E1_2004 CHANNEL  ; 侧压B3左伺服JOG低速
E1_2005 CHANNEL  ; 侧压B3左伺服JOG低速
E1_2006 CHANNEL  ; 侧压B3左伺服加速时间
E1_2007 CHANNEL  ; 侧压B3左伺服加速时间
E1_2008 CHANNEL  ; 侧压B3左伺服减速时间
E1_2009 CHANNEL  ; 侧压B3左伺服减速时间
E1_201 CHANNEL  ; NC433_2_X轴当前位置
E1_2010 CHANNEL  ; 侧压B3左伺服原点偏移
E1_2011 CHANNEL  ; 侧压B3左伺服原点偏移
E1_2012 CHANNEL  ; 侧压B3左伺服正软极限
E1_2013 CHANNEL  ; 侧压B3左伺服正软极限
E1_2014 CHANNEL  ; 侧压B3左伺服负软极限
E1_2015 CHANNEL  ; 负软极限
E1_202 CHANNEL  ; NC433_2_X轴存储器操作正被执行序列号
E1_2020 CHANNEL  ; 侧压B3左伺服待机位
E1_2021 CHANNEL  ; 侧压B3左伺服待机位
E1_2022 CHANNEL  ; 侧压B3左伺服拨料退回位
E1_2023 CHANNEL  ; 侧压B3左伺服拨料退回位
E1_2024 CHANNEL  ; 侧压B3左伺服拨料位
E1_2025 CHANNEL  ; 侧压B3左伺服拨料位
E1_2026 CHANNEL  ; 侧压B3左伺服减速位
E1_2027 CHANNEL  ; 侧压B3左伺服减速位
E1_2028 CHANNEL  ; 侧压B3左伺服等距热压位
E1_2029 CHANNEL  ; 侧压B3左伺服等距热压位
E1_203 CHANNEL  ; NC433_2_X轴存储器操作正被执行序列号
E1_2030 CHANNEL  ; 侧压B3左伺服6#位
E1_2031 CHANNEL  ; 侧压B3左伺服6#位
E1_2032 CHANNEL  ; 侧压B3左伺服7#位
E1_2033 CHANNEL  ; 侧压B3左伺服7#位
E1_2034 CHANNEL  ; 侧压B3左伺服8#位
E1_2035 CHANNEL  ; 侧压B3左伺服8#位
E1_2036 CHANNEL  ; 侧压B3左伺服9#位
E1_2037 CHANNEL  ; 侧压B3左伺服9#位
E1_2038 CHANNEL  ; 侧压B3左伺服10#位
E1_2039 CHANNEL  ; 侧压B3左伺服10#位
E1_204 CHANNEL  ; NC433_2_Y轴当前位置
E1_2046 CHANNEL  ; B3两轴回原宽度
E1_205 CHANNEL  ; NC433_2_Y轴当前位置
E1_2050 CHANNEL  ; 侧压B3右伺服自动速度
E1_2051 CHANNEL  ; 侧压B3右伺服自动速度
E1_2052 CHANNEL  ; 侧压B3右伺服JOG高速
E1_2053 CHANNEL  ; 侧压B3右伺服JOG高速
E1_2054 CHANNEL  ; 侧压B3右伺服JOG低速
E1_2055 CHANNEL  ; 侧压B3右伺服JOG低速
E1_2056 CHANNEL  ; 侧压B3右伺服加速时间
E1_2057 CHANNEL  ; 侧压B3右伺服加速时间
E1_2058 CHANNEL  ; 侧压B3右伺服减速时间
E1_2059 CHANNEL  ; 侧压B3右伺服减速时间
E1_206 CHANNEL  ; NC433_2_Y轴存储器操作正被执行序列号
E1_2060 CHANNEL  ; 侧压B3右伺服原点偏移
E1_2061 CHANNEL  ; 侧压B3右伺服原点偏移
E1_2062 CHANNEL  ; 侧压B3右伺服正软极限
E1_2063 CHANNEL  ; 侧压B3右伺服正软极限
E1_2064 CHANNEL  ; 侧压B3右伺服负软极限
E1_2065 CHANNEL  ; 负软极限
E1_207 CHANNEL  ; NC433_2_Y轴存储器操作正被执行序列号
E1_2070 CHANNEL  ; 侧压B3右伺服待机位
E1_2071 CHANNEL  ; 侧压B3右伺服待机位
E1_2072 CHANNEL  ; 侧压B3右伺服拨料退回位
E1_2073 CHANNEL  ; 侧压B3右伺服拨料退回位
E1_2074 CHANNEL  ; 侧压B3右伺服拨料位
E1_2075 CHANNEL  ; 侧压B3右伺服拨料位
E1_2076 CHANNEL  ; 侧压B3右伺服减速位
E1_2077 CHANNEL  ; 侧压B3右伺服减速位
E1_2078 CHANNEL  ; 侧压B3右伺服等距热压位
E1_2079 CHANNEL  ; 侧压B3右伺服等距热压位
E1_208 CHANNEL  ; NC433_2_Z轴当前位置
E1_2080 CHANNEL  ; 侧压B3右伺服6#位
E1_2081 CHANNEL  ; 侧压B3右伺服6#位
E1_2082 CHANNEL  ; 侧压B3右伺服7#位
E1_2083 CHANNEL  ; 侧压B3右伺服7#位
E1_2084 CHANNEL  ; 侧压B3右伺服8#位
E1_2085 CHANNEL  ; 侧压B3右伺服8#位
E1_2086 CHANNEL  ; 侧压B3右伺服9#位
E1_2087 CHANNEL  ; 侧压B3右伺服9#位
E1_2088 CHANNEL  ; 侧压B3右伺服10#位
E1_2089 CHANNEL  ; 侧压B3右伺服10#位
E1_209 CHANNEL  ; NC433_2_Z轴当前位置
E1_21 CHANNEL  ; NC433_0_Y轴直接操作位置
E1_210 CHANNEL  ; NC433_2_Z轴存储器操作正被执行序列号
E1_2100 CHANNEL  ; 侧压B4左伺服自动速度
E1_2101 CHANNEL  ; 侧压B4左伺服自动速度
E1_2102 CHANNEL  ; 侧压B4左伺服JOG高速
E1_2103 CHANNEL  ; 侧压B4左伺服JOG高速
E1_2104 CHANNEL  ; 侧压B4左伺服JOG低速
E1_2105 CHANNEL  ; 侧压B4左伺服JOG低速
E1_2106 CHANNEL  ; 侧压B4左伺服加速时间
E1_2107 CHANNEL  ; 侧压B4左伺服加速时间
E1_2108 CHANNEL  ; 侧压B4左伺服减速时间
E1_2109 CHANNEL  ; 侧压B4左伺服减速时间
E1_211 CHANNEL  ; NC433_2_Z轴存储器操作正被执行序列号
E1_2110 CHANNEL  ; 侧压B4左伺服原点偏移
E1_2111 CHANNEL  ; 侧压B4左伺服原点偏移
E1_2112 CHANNEL  ; 侧压B4左伺服正软极限
E1_2113 CHANNEL  ; 侧压B4左伺服正软极限
E1_2114 CHANNEL  ; 侧压B4左伺服负软极限
E1_2115 CHANNEL  ; 负软极限
E1_212 CHANNEL  ; NC433_2_U轴当前位置
E1_2120 CHANNEL  ; 侧压B4左伺服待机位
E1_2121 CHANNEL  ; 侧压B4左伺服待机位
E1_2122 CHANNEL  ; 侧压B4左伺服拨料退回位
E1_2123 CHANNEL  ; 侧压B4左伺服拨料退回位
E1_2124 CHANNEL  ; 侧压B4左伺服拨料位
E1_2125 CHANNEL  ; 侧压B4左伺服拨料位
E1_2126 CHANNEL  ; 侧压B4左伺服减速位
E1_2127 CHANNEL  ; 侧压B4左伺服减速位
E1_2128 CHANNEL  ; 侧压B4左伺服等距热压位
E1_2129 CHANNEL  ; 侧压B4左伺服等距热压位
E1_213 CHANNEL  ; NC433_2_U轴当前位置
E1_2130 CHANNEL  ; 侧压B4左伺服6#位
E1_2131 CHANNEL  ; 侧压B4左伺服6#位
E1_2132 CHANNEL  ; 侧压B4左伺服7#位
E1_2133 CHANNEL  ; 侧压B4左伺服7#位
E1_2134 CHANNEL  ; 侧压B4左伺服8#位
E1_2135 CHANNEL  ; 侧压B4左伺服8#位
E1_2136 CHANNEL  ; 侧压B4左伺服9#位
E1_2137 CHANNEL  ; 侧压B4左伺服9#位
E1_2138 CHANNEL  ; 侧压B4左伺服10#位
E1_2139 CHANNEL  ; 侧压B4左伺服10#位
E1_214 CHANNEL  ; NC433_2_U轴存储器操作正被执行序列号
E1_2146 CHANNEL  ; B4两轴回原宽度
E1_215 CHANNEL  ; NC433_2_U轴存储器操作正被执行序列号
E1_2150 CHANNEL  ; 侧压B4右伺服自动速度
E1_2151 CHANNEL  ; 侧压B4右伺服自动速度
E1_2152 CHANNEL  ; 侧压B4右伺服JOG高速
E1_2153 CHANNEL  ; 侧压B4右伺服JOG高速
E1_2154 CHANNEL  ; 侧压B4右伺服JOG低速
E1_2155 CHANNEL  ; 侧压B4右伺服JOG低速
E1_2156 CHANNEL  ; 侧压B4右伺服加速时间
E1_2157 CHANNEL  ; 侧压B4右伺服加速时间
E1_2158 CHANNEL  ; 侧压B4右伺服减速时间
E1_2159 CHANNEL  ; 侧压B4右伺服减速时间
E1_216 CHANNEL  ; NC433_3 数据传送写字数
E1_2160 CHANNEL  ; 侧压B4右伺服原点偏移
E1_2161 CHANNEL  ; 侧压B4右伺服原点偏移
E1_2162 CHANNEL  ; 侧压B4右伺服正软极限
E1_2163 CHANNEL  ; 侧压B4右伺服正软极限
E1_2164 CHANNEL  ; 侧压B4右伺服负软极限
E1_2165 CHANNEL  ; 负软极限
E1_217 CHANNEL  ; NC433_3 数据传送写源区域
E1_2170 CHANNEL  ; 侧压B4右伺服待机位
E1_2171 CHANNEL  ; 侧压B4右伺服待机位
E1_2172 CHANNEL  ; 侧压B4右伺服拨料退回位
E1_2173 CHANNEL  ; 侧压B4右伺服拨料退回位
E1_2174 CHANNEL  ; 侧压B4右伺服拨料位
E1_2175 CHANNEL  ; 侧压B4右伺服拨料位
E1_2176 CHANNEL  ; 侧压B4右伺服减速位
E1_2177 CHANNEL  ; 侧压B4右伺服减速位
E1_2178 CHANNEL  ; 侧压B4右伺服等距热压位
E1_2179 CHANNEL  ; 侧压B4右伺服等距热压位
E1_218 CHANNEL  ; NC433_3 数据传送定源字
E1_2180 CHANNEL  ; 侧压B4右伺服6#位
E1_2181 CHANNEL  ; 侧压B4右伺服6#位
E1_2182 CHANNEL  ; 侧压B4右伺服7#位
E1_2183 CHANNEL  ; 侧压B4右伺服7#位
E1_2184 CHANNEL  ; 侧压B4右伺服8#位
E1_2185 CHANNEL  ; 侧压B4右伺服8#位
E1_2186 CHANNEL  ; 侧压B4右伺服9#位
E1_2187 CHANNEL  ; 侧压B4右伺服9#位
E1_2188 CHANNEL  ; 侧压B4右伺服10#位
E1_2189 CHANNEL  ; 侧压B4右伺服10#位
E1_219 CHANNEL  ; NC433_3 数据传送定目标地址
E1_22 CHANNEL  ; NC433_0_Y轴直接操作速度
E1_220 CHANNEL  ; NC433_3 数据传送读字数
E1_2200 CHANNEL  ; 25#伺服自动速度
E1_2201 CHANNEL  ; 25#伺服自动速度
E1_2202 CHANNEL  ; 25#伺服JOG高速
E1_2203 CHANNEL  ; 25#伺服JOG高速
E1_2204 CHANNEL  ; 25#伺服JOG低速
E1_2205 CHANNEL  ; 25#伺服JOG低速
E1_2206 CHANNEL  ; 25#伺服加速时间
E1_2207 CHANNEL  ; 25#伺服加速时间
E1_2208 CHANNEL  ; 25#伺服减速时间
E1_2209 CHANNEL  ; 25#伺服减速时间
E1_221 CHANNEL  ; NC433_3 数据传送读源区域
E1_2210 CHANNEL  ; 25#伺服原点偏移
E1_2211 CHANNEL  ; 25#伺服原点偏移
E1_2212 CHANNEL  ; 25#伺服正软极限
E1_2213 CHANNEL  ; 25#伺服正软极限
E1_2214 CHANNEL  ; 25#伺服负软极限
E1_2215 CHANNEL  ; 负软极限
E1_222 CHANNEL  ; NC433_3 数据传送读目标区域
E1_2220 CHANNEL  ; 25#伺服1#位
E1_2221 CHANNEL  ; 25#伺服1#位
E1_2222 CHANNEL  ; 25#伺服2#位
E1_2223 CHANNEL  ; 25#伺服2#位
E1_2224 CHANNEL  ; 25#伺服3#位
E1_2225 CHANNEL  ; 25#伺服3#位
E1_2226 CHANNEL  ; 25#伺服4#位
E1_2227 CHANNEL  ; 25#伺服4#位
E1_2228 CHANNEL  ; 25#伺服5#位
E1_2229 CHANNEL  ; 25#伺服5#位
E1_223 CHANNEL  ; NC433_3 数据传送读目标字
E1_2230 CHANNEL  ; 25#伺服6#位
E1_2231 CHANNEL  ; 25#伺服6#位
E1_2232 CHANNEL  ; 25#伺服7#位
E1_2233 CHANNEL  ; 25#伺服7#位
E1_2234 CHANNEL  ; 25#伺服8#位
E1_2235 CHANNEL  ; 25#伺服8#位
E1_2236 CHANNEL  ; 25#伺服9#位
E1_2237 CHANNEL  ; 25#伺服9#位
E1_2238 CHANNEL  ; 25#伺服10#位
E1_2239 CHANNEL  ; 25#伺服10#位
E1_224 CHANNEL  ; NC433_3_X轴直接操作位置
E1_225 CHANNEL  ; NC433_3_X轴直接操作位置
E1_2250 CHANNEL  ; 26#伺服自动速度
E1_2251 CHANNEL  ; 26#伺服自动速度
E1_2252 CHANNEL  ; 26#伺服JOG高速
E1_2253 CHANNEL  ; 26#伺服JOG高速
E1_2254 CHANNEL  ; 26#伺服JOG低速
E1_2255 CHANNEL  ; 26#伺服JOG低速
E1_2256 CHANNEL  ; 26#伺服加速时间
E1_2257 CHANNEL  ; 26#伺服加速时间
E1_2258 CHANNEL  ; 26#伺服减速时间
E1_2259 CHANNEL  ; 26#伺服减速时间
E1_226 CHANNEL  ; NC433_3_X轴直接操作速度
E1_2260 CHANNEL  ; 26#伺服原点偏移
E1_2261 CHANNEL  ; 26#伺服原点偏移
E1_2262 CHANNEL  ; 26#伺服正软极限
E1_2263 CHANNEL  ; 26#伺服正软极限
E1_2264 CHANNEL  ; 26#伺服负软极限
E1_2265 CHANNEL  ; 负软极限
E1_227 CHANNEL  ; NC433_3_X轴直接操作速度
E1_2270 CHANNEL  ; 26#伺服1#位
E1_2271 CHANNEL  ; 26#伺服1#位
E1_2272 CHANNEL  ; 26#伺服2#位
E1_2273 CHANNEL  ; 26#伺服2#位
E1_2274 CHANNEL  ; 26#伺服3#位
E1_2275 CHANNEL  ; 26#伺服3#位
E1_2276 CHANNEL  ; 26#伺服4#位
E1_2277 CHANNEL  ; 26#伺服4#位
E1_2278 CHANNEL  ; 26#伺服5#位
E1_2279 CHANNEL  ; 26#伺服5#位
E1_228 CHANNEL  ; NC433_3_X轴直接操作加速时间
E1_2280 CHANNEL  ; 26#伺服6#位
E1_2281 CHANNEL  ; 26#伺服6#位
E1_2282 CHANNEL  ; 26#伺服7#位
E1_2283 CHANNEL  ; 26#伺服7#位
E1_2284 CHANNEL  ; 26#伺服8#位
E1_2285 CHANNEL  ; 26#伺服8#位
E1_2286 CHANNEL  ; 26#伺服9#位
E1_2287 CHANNEL  ; 26#伺服9#位
E1_2288 CHANNEL  ; 26#伺服10#位
E1_2289 CHANNEL  ; 26#伺服10#位
E1_229 CHANNEL  ; NC433_3_X轴直接操作加速时间
E1_23 CHANNEL  ; NC433_0_Y轴直接操作速度
E1_230 CHANNEL  ; NC433_3_X轴直接操作减速时间
E1_2300 CHANNEL  ; 27#伺服自动速度
E1_2301 CHANNEL  ; 27#伺服自动速度
E1_2302 CHANNEL  ; 27#伺服JOG高速
E1_2303 CHANNEL  ; 27#伺服JOG高速
E1_2304 CHANNEL  ; 27#伺服JOG低速
E1_2305 CHANNEL  ; 27#伺服JOG低速
E1_2306 CHANNEL  ; 27#伺服加速时间
E1_2307 CHANNEL  ; 27#伺服加速时间
E1_2308 CHANNEL  ; 27#伺服减速时间
E1_2309 CHANNEL  ; 27#伺服减速时间
E1_231 CHANNEL  ; NC433_3_X轴直接操作减速时间
E1_2310 CHANNEL  ; 27#伺服原点偏移
E1_2311 CHANNEL  ; 27#伺服原点偏移
E1_2312 CHANNEL  ; 27#伺服正软极限
E1_2313 CHANNEL  ; 27#伺服正软极限
E1_2314 CHANNEL  ; 27#伺服负软极限
E1_2315 CHANNEL  ; 负软极限
E1_232 CHANNEL  ; NC433_3_X轴存储器操作序列号
E1_2320 CHANNEL  ; 27#伺服1#位
E1_2321 CHANNEL  ; 27#伺服1#位
E1_2322 CHANNEL  ; 27#伺服2#位
E1_2323 CHANNEL  ; 27#伺服2#位
E1_2324 CHANNEL  ; 27#伺服3#位
E1_2325 CHANNEL  ; 27#伺服3#位
E1_2326 CHANNEL  ; 27#伺服4#位
E1_2327 CHANNEL  ; 27#伺服4#位
E1_2328 CHANNEL  ; 27#伺服5#位
E1_2329 CHANNEL  ; 27#伺服5#位
E1_233 CHANNEL  ; NC433_3_X轴特殊操作Override
E1_2330 CHANNEL  ; 27#伺服6#位
E1_2331 CHANNEL  ; 27#伺服6#位
E1_2332 CHANNEL  ; 27#伺服7#位
E1_2333 CHANNEL  ; 27#伺服7#位
E1_2334 CHANNEL  ; 27#伺服8#位
E1_2335 CHANNEL  ; 27#伺服8#位
E1_2336 CHANNEL  ; 27#伺服9#位
E1_2337 CHANNEL  ; 27#伺服9#位
E1_2338 CHANNEL  ; 27#伺服10#位
E1_2339 CHANNEL  ; 27#伺服10#位
E1_234 CHANNEL  ; NC433_3_X轴特殊操作示教地址
E1_235 CHANNEL  ; NC433_3_X轴特殊操作预留
E1_2350 CHANNEL  ; 接料伺服自动速度
E1_2351 CHANNEL  ; 接料伺服自动速度
E1_2352 CHANNEL  ; 接料伺服JOG高速
E1_2353 CHANNEL  ; 接料伺服JOG高速
E1_2354 CHANNEL  ; 接料伺服JOG低速
E1_2355 CHANNEL  ; 接料伺服JOG低速
E1_2356 CHANNEL  ; 接料伺服加速时间
E1_2357 CHANNEL  ; 接料伺服加速时间
E1_2358 CHANNEL  ; 接料伺服减速时间
E1_2359 CHANNEL  ; 接料伺服减速时间
E1_236 CHANNEL  ; NC433_3_Y轴直接操作位置
E1_2360 CHANNEL  ; 接料伺服原点偏移
E1_2361 CHANNEL  ; 接料伺服原点偏移
E1_2362 CHANNEL  ; 接料伺服正软极限
E1_2363 CHANNEL  ; 接料伺服正软极限
E1_2364 CHANNEL  ; 接料伺服负软极限
E1_2365 CHANNEL  ; 负软极限
E1_237 CHANNEL  ; NC433_3_Y轴直接操作位置
E1_2370 CHANNEL  ; 接料伺服出料位
E1_2371 CHANNEL  ; 接料伺服出料位
E1_2372 CHANNEL  ; 接料伺服接料位
E1_2373 CHANNEL  ; 接料伺服接料位
E1_2374 CHANNEL  ; 接料伺服3#位
E1_2375 CHANNEL  ; 接料伺服3#位
E1_2376 CHANNEL  ; 接料伺服4#位
E1_2377 CHANNEL  ; 接料伺服4#位
E1_2378 CHANNEL  ; 接料伺服5#位
E1_2379 CHANNEL  ; 接料伺服5#位
E1_238 CHANNEL  ; NC433_3_Y轴直接操作速度
E1_2380 CHANNEL  ; 接料伺服6#位
E1_2381 CHANNEL  ; 接料伺服6#位
E1_2382 CHANNEL  ; 接料伺服7#位
E1_2383 CHANNEL  ; 接料伺服7#位
E1_2384 CHANNEL  ; 接料伺服8#位
E1_2385 CHANNEL  ; 接料伺服8#位
E1_2386 CHANNEL  ; 接料伺服9#位
E1_2387 CHANNEL  ; 接料伺服9#位
E1_2388 CHANNEL  ; 接料伺服10#位
E1_2389 CHANNEL  ; 接料伺服10#位
E1_239 CHANNEL  ; NC433_3_Y轴直接操作速度
E1_24 CHANNEL  ; NC433_0_Y轴直接操作加速时间
E1_240 CHANNEL  ; NC433_3_Y轴直接操作加速时间
E1_241 CHANNEL  ; NC433_3_Y轴直接操作加速时间
E1_242 CHANNEL  ; NC433_3_Y轴直接操作减速时间
E1_243 CHANNEL  ; NC433_3_Y轴直接操作减速时间
E1_244 CHANNEL  ; NC433_3_Y轴存储器操作序列号
E1_245 CHANNEL  ; NC433_3_Y轴特殊操作Override
E1_246 CHANNEL  ; NC433_3_Y轴特殊操作示教地址
E1_247 CHANNEL  ; NC433_3_Y轴特殊操作预留
E1_248 CHANNEL  ; NC433_3_Z轴直接操作位置
E1_249 CHANNEL  ; NC433_3_Z轴直接操作位置
E1_25 CHANNEL  ; NC433_0_Y轴直接操作加速时间
E1_250 CHANNEL  ; NC433_3_Z轴直接操作速度
E1_251 CHANNEL  ; NC433_3_Z轴直接操作速度
E1_252 CHANNEL  ; NC433_3_Z轴直接操作加速时间
E1_253 CHANNEL  ; NC433_3_Z轴直接操作加速时间
E1_254 CHANNEL  ; NC433_3_Z轴直接操作减速时间
E1_255 CHANNEL  ; NC433_3_Z轴直接操作减速时间
E1_256 CHANNEL  ; NC433_3_Z轴存储器操作序列号
E1_257 CHANNEL  ; NC433_3_Z轴特殊操作Override
E1_258 CHANNEL  ; NC433_3_Z轴特殊操作示教地址
E1_259 CHANNEL  ; NC433_3_Z轴特殊操作预留
E1_26 CHANNEL  ; NC433_0_Y轴直接操作减速时间
E1_260 CHANNEL  ; NC433_3_U轴直接操作位置
E1_261 CHANNEL  ; NC433_3_U轴直接操作位置
E1_262 CHANNEL  ; NC433_3_U轴直接操作速度
E1_263 CHANNEL  ; NC433_3_U轴直接操作速度
E1_264 CHANNEL  ; NC433_3_U轴直接操作加速时间
E1_265 CHANNEL  ; NC433_3_U轴直接操作加速时间
E1_266 CHANNEL  ; NC433_3_U轴直接操作减速时间
E1_267 CHANNEL  ; NC433_3_U轴直接操作减速时间
E1_268 CHANNEL  ; NC433_3_U轴存储器操作序列号
E1_269 CHANNEL  ; NC433_3_U轴特殊操作Override
E1_27 CHANNEL  ; NC433_0_Y轴直接操作减速时间
E1_270 CHANNEL  ; NC433_3_U轴特殊操作示教地址
E1_271 CHANNEL  ; NC433_3_U轴特殊操作预留
E1_272 CHANNEL  ; NC433_3_X轴当前位置
E1_273 CHANNEL  ; NC433_3_X轴当前位置
E1_274 CHANNEL  ; NC433_3_X轴存储器操作正被执行序列号
E1_275 CHANNEL  ; NC433_3_X轴存储器操作正被执行序列号
E1_276 CHANNEL  ; NC433_3_Y轴当前位置
E1_277 CHANNEL  ; NC433_3_Y轴当前位置
E1_278 CHANNEL  ; NC433_3_Y轴存储器操作正被执行序列号
E1_279 CHANNEL  ; NC433_3_Y轴存储器操作正被执行序列号
E1_28 CHANNEL  ; NC433_0_Y轴存储器操作序列号
E1_280 CHANNEL  ; NC433_3_Z轴当前位置
E1_281 CHANNEL  ; NC433_3_Z轴当前位置
E1_282 CHANNEL  ; NC433_3_Z轴存储器操作正被执行序列号
E1_283 CHANNEL  ; NC433_3_Z轴存储器操作正被执行序列号
E1_284 CHANNEL  ; NC433_3_U轴当前位置
E1_285 CHANNEL  ; NC433_3_U轴当前位置
E1_286 CHANNEL  ; NC433_3_U轴存储器操作正被执行序列号
E1_287 CHANNEL  ; NC433_3_U轴存储器操作正被执行序列号
E1_288 CHANNEL  ; NC433_4 数据传送写字数
E1_289 CHANNEL  ; NC433_4 数据传送写源区域
E1_29 CHANNEL  ; NC433_0_Y轴特殊操作Override
E1_290 CHANNEL  ; NC433_4 数据传送定源字
E1_2900 CHANNEL  ; A1两轴运行宽度
E1_2902 CHANNEL  ; A1单轴运行宽度
E1_291 CHANNEL  ; NC433_4 数据传送定目标地址
E1_2910 CHANNEL  ; A2两轴运行宽度
E1_2912 CHANNEL  ; A2单轴运行宽度
E1_292 CHANNEL  ; NC433_4 数据传送读字数
E1_2920 CHANNEL  ; A3两轴运行宽度
E1_2922 CHANNEL  ; A3单轴运行宽度
E1_293 CHANNEL  ; NC433_4 数据传送读源区域
E1_2930 CHANNEL  ; A4两轴运行宽度
E1_2932 CHANNEL  ; A4单轴运行宽度
E1_294 CHANNEL  ; NC433_4 数据传送读目标区域
E1_295 CHANNEL  ; NC433_4 数据传送读目标字
E1_2950 CHANNEL  ; B1两轴运行宽度
E1_2952 CHANNEL  ; B1单轴运行宽度
E1_296 CHANNEL  ; NC433_4_X轴直接操作位置
E1_2960 CHANNEL  ; B2两轴运行宽度
E1_2962 CHANNEL  ; B2单轴运行宽度
E1_297 CHANNEL  ; NC433_4_X轴直接操作位置
E1_2970 CHANNEL  ; B3两轴运行宽度
E1_2972 CHANNEL  ; B3单轴运行宽度
E1_298 CHANNEL  ; NC433_4_X轴直接操作速度
E1_2980 CHANNEL  ; B4两轴运行宽度
E1_2982 CHANNEL  ; B3单轴运行宽度
E1_299 CHANNEL  ; NC433_4_X轴直接操作速度
E1_3 CHANNEL  ; NC433_0 数据传送定目标地址
E1_30 CHANNEL  ; NC433_0_Y轴特殊操作示教地址
E1_300 CHANNEL  ; NC433_4_X轴直接操作加速时间
E1_301 CHANNEL  ; NC433_4_X轴直接操作加速时间
E1_302 CHANNEL  ; NC433_4_X轴直接操作减速时间
E1_303 CHANNEL  ; NC433_4_X轴直接操作减速时间
E1_304 CHANNEL  ; NC433_4_X轴存储器操作序列号
E1_305 CHANNEL  ; NC433_4_X轴特殊操作Override
E1_306 CHANNEL  ; NC433_4_X轴特殊操作示教地址
E1_307 CHANNEL  ; NC433_4_X轴特殊操作预留
E1_308 CHANNEL  ; NC433_4_Y轴直接操作位置
E1_309 CHANNEL  ; NC433_4_Y轴直接操作位置
E1_31 CHANNEL  ; NC433_0_Y轴特殊操作预留
E1_310 CHANNEL  ; NC433_4_Y轴直接操作速度
E1_311 CHANNEL  ; NC433_4_Y轴直接操作速度
E1_312 CHANNEL  ; NC433_4_Y轴直接操作加速时间
E1_313 CHANNEL  ; NC433_4_Y轴直接操作加速时间
E1_314 CHANNEL  ; NC433_4_Y轴直接操作减速时间
E1_315 CHANNEL  ; NC433_4_Y轴直接操作减速时间
E1_316 CHANNEL  ; NC433_4_Y轴存储器操作序列号
E1_317 CHANNEL  ; NC433_4_Y轴特殊操作Override
E1_318 CHANNEL  ; NC433_4_Y轴特殊操作示教地址
E1_319 CHANNEL  ; NC433_4_Y轴特殊操作预留
E1_32 CHANNEL  ; NC433_0_Z轴直接操作位置
E1_320 CHANNEL  ; NC433_4_Z轴直接操作位置
E1_321 CHANNEL  ; NC433_4_Z轴直接操作位置
E1_322 CHANNEL  ; NC433_4_Z轴直接操作速度
E1_323 CHANNEL  ; NC433_4_Z轴直接操作速度
E1_324 CHANNEL  ; NC433_4_Z轴直接操作加速时间
E1_325 CHANNEL  ; NC433_4_Z轴直接操作加速时间
E1_326 CHANNEL  ; NC433_4_Z轴直接操作减速时间
E1_327 CHANNEL  ; NC433_4_Z轴直接操作减速时间
E1_328 CHANNEL  ; NC433_4_Z轴存储器操作序列号
E1_329 CHANNEL  ; NC433_4_Z轴特殊操作Override
E1_33 CHANNEL  ; NC433_0_Z轴直接操作位置
E1_330 CHANNEL  ; NC433_4_Z轴特殊操作示教地址
E1_331 CHANNEL  ; NC433_4_Z轴特殊操作预留
E1_332 CHANNEL  ; NC433_4_U轴直接操作位置
E1_333 CHANNEL  ; NC433_4_U轴直接操作位置
E1_334 CHANNEL  ; NC433_4_U轴直接操作速度
E1_335 CHANNEL  ; NC433_4_U轴直接操作速度
E1_336 CHANNEL  ; NC433_4_U轴直接操作加速时间
E1_337 CHANNEL  ; NC433_4_U轴直接操作加速时间
E1_338 CHANNEL  ; NC433_4_U轴直接操作减速时间
E1_339 CHANNEL  ; NC433_4_U轴直接操作减速时间
E1_34 CHANNEL  ; NC433_0_Z轴直接操作速度
E1_340 CHANNEL  ; NC433_4_U轴存储器操作序列号
E1_341 CHANNEL  ; NC433_4_U轴特殊操作Override
E1_342 CHANNEL  ; NC433_4_U轴特殊操作示教地址
E1_343 CHANNEL  ; NC433_4_U轴特殊操作预留
E1_344 CHANNEL  ; NC433_4_X轴当前位置
E1_345 CHANNEL  ; NC433_4_X轴当前位置
E1_346 CHANNEL  ; NC433_4_X轴存储器操作正被执行序列号
E1_347 CHANNEL  ; NC433_4_X轴存储器操作正被执行序列号
E1_348 CHANNEL  ; NC433_4_Y轴当前位置
E1_349 CHANNEL  ; NC433_4_Y轴当前位置
E1_35 CHANNEL  ; NC433_0_Z轴直接操作速度
E1_350 CHANNEL  ; NC433_4_Y轴存储器操作正被执行序列号
E1_351 CHANNEL  ; NC433_4_Y轴存储器操作正被执行序列号
E1_352 CHANNEL  ; NC433_4_Z轴当前位置
E1_353 CHANNEL  ; NC433_4_Z轴当前位置
E1_354 CHANNEL  ; NC433_4_Z轴存储器操作正被执行序列号
E1_355 CHANNEL  ; NC433_4_Z轴存储器操作正被执行序列号
E1_356 CHANNEL  ; NC433_4_U轴当前位置
E1_357 CHANNEL  ; NC433_4_U轴当前位置
E1_358 CHANNEL  ; NC433_4_U轴存储器操作正被执行序列号
E1_359 CHANNEL  ; NC433_4_U轴存储器操作正被执行序列号
E1_36 CHANNEL  ; NC433_0_Z轴直接操作加速时间
E1_360 CHANNEL  ; NC433_5 数据传送写字数
E1_361 CHANNEL  ; NC433_5 数据传送写源区域
E1_362 CHANNEL  ; NC433_5 数据传送定源字
E1_363 CHANNEL  ; NC433_5 数据传送定目标地址
E1_364 CHANNEL  ; NC433_5 数据传送读字数
E1_365 CHANNEL  ; NC433_5 数据传送读源区域
E1_366 CHANNEL  ; NC433_5 数据传送读目标区域
E1_367 CHANNEL  ; NC433_5 数据传送读目标字
E1_368 CHANNEL  ; NC433_5_X轴直接操作位置
E1_369 CHANNEL  ; NC433_5_X轴直接操作位置
E1_37 CHANNEL  ; NC433_0_Z轴直接操作加速时间
E1_370 CHANNEL  ; NC433_5_X轴直接操作速度
E1_371 CHANNEL  ; NC433_5_X轴直接操作速度
E1_372 CHANNEL  ; NC433_5_X轴直接操作加速时间
E1_373 CHANNEL  ; NC433_5_X轴直接操作加速时间
E1_374 CHANNEL  ; NC433_5_X轴直接操作减速时间
E1_375 CHANNEL  ; NC433_5_X轴直接操作减速时间
E1_376 CHANNEL  ; NC433_5_X轴存储器操作序列号
E1_377 CHANNEL  ; NC433_5_X轴特殊操作Override
E1_378 CHANNEL  ; NC433_5_X轴特殊操作示教地址
E1_379 CHANNEL  ; NC433_5_X轴特殊操作预留
E1_38 CHANNEL  ; NC433_0_Z轴直接操作减速时间
E1_380 CHANNEL  ; NC433_5_Y轴直接操作位置
E1_381 CHANNEL  ; NC433_5_Y轴直接操作位置
E1_382 CHANNEL  ; NC433_5_Y轴直接操作速度
E1_383 CHANNEL  ; NC433_5_Y轴直接操作速度
E1_384 CHANNEL  ; NC433_5_Y轴直接操作加速时间
E1_385 CHANNEL  ; NC433_5_Y轴直接操作加速时间
E1_386 CHANNEL  ; NC433_5_Y轴直接操作减速时间
E1_387 CHANNEL  ; NC433_5_Y轴直接操作减速时间
E1_388 CHANNEL  ; NC433_5_Y轴存储器操作序列号
E1_389 CHANNEL  ; NC433_5_Y轴特殊操作Override
E1_39 CHANNEL  ; NC433_0_Z轴直接操作减速时间
E1_390 CHANNEL  ; NC433_5_Y轴特殊操作示教地址
E1_391 CHANNEL  ; NC433_5_Y轴特殊操作预留
E1_392 CHANNEL  ; NC433_5_Z轴直接操作位置
E1_393 CHANNEL  ; NC433_5_Z轴直接操作位置
E1_394 CHANNEL  ; NC433_5_Z轴直接操作速度
E1_395 CHANNEL  ; NC433_5_Z轴直接操作速度
E1_396 CHANNEL  ; NC433_5_Z轴直接操作加速时间
E1_397 CHANNEL  ; NC433_5_Z轴直接操作加速时间
E1_398 CHANNEL  ; NC433_5_Z轴直接操作减速时间
E1_399 CHANNEL  ; NC433_5_Z轴直接操作减速时间
E1_4 CHANNEL  ; NC433_0 数据传送读字数
E1_40 CHANNEL  ; NC433_0_Z轴存储器操作序列号
E1_400 CHANNEL  ; NC433_5_Z轴存储器操作序列号
E1_401 CHANNEL  ; NC433_5_Z轴特殊操作Override
E1_402 CHANNEL  ; NC433_5_Z轴特殊操作示教地址
E1_403 CHANNEL  ; NC433_5_Z轴特殊操作预留
E1_404 CHANNEL  ; NC433_5_U轴直接操作位置
E1_405 CHANNEL  ; NC433_5_U轴直接操作位置
E1_406 CHANNEL  ; NC433_5_U轴直接操作速度
E1_407 CHANNEL  ; NC433_5_U轴直接操作速度
E1_408 CHANNEL  ; NC433_5_U轴直接操作加速时间
E1_409 CHANNEL  ; NC433_5_U轴直接操作加速时间
E1_41 CHANNEL  ; NC433_0_Z轴特殊操作Override
E1_410 CHANNEL  ; NC433_5_U轴直接操作减速时间
E1_411 CHANNEL  ; NC433_5_U轴直接操作减速时间
E1_412 CHANNEL  ; NC433_5_U轴存储器操作序列号
E1_413 CHANNEL  ; NC433_5_U轴特殊操作Override
E1_414 CHANNEL  ; NC433_5_U轴特殊操作示教地址
E1_415 CHANNEL  ; NC433_5_U轴特殊操作预留
E1_416 CHANNEL  ; NC433_5_X轴当前位置
E1_417 CHANNEL  ; NC433_5_X轴当前位置
E1_418 CHANNEL  ; NC433_5_X轴存储器操作正被执行序列号
E1_419 CHANNEL  ; NC433_5_X轴存储器操作正被执行序列号
E1_42 CHANNEL  ; NC433_0_Z轴特殊操作示教地址
E1_420 CHANNEL  ; NC433_5_Y轴当前位置
E1_421 CHANNEL  ; NC433_5_Y轴当前位置
E1_422 CHANNEL  ; NC433_5_Y轴存储器操作正被执行序列号
E1_423 CHANNEL  ; NC433_5_Y轴存储器操作正被执行序列号
E1_424 CHANNEL  ; NC433_5_Z轴当前位置
E1_425 CHANNEL  ; NC433_5_Z轴当前位置
E1_426 CHANNEL  ; NC433_5_Z轴存储器操作正被执行序列号
E1_427 CHANNEL  ; NC433_5_Z轴存储器操作正被执行序列号
E1_428 CHANNEL  ; NC433_5_U轴当前位置
E1_429 CHANNEL  ; NC433_5_U轴当前位置
E1_43 CHANNEL  ; NC433_0_Z轴特殊操作预留
E1_430 CHANNEL  ; NC433_5_U轴存储器操作正被执行序列号
E1_431 CHANNEL  ; NC433_5_U轴存储器操作正被执行序列号
E1_432 CHANNEL  ; NC433_6 数据传送写字数
E1_433 CHANNEL  ; NC433_6 数据传送写源区域
E1_434 CHANNEL  ; NC433_6 数据传送定源字
E1_435 CHANNEL  ; NC433_6 数据传送定目标地址
E1_436 CHANNEL  ; NC433_6 数据传送读字数
E1_437 CHANNEL  ; NC433_6 数据传送读源区域
E1_438 CHANNEL  ; NC433_6 数据传送读目标区域
E1_439 CHANNEL  ; NC433_6 数据传送读目标字
E1_44 CHANNEL  ; NC433_0_U轴直接操作位置
E1_440 CHANNEL  ; NC433_6_X轴直接操作位置
E1_441 CHANNEL  ; NC433_6_X轴直接操作位置
E1_442 CHANNEL  ; NC433_6_X轴直接操作速度
E1_443 CHANNEL  ; NC433_6_X轴直接操作速度
E1_444 CHANNEL  ; NC433_6_X轴直接操作加速时间
E1_445 CHANNEL  ; NC433_6_X轴直接操作加速时间
E1_446 CHANNEL  ; NC433_6_X轴直接操作减速时间
E1_447 CHANNEL  ; NC433_6_X轴直接操作减速时间
E1_448 CHANNEL  ; NC433_6_X轴存储器操作序列号
E1_449 CHANNEL  ; NC433_6_X轴特殊操作Override
E1_45 CHANNEL  ; NC433_0_U轴直接操作位置
E1_450 CHANNEL  ; NC433_6_X轴特殊操作示教地址
E1_451 CHANNEL  ; NC433_6_X轴特殊操作预留
E1_452 CHANNEL  ; NC433_6_Y轴直接操作位置
E1_453 CHANNEL  ; NC433_6_Y轴直接操作位置
E1_454 CHANNEL  ; NC433_6_Y轴直接操作速度
E1_455 CHANNEL  ; NC433_6_Y轴直接操作速度
E1_456 CHANNEL  ; NC433_6_Y轴直接操作加速时间
E1_457 CHANNEL  ; NC433_6_Y轴直接操作加速时间
E1_458 CHANNEL  ; NC433_6_Y轴直接操作减速时间
E1_459 CHANNEL  ; NC433_6_Y轴直接操作减速时间
E1_46 CHANNEL  ; NC433_0_U轴直接操作速度
E1_460 CHANNEL  ; NC433_6_Y轴存储器操作序列号
E1_461 CHANNEL  ; NC433_6_Y轴特殊操作Override
E1_462 CHANNEL  ; NC433_6_Y轴特殊操作示教地址
E1_463 CHANNEL  ; NC433_6_Y轴特殊操作预留
E1_464 CHANNEL  ; NC433_6_Z轴直接操作位置
E1_465 CHANNEL  ; NC433_6_Z轴直接操作位置
E1_466 CHANNEL  ; NC433_6_Z轴直接操作速度
E1_467 CHANNEL  ; NC433_6_Z轴直接操作速度
E1_468 CHANNEL  ; NC433_6_Z轴直接操作加速时间
E1_469 CHANNEL  ; NC433_6_Z轴直接操作加速时间
E1_47 CHANNEL  ; NC433_0_U轴直接操作速度
E1_470 CHANNEL  ; NC433_6_Z轴直接操作减速时间
E1_471 CHANNEL  ; NC433_6_Z轴直接操作减速时间
E1_472 CHANNEL  ; NC433_6_Z轴存储器操作序列号
E1_473 CHANNEL  ; NC433_6_Z轴特殊操作Override
E1_474 CHANNEL  ; NC433_6_Z轴特殊操作示教地址
E1_475 CHANNEL  ; NC433_6_Z轴特殊操作预留
E1_476 CHANNEL  ; NC433_6_U轴直接操作位置
E1_477 CHANNEL  ; NC433_6_U轴直接操作位置
E1_478 CHANNEL  ; NC433_6_U轴直接操作速度
E1_479 CHANNEL  ; NC433_6_U轴直接操作速度
E1_48 CHANNEL  ; NC433_0_U轴直接操作加速时间
E1_480 CHANNEL  ; NC433_6_U轴直接操作加速时间
E1_481 CHANNEL  ; NC433_6_U轴直接操作加速时间
E1_482 CHANNEL  ; NC433_6_U轴直接操作减速时间
E1_483 CHANNEL  ; NC433_6_U轴直接操作减速时间
E1_484 CHANNEL  ; NC433_6_U轴存储器操作序列号
E1_485 CHANNEL  ; NC433_6_U轴特殊操作Override
E1_486 CHANNEL  ; NC433_6_U轴特殊操作示教地址
E1_487 CHANNEL  ; NC433_6_U轴特殊操作预留
E1_488 CHANNEL  ; NC433_6_X轴当前位置
E1_489 CHANNEL  ; NC433_6_X轴当前位置
E1_49 CHANNEL  ; NC433_0_U轴直接操作加速时间
E1_490 CHANNEL  ; NC433_6_X轴存储器操作正被执行序列号
E1_491 CHANNEL  ; NC433_6_X轴存储器操作正被执行序列号
E1_492 CHANNEL  ; NC433_6_Y轴当前位置
E1_493 CHANNEL  ; NC433_6_Y轴当前位置
E1_494 CHANNEL  ; NC433_6_Y轴存储器操作正被执行序列号
E1_495 CHANNEL  ; NC433_6_Y轴存储器操作正被执行序列号
E1_496 CHANNEL  ; NC433_6_Z轴当前位置
E1_497 CHANNEL  ; NC433_6_Z轴当前位置
E1_498 CHANNEL  ; NC433_6_Z轴存储器操作正被执行序列号
E1_499 CHANNEL  ; NC433_6_Z轴存储器操作正被执行序列号
E1_5 CHANNEL  ; NC433_0 数据传送读源区域
E1_50 CHANNEL  ; NC433_0_U轴直接操作减速时间
E1_500 CHANNEL  ; NC433_6_U轴当前位置
E1_501 CHANNEL  ; NC433_6_U轴当前位置
E1_502 CHANNEL  ; NC433_6_U轴存储器操作正被执行序列号
E1_503 CHANNEL  ; NC433_6_U轴存储器操作正被执行序列号
E1_51 CHANNEL  ; NC433_0_U轴直接操作减速时间
E1_52 CHANNEL  ; NC433_0_U轴存储器操作序列号
E1_53 CHANNEL  ; NC433_0_U轴特殊操作Override
E1_54 CHANNEL  ; NC433_0_U轴特殊操作示教地址
E1_55 CHANNEL  ; NC433_0_U轴特殊操作预留
E1_56 CHANNEL  ; NC433_0_X轴当前位置
E1_57 CHANNEL  ; NC433_0_X轴当前位置
E1_58 CHANNEL  ; NC433_0_X轴存储器操作正被执行序列号
E1_59 CHANNEL  ; NC433_0_X轴存储器操作正被执行序列号
E1_6 CHANNEL  ; NC433_0 数据传送读目标区域
E1_60 CHANNEL  ; NC433_0_Y轴当前位置
E1_61 CHANNEL  ; NC433_0_Y轴当前位置
E1_62 CHANNEL  ; NC433_0_Y轴存储器操作正被执行序列号
E1_63 CHANNEL  ; NC433_0_Y轴存储器操作正被执行序列号
E1_64 CHANNEL  ; NC433_0_Z轴当前位置
E1_65 CHANNEL  ; NC433_0_Z轴当前位置
E1_66 CHANNEL  ; NC433_0_Z轴存储器操作正被执行序列号
E1_67 CHANNEL  ; NC433_0_Z轴存储器操作正被执行序列号
E1_68 CHANNEL  ; NC433_0_U轴当前位置
E1_69 CHANNEL  ; NC433_0_U轴当前位置
E1_7 CHANNEL  ; NC433_0 数据传送读目标字
E1_70 CHANNEL  ; NC433_0_U轴存储器操作正被执行序列号
E1_71 CHANNEL  ; NC433_0_U轴存储器操作正被执行序列号
E1_72 CHANNEL  ; NC433_1 数据传送写字数
E1_73 CHANNEL  ; NC433_1 数据传送写源区域
E1_74 CHANNEL  ; NC433_1 数据传送定源字
E1_75 CHANNEL  ; NC433_1 数据传送定目标地址
E1_76 CHANNEL  ; NC433_1 数据传送读字数
E1_77 CHANNEL  ; NC433_1 数据传送读源区域
E1_78 CHANNEL  ; NC433_1 数据传送读目标区域
E1_79 CHANNEL  ; NC433_1 数据传送读目标字
E1_8 CHANNEL  ; NC433_0_X轴直接操作位置
E1_80 CHANNEL  ; NC433_1_X轴直接操作位置
E1_81 CHANNEL  ; NC433_1_X轴直接操作位置
E1_82 CHANNEL  ; NC433_1_X轴直接操作速度
E1_83 CHANNEL  ; NC433_1_X轴直接操作速度
E1_84 CHANNEL  ; NC433_1_X轴直接操作加速时间
E1_85 CHANNEL  ; NC433_1_X轴直接操作加速时间
E1_86 CHANNEL  ; NC433_1_X轴直接操作减速时间
E1_87 CHANNEL  ; NC433_1_X轴直接操作减速时间
E1_88 CHANNEL  ; NC433_1_X轴存储器操作序列号
E1_89 CHANNEL  ; NC433_1_X轴特殊操作Override
E1_9 CHANNEL  ; NC433_0_X轴直接操作位置
E1_90 CHANNEL  ; NC433_1_X轴特殊操作示教地址
E1_91 CHANNEL  ; NC433_1_X轴特殊操作预留
E1_92 CHANNEL  ; NC433_1_Y轴直接操作位置
E1_93 CHANNEL  ; NC433_1_Y轴直接操作位置
E1_94 CHANNEL  ; NC433_1_Y轴直接操作速度
E1_95 CHANNEL  ; NC433_1_Y轴直接操作速度
E1_96 CHANNEL  ; NC433_1_Y轴直接操作加速时间
E1_97 CHANNEL  ; NC433_1_Y轴直接操作加速时间
E1_98 CHANNEL  ; NC433_1_Y轴直接操作减速时间
E1_99 CHANNEL  ; NC433_1_Y轴直接操作减速时间
H0.00 BOOL  ; 手动运行
H0.04 BOOL  ; 副急停屏蔽
H0.06 BOOL  ; 无使用信号小屏禁止使用
H0.09 BOOL  ; 气缸保持（1保持）
H0.14 BOOL  ; 调出
H100.00 BOOL  ; 夹爪1有料记忆
H100.01 BOOL  ; 夹爪2有料记忆
H100.02 BOOL  ; 夹爪3有料记忆
H100.03 BOOL  ; 夹爪4有料记忆
H100.04 BOOL  ; 夹爪5有料记忆
H101 CHANNEL  ; 下料机器人有工艺NG电芯记忆
H101.00 BOOL  ; 夹爪1有工艺NG电芯记忆
H101.01 BOOL  ; 夹爪2有工艺NG电芯记忆
H101.02 BOOL  ; 夹爪3有工艺NG电芯记忆
H101.03 BOOL  ; 夹爪4有工艺NG电芯记忆
H101.04 BOOL  ; 夹爪5有工艺NG电芯记忆
H102 CHANNEL  ; 下料机器人有HipotNG电芯记忆
H102.00 BOOL  ; 夹爪1有HipotNG电芯记忆
H102.01 BOOL  ; 夹爪2有HipotNG电芯记忆
H102.02 BOOL  ; 夹爪3有HipotNG电芯记忆
H102.03 BOOL  ; 夹爪4有HipotNG电芯记忆
H102.04 BOOL  ; 夹爪5有HipotNG电芯记忆
H103 CHANNEL  ; 下料机器人有OK电芯记忆
H103.00 BOOL  ; 夹爪1有OK电芯记忆
H103.01 BOOL  ; 夹爪2有OK电芯记忆
H103.02 BOOL  ; 夹爪3有OK电芯记忆
H103.03 BOOL  ; 夹爪4有OK电芯记忆
H103.04 BOOL  ; 夹爪5有OK电芯记忆
H104.00 BOOL  ; A边已抓
H10.00 BOOL  ; $?St$Bk?_#[468] / 上料机器人有电芯记忆 / $?St$Bk?_#[468]
H10.03 BOOL  ; 放料A已放
H10.04 BOOL  ; 取料A已抓
H11 CHANNEL  ; 上料夹爪扫码NG记忆
H110 CHANNEL  ; A1取料位扫码OK记忆
H110.00 BOOL  ; A1扫码OK
H110.01 BOOL  ; A2扫码OK
H110.02 BOOL  ; A3扫码OK
H110.03 BOOL  ; A4扫码OK
H110.04 BOOL  ; A5扫码OK
H111 CHANNEL  ; A1取料位扫码NG记忆
H111.00 BOOL  ; A1扫码NG
H111.01 BOOL  ; A2扫码NG
H111.02 BOOL  ; A3扫码NG
H111.03 BOOL  ; A4扫码NG
H111.04 BOOL  ; A5扫码NG
H112 CHANNEL  ; B1取料位扫码OK记忆
H112.00 BOOL  ; B1扫码OK
H112.01 BOOL  ; B2扫码OK
H112.02 BOOL  ; B3扫码OK
H112.03 BOOL  ; B4扫码OK
H112.04 BOOL  ; B5扫码OK
H113 CHANNEL  ; B1取料位扫码NG记忆
H113.00 BOOL  ; B1扫码NG
H113.01 BOOL  ; B2扫码NG
H113.02 BOOL  ; B3扫码NG
H113.03 BOOL  ; B4扫码NG
H113.04 BOOL  ; B5扫码NG
H114.00 BOOL  ; A扫码完成记忆
H114.01 BOOL  ; B扫码完成记忆
H114.02 BOOL  ; A有料记忆
H114.03 BOOL  ; B有料记忆
H114.04 BOOL  ; A1扫码完成记忆
H114.05 BOOL  ; A2扫码完成记忆
H114.06 BOOL  ; B1扫码完成记忆
H114.07 BOOL  ; B2扫码完成记忆
H114.08 BOOL  ; A1抓完记忆
H114.09 BOOL  ; A2抓完记忆
H114.10 BOOL  ; B1抓完记忆
H114.11 BOOL  ; B2抓完记忆
H115 CHANNEL  ; A2取料位扫码OK记忆
H115.00 BOOL  ; A2取料位1扫码OK记忆
H115.01 BOOL  ; A2取料位2扫码OK记忆
H115.02 BOOL  ; A2取料位3扫码OK记忆
H115.03 BOOL  ; A2取料位4扫码OK记忆
H115.04 BOOL  ; A2取料位5扫码OK记忆
H116 CHANNEL  ; A2取料位扫码NG记忆
H116.00 BOOL  ; A2取料位1扫码NG记忆
H116.01 BOOL  ; A2取料位2扫码NG记忆
H116.02 BOOL  ; A2取料位3扫码NG记忆
H116.03 BOOL  ; A2取料位4扫码NG记忆
H116.04 BOOL  ; A2取料位5扫码NG记忆
H117 CHANNEL  ; B2取料位扫码OK记忆
H117.00 BOOL  ; B2取料位1扫码OK记忆
H117.01 BOOL  ; B2取料位2扫码OK记忆
H117.02 BOOL  ; B2取料位3扫码OK记忆
H117.03 BOOL  ; B2取料位4扫码OK记忆
H117.04 BOOL  ; B2取料位5扫码OK记忆
H118 CHANNEL  ; B2取料位扫码NG记忆
H118.00 BOOL  ; B2取料位1扫码NG记忆
H118.01 BOOL  ; B2取料位2扫码NG记忆
H118.02 BOOL  ; B2取料位3扫码NG记忆
H118.03 BOOL  ; B2取料位4扫码NG记忆
H118.04 BOOL  ; B2取料位5扫码NG记忆
H11.00 BOOL  ; 1号夹爪扫码NG记忆
H11.01 BOOL  ; 2号夹爪扫码NG记忆
H11.02 BOOL  ; 3号夹爪扫码NG记忆
H11.03 BOOL  ; 4号夹爪扫码NG记忆
H11.04 BOOL  ; 5号夹爪扫码NG记忆
H12 CHANNEL  ; 上料夹爪扫码OK记忆
H12.00 BOOL  ; 1号夹爪扫码OK记忆
H12.01 BOOL  ; 2号夹爪扫码OK记忆
H12.02 BOOL  ; 3号夹爪扫码OK记忆
H12.03 BOOL  ; 4号夹爪扫码OK记忆
H12.04 BOOL  ; 5号夹爪扫码OK记忆
H13 CHANNEL  ; 上料机器人有料
H13.00 BOOL  ; 夹爪1有料
H13.01 BOOL  ; 夹爪2有料
H13.02 BOOL  ; 夹爪3有料
H13.03 BOOL  ; 夹爪4有料
H13.04 BOOL  ; 夹爪5有料
H150.00 BOOL  ; 进出料横移伺服A回原完成记忆
H150.01 BOOL  ; 进出料伸缩伺服A回原完成记忆
H150.02 BOOL  ; 进出料横移伺服B回原完成记忆
H150.03 BOOL  ; 进出料伸缩伺服B回原完成记忆
H150.04 BOOL  ; 正压伺服A回原完成记忆
H150.05 BOOL  ; 压板平移伺服A回原完成记忆
H150.06 BOOL  ; 侧压A1左伺服回原完成记忆
H150.07 BOOL  ; 侧压A1右伺服回原完成记忆
H150.08 BOOL  ; 侧压A2左伺服回原完成记忆
H150.09 BOOL  ; 侧压A2右伺服回原完成记忆
H150.10 BOOL  ; 侧压A3左伺服回原完成记忆
H150.11 BOOL  ; 侧压A3右伺服回原完成记忆
H150.12 BOOL  ; 侧压A4左伺服回原完成记忆
H150.13 BOOL  ; 侧压A4右伺服回原完成记忆
H150.14 BOOL  ; 正压伺服B回原完成记忆
H150.15 BOOL  ; 压板平移伺服B回原完成记忆
H151.00 BOOL  ; 侧压B1左伺服回原完成记忆
H151.01 BOOL  ; 侧压B1右伺服回原完成记忆
H151.02 BOOL  ; 侧压B2左伺服回原完成记忆
H151.03 BOOL  ; 侧压B2右伺服回原完成记忆
H151.04 BOOL  ; 侧压B3左伺服回原完成记忆
H151.05 BOOL  ; 侧压B3右伺服回原完成记忆
H151.06 BOOL  ; 侧压B4左伺服回原完成记忆
H151.07 BOOL  ; 侧压B4右伺服回原完成记忆
H151.08 BOOL  ; 25#伺服回原完成记忆
H151.09 BOOL  ; 26#伺服回原完成记忆
H151.10 BOOL  ; 27#伺服回原完成记忆
H151.11 BOOL  ; 接料伺服回原完成记忆
H160.00 BOOL  ; 4ST-A 热压料由A侧进入
H160.01 BOOL  ; 4ST-A 热压料由B侧进入
H161.00 BOOL  ; 4ST_A预压计时
H161.01 BOOL  ; 4ST_A正压计时
H162.00 BOOL  ; 4ST_A A1HIP测试完成
H162.01 BOOL  ; 4ST_A A2HIP测试完成
H162.02 BOOL  ; 4ST_A A3HIP测试完成
H162.03 BOOL  ; 4ST_A A4HIP测试完成
H162.04 BOOL  ; 4ST_A A5HIP测试完成
H163.00 BOOL  ; 清料启动
H164 CHANNEL  ; 热压A记忆交换字
H164.00 BOOL  ; 4A记忆已由A侧转移到B侧(待热压料)
H164.01 BOOL  ; 4A记忆已由A侧转移到B侧(2料)
H164.02 BOOL  ; 4A记忆移转到B侧（完成料）
H164.03 BOOL  ; 4A记忆B转A(待热压料)
H164.04 BOOL  ; 4A记忆B转A（2个）
H164.05 BOOL  ; 4A记忆B转A（完成料）
H165 CHANNEL  ; A顶升伸出记忆字
H170.00 BOOL  ; 4ST-B 热压料由A侧进入
H170.01 BOOL  ; 4ST-B 热压料由B侧进入
H171.00 BOOL  ; 4ST_B预压计时
H171.01 BOOL  ; 4ST_B正压计时
H172.00 BOOL  ; 4ST_B B1HIP测试完成
H172.01 BOOL  ; 4ST_B B2HIP测试完成
H172.02 BOOL  ; 4ST_B B3HIP测试完成
H172.03 BOOL  ; 4ST_B B4HIP测试完成
H172.04 BOOL  ; 4ST_B B5HIP测试完成
H173.00 BOOL  ; 清料启动
H174 CHANNEL  ; 热压B记忆转移字
H174.00 BOOL  ; 4B记忆已由A侧转移到B侧(待热压料)
H174.01 BOOL  ; 4B记忆已由A侧转移到B侧(2料)
H174.02 BOOL  ; 4A记忆移转到B侧（完成料）
H174.03 BOOL  ; 4B记忆已由B侧转移到A侧(待热压料)
H174.04 BOOL  ; 4B记忆已由B侧转移到A侧(2料)
H174.05 BOOL  ; 4A记忆移转到A侧（完成料）
H175 CHANNEL  ; B顶升伸出记忆字
H1.00 BOOL  ; 工位步序初始（1启用）
H1.05 BOOL  ; 进出料伺服励磁关闭 1关闭
H200.00 BOOL  ; 切换使用功能块
H20.00 BOOL  ; 上料定位上层有料记忆
H20.01 BOOL  ; 上料定位下层有料记忆
H20.02 BOOL  ; 上料定位A3有料记忆
H20.03 BOOL  ; 上料定位A4有料记忆
H20.04 BOOL  ; 上料定位A5有料记忆
H21.00 BOOL  ; 2St_A进料定位完成记忆
H2.00 BOOL  ; 五层使用 1-使用
H2.01 BOOL  ; 进出料转移分动力
H2.02 BOOL  ; HIP测试气缸 1使用
H2.03 BOOL  ; 扫码伸缩使用
H2.04 BOOL  ; 出料定位升降屏蔽
H2.05 BOOL  ; 下料机器人变距使用
H2.06 BOOL  ; 出料夹爪出料定位变距使用（1=上升）
H2.07 BOOL  ; 空跑模式
H2.08 BOOL  ; 安全门屏蔽
H2.09 BOOL  ; 出料夹爪热压工位变距使用(1=上升)
H2.10 BOOL  ; 蜂鸣器屏蔽
H2.11 BOOL  ; 热压NG光栅屏蔽
H2.12 BOOL  ; 进料夹爪上升下降（0-平台位上升  热压位下降）
H30.00 BOOL  ; 出料定位上层有料记忆
H30.01 BOOL  ; 出料定位下层有料记忆
H30.02 BOOL  ; 上层NG
H30.03 BOOL  ; 下层NG
H30.04 BOOL  ; 上料定位B5有料记忆
H31.00 BOOL  ; 2St_B进料定位完成记忆
H3.00 BOOL  ; 工位1先放B侧
H3.01 BOOL  ; 工位2先放B侧
H3.02 BOOL  ; $?St$Bk?_#[469] / 进料先抓1层/2层(0:先1层） / $?St$Bk?_#[469]
H3.03 BOOL  ; $?St$Bk?_#[470] / 进料先抓A侧/B侧(0:先A侧） / $?St$Bk?_#[470]
H3.04 BOOL  ; $?St$Bk?_#[471] / 扫码前进使用(1:使用) / $?St$Bk?_#[471]
H3.10 BOOL  ; 控压选择（0位置 1转矩）
H3.15 BOOL  ; 位置模式
H40 CHANNEL  ; 3ST_A进料夹爪有料记忆
H40.00 BOOL  ; 进料转移夹爪上层有料记忆
H40.01 BOOL  ; 进料转移夹爪下层有料记忆
H40.02 BOOL  ; 出料转移夹爪上层有料记忆
H40.03 BOOL  ; 出料转移夹爪下层有料记忆
H40.04 BOOL  ; 进料转移夹爪上料中
H40.05 BOOL  ; 出料移转夹爪放料中
H41 CHANNEL  ; 3ST_A出料夹爪有料记忆
H41.00 BOOL  ; 出料转移夹爪A1有料记忆
H41.01 BOOL  ; 出料转移夹爪A2有料记忆
H41.02 BOOL  ; 出料转移夹爪A3有料记忆
H41.03 BOOL  ; 出料转移夹爪A4有料记忆
H41.04 BOOL  ; 出料转移夹爪A5有料记忆
H42.00 BOOL  ; 3ST_A A侧放料标志
H42.01 BOOL  ; 3ST_B A侧放料标志
H42.02 BOOL  ; 3ST_A A侧取料标志
H42.03 BOOL  ; 3ST_B A侧取料标志
H42.04 BOOL  ; 3ST_A除尘电机启动
H48.00 BOOL  ; 热压A1-1有料记忆
H48.01 BOOL  ; 热压A1-2有料记忆
H48.02 BOOL  ; 热压A1-3有料记忆
H48.03 BOOL  ; 热压A1-4有料记忆
H48.04 BOOL  ; 热压A1-5有料记忆
H49.00 BOOL  ; 热压A2-1有料记忆
H49.01 BOOL  ; 热压A2-2有料记忆
H49.02 BOOL  ; 热压A2-3有料记忆
H49.03 BOOL  ; 热压A2-4有料记忆
H49.04 BOOL  ; 热压A2-5有料记忆
H4.00 BOOL  ; 侧压启用 1-启用
H4.01 BOOL  ; 预压启用 1-启用
H4.02 BOOL  ; 侧压最后拨料 1—启用
H4.03 BOOL  ; 关闭待料卸压 1-关闭
H4.04 BOOL  ; 电脑屏蔽 1屏蔽
H4.05 BOOL  ; 扫码屏蔽 1屏蔽
H4.06 BOOL  ; 重复扫码 1屏蔽
H4.07 BOOL  ; MES屏蔽 1屏蔽
H50 CHANNEL  ; 3ST_B进料夹爪有料记忆
H50.00 BOOL  ; 4ST_1热压A上层有料记忆
H50.01 BOOL  ; 4ST_1热压A下层有料记忆
H50.02 BOOL  ; 3ST_B进料夹爪B3有料记忆
H50.03 BOOL  ; 3ST_B进料夹爪B4有料记忆
H50.04 BOOL  ; 3ST_B进料夹爪B5有料记忆
H51 CHANNEL  ; 3ST_B出料夹爪有料记忆
H51.00 BOOL  ; 3ST_B出料夹爪B1有料记忆
H51.01 BOOL  ; 3ST_B出料夹爪B2有料记忆
H51.02 BOOL  ; 3ST_B出料夹爪B3有料记忆
H51.03 BOOL  ; 3ST_B出料夹爪B4有料记忆
H51.04 BOOL  ; 3ST_B出料夹爪B5有料记忆
H52.00 BOOL  ; 3ST_A B侧放料标志
H52.01 BOOL  ; 3ST_B B侧放料标志
H52.02 BOOL  ; 3ST_A B侧取料标志
H52.03 BOOL  ; 3ST_B B侧取料标志
H52.04 BOOL  ; 3ST_B除尘电机启动
H5.00 BOOL  ; A模组屏蔽 1屏蔽
H5.01 BOOL  ; B模组屏蔽 1屏蔽
H5.02 BOOL  ; 模组加热屏蔽 1-屏蔽
H5.03 BOOL  ; B模组加热屏蔽 1屏蔽
H5.04 BOOL  ; 模组C加热屏蔽
H5.05 BOOL  ; 3ST_B屏蔽  1屏蔽
H5.08 BOOL  ; A调试
H5.15 BOOL  ; HIP测试屏蔽
H60 CHANNEL  ; 4ST-A A边有待热压料
H60.00 BOOL  ; 4ST_A A边_1层有待热压
H60.01 BOOL  ; 4ST_A A边_2层有待热压
H60.02 BOOL  ; 4ST_A A边_3层有待热压
H60.03 BOOL  ; 4ST_A A边_4层有待热压
H60.04 BOOL  ; 4ST_A A边_5层有待热压
H61 CHANNEL  ; 4ST-A B边有待热压料
H61.00 BOOL  ; 4ST_A B边_1层有待热压
H61.01 BOOL  ; 4ST_A B边_2层有待热压
H61.02 BOOL  ; 4ST_A B边_3层有待热压
H61.03 BOOL  ; 4ST_A B边_4层有待热压
H61.04 BOOL  ; 4ST_A B边_5层有待热压
H62 CHANNEL  ; 4ST-A 热压位有料
H62.00 BOOL  ; 4ST_A A1热压位有料
H62.01 BOOL  ; 4ST_A A2热压位有料
H62.02 BOOL  ; 4ST_A A3热压位有料
H62.03 BOOL  ; 4ST_A A4热压位有料
H62.04 BOOL  ; 4ST_A A5热压位有料
H63 CHANNEL  ; 4ST-A B边有完成料
H63.00 BOOL  ; 4ST_A A边_1层有热压完成料
H63.01 BOOL  ; 4ST_A A边_2层有热压完成料
H63.02 BOOL  ; 4ST_A A边_3层有热压完成料
H63.03 BOOL  ; 4ST_A A边_4层有热压完成料
H63.04 BOOL  ; 4ST_A A边_5层有热压完成料
H64 CHANNEL  ; 4ST-A A边有完成料
H64.00 BOOL  ; 4ST_A B边_1层有热压完成料
H64.01 BOOL  ; 4ST_A B边_2层有热压完成料
H64.02 BOOL  ; 4ST_A B边_3层有热压完成料
H64.03 BOOL  ; 4ST_A B边_4层有热压完成料
H64.04 BOOL  ; 4ST_A B边_5层有热压完成料
H66.00 BOOL  ; 4ST_A 抵消重力标志
H6.00 BOOL  ; 热压带料复位启用
H6.02 BOOL  ; 抵消重力关闭
H6.10 BOOL  ; 机器人屏蔽
H70 CHANNEL  ; 4ST-B A边有待热压料
H70.00 BOOL  ; 4ST_3 热压C上层有料记忆
H70.01 BOOL  ; 4ST_3 热压C下层有料记忆
H70.02 BOOL  ; 4ST_B A边_3层有待热压
H70.03 BOOL  ; 4ST_B A边_4层有待热压
H70.04 BOOL  ; 4ST_B A边_5层有待热压
H71 CHANNEL  ; 4ST-B B边有待热压料
H71.00 BOOL  ; 4ST_B B边_1层有待热压
H71.01 BOOL  ; 4ST_B B边_2层有待热压
H71.02 BOOL  ; 4ST_B B边_3层有待热压
H71.03 BOOL  ; 4ST_B B边_4层有待热压
H71.04 BOOL  ; 4ST_B B边_5层有待热压
H72 CHANNEL  ; 4ST-B 热压位有料
H72.00 BOOL  ; 4ST_B B1热压位有料
H72.01 BOOL  ; 4ST_B B2热压位有料
H72.02 BOOL  ; 4ST_B B3热压位有料
H72.03 BOOL  ; 4ST_B B4热压位有料
H72.04 BOOL  ; 4ST_B B5热压位有料
H73 CHANNEL  ; 4ST-B B边有完成料
H73.00 BOOL  ; 4ST_B A边_1层有热压完成料
H73.01 BOOL  ; 4ST_B A边_2层有热压完成料
H73.02 BOOL  ; 4ST_B A边_3层有热压完成料
H73.03 BOOL  ; 4ST_B A边_4层有热压完成料
H73.04 BOOL  ; 4ST_B A边_5层有热压完成料
H74 CHANNEL  ; 4ST-B A边有完成料
H74.00 BOOL  ; 4ST_B B边_1层有热压完成料
H74.01 BOOL  ; 4ST_B B边_2层有热压完成料
H74.02 BOOL  ; 4ST_B B边_3层有热压完成料
H74.03 BOOL  ; 4ST_B B边_4层有热压完成料
H74.04 BOOL  ; 4ST_B B边_5层有热压完成料
H76.00 BOOL  ; 4ST_B 重力抵消标志
H80.00 BOOL  ; 下料定位A1有料记忆
H80.01 BOOL  ; 下料定位A2有料记忆
H80.02 BOOL  ; 下料定位A3有料记忆
H80.03 BOOL  ; 下料定位A4有料记忆
H80.04 BOOL  ; 下料定位A5有料记忆
H81.00 BOOL  ; A1有OK电芯
H81.01 BOOL  ; A2有OK电芯
H81.02 BOOL  ; A3有OK电芯
H81.03 BOOL  ; A4有OK电芯
H81.04 BOOL  ; A5有OK电芯
H82.00 BOOL  ; A1有工艺NG电芯
H82.01 BOOL  ; A2有工艺NG电芯
H82.02 BOOL  ; A3有工艺NG电芯
H82.03 BOOL  ; A4有工艺NG电芯
H82.04 BOOL  ; A5有工艺NG电芯
H83.00 BOOL  ; A1有HipotNG电芯
H83.01 BOOL  ; A2有HipotNG电芯
H83.02 BOOL  ; A3有HipotNG电芯
H83.03 BOOL  ; A4有HipotNG电芯
H83.04 BOOL  ; A5有HipotNG电芯
H84.00 BOOL  ; A整定完成信号
H8.02 BOOL  ; 转矩使用
H8.05 BOOL  ; 拨料位运行位置切换
H90.00 BOOL  ; 下料定位B1有料记忆
H90.01 BOOL  ; 下料定位B2有料记忆
H90.02 BOOL  ; 下料定位B3有料记忆
H90.03 BOOL  ; 下料定位B4有料记忆
H90.04 BOOL  ; 下料定位B5有料记忆
H91.00 BOOL  ; B1有OK电芯
H91.01 BOOL  ; B2有OK电芯
H91.02 BOOL  ; B3有OK电芯
H91.03 BOOL  ; B4有OK电芯
H91.04 BOOL  ; B5有OK电芯
H92.00 BOOL  ; B1有工艺NG电芯
H92.01 BOOL  ; B2有工艺NG电芯
H92.02 BOOL  ; B3有工艺NG电芯
H92.03 BOOL  ; B4有工艺NG电芯
H92.04 BOOL  ; B5有工艺NG电芯
H93.00 BOOL  ; B1有HipotNG电芯
H93.01 BOOL  ; B2有HipotNG电芯
H93.02 BOOL  ; B3有HipotNG电芯
H93.03 BOOL  ; B4有HipotNG电芯
H93.04 BOOL  ; B5有HipotNG电芯
H94.00 BOOL  ; B整定完成信号
T0000 BOOL  ; PLC上电延时5S
T0002 BOOL  ; 上位机连接失败
T0010 BOOL  ; 手自动切换延时
T0011 BOOL  ; 自动停止完成延时
T0012 BOOL  ; 清料停止延时
T0014 BOOL  ; 初始化完成延时
T0018 BOOL  ; 延时自动切换
T0050 BOOL  ; 1St上料机器人初始位延时
T0051 BOOL  ; 2St-A初始位延时
T0052 BOOL  ; 2St-B初始位延时
T0053 BOOL  ; 3St-A初始位延时
T0054 BOOL  ; 3St-B初始位延时
T0055 BOOL  ; 4St-A初始位延时
T0056 BOOL  ; 4St-B初始位延时
T0057 BOOL  ; 5St初始位延时
T0058 BOOL  ; 5St初始位延时
T0059 BOOL  ; 6St初始位延时
T0060 BOOL  ; 7St初始位延时
T0100 BOOL  ; 手/自动选择延时
T0101 BOOL  ; 启动按钮延时
T0102 BOOL  ; 停止按钮延时
T0103 BOOL  ; 复位按钮延时
T0104 BOOL  ; 前门磁延时
T0105 BOOL  ; 后门磁延时
T0106 BOOL  ; 左门磁延时
T0107 BOOL  ; 右门磁延时
T0108 BOOL  ; 气源压力开关延时
T0109 BOOL  ; 主急停按钮延时
T0110 BOOL  ; 移动屏急停延时
T0111 BOOL  ; 移动屏使用中延时
T0112 BOOL  ; 备用1延时
T0113 BOOL  ; 备用2延时
T0114 BOOL  ; 备用3延时
T0115 BOOL  ; 备用4延时
T0116 BOOL  ; 启动按钮1延时
T0117 BOOL  ; 启动按钮2延时
T0118 BOOL  ; 进出料安全光栅延时
T0119 BOOL  ; 进料定位上层前后松开位延时
T0120 BOOL  ; 进料定位上层前后夹紧位延时
T0121 BOOL  ; 进料定位下层前后松开位延时
T0122 BOOL  ; 进料定位下层前后夹紧位延时
T0123 BOOL  ; 进料定位上层左右松开位延时
T0124 BOOL  ; 进料定位上层左右夹紧位延时
T0125 BOOL  ; 进料定位下层左右松开位延时
T0126 BOOL  ; 进料定位下层左右夹紧位延时
T0127 BOOL  ; 进料定位平台上层待料位延时
T0128 BOOL  ; 进料定位平台上层出料位延时
T0129 BOOL  ; 进料定位平台下层待料位延时
T0130 BOOL  ; 进料定位平台下层出料位延时
T0131 BOOL  ; 进料定位上层有料感应延时
T0132 BOOL  ; 进料定位下层有料感应延时
T0133 BOOL  ; 出料定位上层前后松开位延时
T0134 BOOL  ; 出料定位上层前后夹紧位延时
T0135 BOOL  ; 出料定位下层前后松开位延时
T0136 BOOL  ; 出料定位下层前后夹紧位延时
T0137 BOOL  ; 出料定位上层左右松开位延时
T0138 BOOL  ; 出料定位上层左右夹紧位延时
T0139 BOOL  ; 出料定位下层左右松开位延时
T0140 BOOL  ; 出料定位下层左右夹紧位延时
T0141 BOOL  ; 出料定位平台上层接料位延时
T0142 BOOL  ; 出料定位平台上层出料位延时
T0143 BOOL  ; 出料定位平台下层接料位延时
T0144 BOOL  ; 出料定位平台下层出料位延时
T0145 BOOL  ; 出料定位上层有料感应延时
T0146 BOOL  ; 出料定位下层有料感应延时
T0147 BOOL  ; 备用5延时
T0148 BOOL  ; 进料夹爪张开位延时
T0149 BOOL  ; 进料夹爪夹紧位延时
T0150 BOOL  ; 进料爪上层左压紧上升位延时
T0151 BOOL  ; 进料爪上层右压紧上升位延时
T0152 BOOL  ; 进料爪下层左压紧上升位延时
T0153 BOOL  ; 进料爪下层右压紧上升位延时
T0154 BOOL  ; 进料爪上层中间压紧上升位延时
T0155 BOOL  ; 进料爪下层中间压紧上升位延时
T0156 BOOL  ; 进料夹爪上升位延时
T0157 BOOL  ; 进料夹爪下降位延时
T0158 BOOL  ; 进料爪上层有料感应延时
T0159 BOOL  ; 进料爪下层有料感应延时
T0160 BOOL  ; 出料夹爪张开位延时
T0161 BOOL  ; 出料夹爪夹紧位延时
T0162 BOOL  ; 出料爪上层左压紧上升位延时
T0163 BOOL  ; 出料爪上层右压紧上升位延时
T0164 BOOL  ; 出料爪下层左压紧上升位延时
T0165 BOOL  ; 出料爪下层右压紧上升位延时
T0166 BOOL  ; 出料夹爪上升位延时
T0167 BOOL  ; 出料夹爪下降位延时
T0168 BOOL  ; 出料爪上层有料感应延时
T0169 BOOL  ; 出料爪下层有料感应延时
T0170 BOOL  ; 备用6延时
T0171 BOOL  ; 备用7延时
T0172 BOOL  ; 热压A增压缸上升位延时
T0173 BOOL  ; 热压A增压缸下降位延时
T0174 BOOL  ; 热压A上层顶升气缸上升位延时
T0175 BOOL  ; 热压A上层顶升气缸下降位延时
T0176 BOOL  ; 热压A下层顶升气缸上升位延时
T0177 BOOL  ; 热压A下层顶升气缸下降位延时
T0178 BOOL  ; 热压A垫高气缸移出位延时
T0179 BOOL  ; 热压A垫高气缸热压位延时
T0180 BOOL  ; 热压A上层Hip测试气缸上升位延时
T0181 BOOL  ; 热压A上层Hip测试气缸下降位延时
T0182 BOOL  ; 热压A下层Hip测试气缸上升位延时
T0183 BOOL  ; 热压A下层Hip测试气缸下降位延时
T0184 BOOL  ; 热压A上层有料感应延时
T0185 BOOL  ; 热压A下层有料感应延时
T0186 BOOL  ; 热压A上层极耳检查输入延时
T0187 BOOL  ; 热压A下层极耳检查输入延时
T0188 BOOL  ; 备用8延时
T0189 BOOL  ; 热压B增压缸上升位延时
T0190 BOOL  ; 热压B增压缸下降位延时
T0191 BOOL  ; 热压B上层顶升气缸上升位延时
T0192 BOOL  ; 热压B上层顶升气缸下降位延时
T0193 BOOL  ; 热压B下层顶升气缸上升位延时
T0194 BOOL  ; 热压B下层顶升气缸下降位延时
T0195 BOOL  ; 热压B垫高气缸移出位延时
T0196 BOOL  ; 热压B垫高气缸热压位延时
T0197 BOOL  ; 热压B上层Hip测试气缸上升位延时
T0198 BOOL  ; 热压B上层Hip测试气缸下降位延时
T0199 BOOL  ; 热压B下层Hip测试气缸上升位延时
T0200 BOOL  ; 热压B下层Hip测试气缸下降位延时
T0201 BOOL  ; 热压B上层有料感应延时
T0202 BOOL  ; 热压B下层有料感应延时
T0203 BOOL  ; 热压B上层极耳检查输入延时
T0204 BOOL  ; 热压B下层极耳检查输入延时
T0205 BOOL  ; 备用9延时
T0206 BOOL  ; 热压C增压缸上升位延时
T0207 BOOL  ; 热压C增压缸下降位延时
T0208 BOOL  ; 热压C上层顶升气缸上升位延时
T0209 BOOL  ; 热压C上层顶升气缸下降位延时
T0210 BOOL  ; 热压C下层顶升气缸上升位延时
T0211 BOOL  ; 热压C下层顶升气缸下降位延时
T0212 BOOL  ; 热压C垫高气缸移出位延时
T0213 BOOL  ; 热压C垫高气缸热压位延时
T0214 BOOL  ; 热压C上层Hip测试气缸上升位延时
T0215 BOOL  ; 热压C上层Hip测试气缸下降位延时
T0216 BOOL  ; 热压C下层Hip测试气缸上升位延时
T0217 BOOL  ; 热压C下层Hip测试气缸下降位延时
T0218 BOOL  ; 热压C上层有料感应延时
T0219 BOOL  ; 热压C下层有料感应延时
T0220 BOOL  ; 热压C上层极耳检查输入延时
T0221 BOOL  ; 热压C下层极耳检查输入延时
T0222 BOOL  ; 备用10延时
T0223 BOOL  ; 进出料转移伺服准备好延时
T0224 BOOL  ; 进出料转移伺服报警延时
T0225 BOOL  ; 伸缩伺服准备好延时
T0226 BOOL  ; 伸缩伺服报警延时
T0227 BOOL  ; 备用11延时
T0228 BOOL  ; 加热A跳闸延时
T0229 BOOL  ; 加热B跳闸延时
T0230 BOOL  ; 加热C跳闸延时
T0231 BOOL  ; 副PLC 0.03延时
T0232 BOOL  ; 副PLC 0.04延时
T0233 BOOL  ; 副PLC 0.05延时
T0234 BOOL  ; 副PLC 0.06延时
T0235 BOOL  ; 副PLC 0.07延时
T0236 BOOL  ; 副PLC 0.08延时
T0237 BOOL  ; 副PLC 0.09延时
T0238 BOOL  ; 副PLC 0.10延时
T0239 BOOL  ; 副PLC 0.11延时
T0240 BOOL  ; 延时
T0241 BOOL  ; 延时
T0242 BOOL  ; 延时
T0243 BOOL  ; 延时
T0244 BOOL  ; 副PLC 1.00延时
T0245 BOOL  ; 副PLC 1.01延时
T0246 BOOL  ; 副PLC 1.02延时
T0247 BOOL  ; 副PLC 1.03延时
T0248 BOOL  ; 副PLC 1.04延时
T0249 BOOL  ; 副PLC 1.05延时
T0250 BOOL  ; 副PLC 1.06延时
T0251 BOOL  ; 副PLC 1.07延时
T0252 BOOL  ; 副PLC 1.08延时
T0253 BOOL  ; 副PLC 1.09延时
T0254 BOOL  ; 副PLC 1.10延时
T0255 BOOL  ; 副PLC 1.11延时
T0256 BOOL  ; 延时
T0257 BOOL  ; 延时
T0258 BOOL  ; 延时
T0259 BOOL  ; 延时
T0260 BOOL  ; 延时
T0450 BOOL  ; $?St$Bk?_#[472] / 热压模组A压力清零延时1秒 / $?St$Bk?_#[472]
T0815 BOOL  ; 双手启动0.5秒内响应延时
T0816 BOOL  ; 进料定位有料状态正常
T1000 BOOL  ; 进出料横移伺服在平台进出料位
T1001 BOOL  ; 进出料横移伺服在热压A放料位
T1002 BOOL  ; 进出料横移伺服在热压A取料位
T1003 BOOL  ; 进出料横移伺服在热压B放料位
T1004 BOOL  ; 进出料横移伺服在热压B取料位
T1005 BOOL  ; 进出料横移伺服在热压C放料位
T1006 BOOL  ; 进出料横移伺服在热压C取料位
T1007 BOOL  ; 进出料横移伺服在出料位
T1008 BOOL  ; 进出料横移伺服在位置9
T1009 BOOL  ; 进出料横移伺服在位置10
T1010 BOOL  ; 进出料伸缩伺服在初始位
T1011 BOOL  ; 进出料伸缩伺服在平台取料位
T1012 BOOL  ; 进出料伸缩伺服在热压取放位
T1013 BOOL  ; 进出料伸缩伺服在位置4
T1014 BOOL  ; 进出料伸缩伺服在位置5
T1015 BOOL  ; 进出料伸缩伺服在位置6
T1016 BOOL  ; 进出料伸缩伺服在位置7
T1017 BOOL  ; 进出料伸缩伺服在位置8
T1018 BOOL  ; 进出料伸缩伺服在位置9
T1019 BOOL  ; 进出料伸缩伺服在位置10
T1040 BOOL  ; 正压伺服A在初始位
T1041 BOOL  ; 正压伺服A在减速位
T1042 BOOL  ; 正压伺服A在等距热压位
T1043 BOOL  ; 正压伺服A在预压退回位
T1044 BOOL  ; 正压伺服A在MASK测试位
T1045 BOOL  ; 正压伺服A在位置6
T1046 BOOL  ; 正压伺服A在位置7
T1047 BOOL  ; 正压伺服A在位置8
T1048 BOOL  ; 正压伺服A在位置9
T1049 BOOL  ; 正压伺服A在位置10
T1050 BOOL  ; 压板平移伺服A在A面取放位
T1051 BOOL  ; 压板平移伺服A在B面取放位
T1052 BOOL  ; 压板平移伺服A在位置3
T1053 BOOL  ; 压板平移伺服A在位置4
T1054 BOOL  ; 压板平移伺服A在位置5
T1055 BOOL  ; 压板平移伺服A在位置6
T1056 BOOL  ; 压板平移伺服A在位置7
T1057 BOOL  ; 压板平移伺服A在位置8
T1058 BOOL  ; 压板平移伺服A在位置9
T1059 BOOL  ; 压板平移伺服A在位置10
T1060 BOOL  ; A1左伺服在待机位
T1061 BOOL  ; A1左伺服在拨料退回位
T1062 BOOL  ; A1左伺服在拨料位
T1063 BOOL  ; A1左伺服在减速位
T1064 BOOL  ; A1左伺服在等距热压位
T1065 BOOL  ; A1左伺服在位置6
T1066 BOOL  ; A1左伺服在位置7
T1067 BOOL  ; A1左伺服在位置8
T1068 BOOL  ; A1左伺服在位置9
T1069 BOOL  ; A1左伺服在位置10
T1070 BOOL  ; A1右伺服在待机位
T1071 BOOL  ; A1右伺服在拨料退回位
T1072 BOOL  ; A1右伺服在拨料位
T1073 BOOL  ; A1右伺服在减速位
T1074 BOOL  ; A1右伺服在等距热压位
T1075 BOOL  ; A1右伺服在位置6
T1076 BOOL  ; A1右伺服在位置7
T1077 BOOL  ; A1右伺服在位置8
T1078 BOOL  ; A1右伺服在位置9
T1079 BOOL  ; A1右伺服在位置10
T1080 BOOL  ; A2左伺服在待机位
T1081 BOOL  ; A2左伺服在拨料退回位
T1082 BOOL  ; A2左伺服在拨料位
T1083 BOOL  ; A2左伺服在减速位
T1084 BOOL  ; A2左伺服在等距热压位
T1090 BOOL  ; A2右伺服在待机位
T1091 BOOL  ; A2右伺服在拨料退回位
T1092 BOOL  ; A2右伺服在拨料位
T1093 BOOL  ; A2右伺服在减速位
T1094 BOOL  ; A2右伺服在等距热压位
T1095 BOOL  ; A2右伺服在位置6
T1096 BOOL  ; A2右伺服在位置7
T1097 BOOL  ; A2右伺服在位置8
T1098 BOOL  ; A2右伺服在位置9
T1099 BOOL  ; A2右伺服在位置10
T1100 BOOL  ; A3左伺服在待机位
T1101 BOOL  ; A3左伺服在拨料退回位
T1102 BOOL  ; A3左伺服在拨料位
T1103 BOOL  ; A3左伺服在减速位
T1104 BOOL  ; A3左伺服在等距热压位
T1110 BOOL  ; A3右伺服在待机位
T1111 BOOL  ; A3右伺服在拨料退回位
T1112 BOOL  ; A3右伺服在拨料位
T1113 BOOL  ; A3右伺服在减速位
T1114 BOOL  ; A3右伺服在等距热压位
T1120 BOOL  ; A4左伺服在待机位
T1121 BOOL  ; A4左伺服在拨料退回位
T1122 BOOL  ; A4左伺服在拨料位
T1123 BOOL  ; A4左伺服在减速位
T1124 BOOL  ; A4左伺服在等距热压位
T1125 BOOL  ; A4左伺服在位置6
T1130 BOOL  ; A4右伺服在待机位
T1131 BOOL  ; A4右伺服在拨料退回位
T1132 BOOL  ; A4右伺服在拨料位
T1133 BOOL  ; A4右伺服在减速位
T1134 BOOL  ; A4右伺服在等距热压位
T1135 BOOL  ; A4右伺服在位置6
T1136 BOOL  ; A4右伺服在位置7
T1137 BOOL  ; A4右伺服在位置8
T1138 BOOL  ; A4右伺服在位置9
T1139 BOOL  ; A4右伺服在位置10
T1140 BOOL  ; 正压伺服B在初始位
T1141 BOOL  ; 正压伺服B在减速位
T1142 BOOL  ; 正压伺服B在等距热压位
T1143 BOOL  ; 正压伺服B在预压退回位
T1144 BOOL  ; 正压伺服B在MASK测试位
T1145 BOOL  ; 正压伺服B在位置6
T1146 BOOL  ; 正压伺服B在位置7
T1147 BOOL  ; 正压伺服B在位置8
T1148 BOOL  ; 正压伺服B在位置9
T1149 BOOL  ; 正压伺服B在位置10
T1150 BOOL  ; 压板平移伺服B在A面取放位
T1151 BOOL  ; 压板平移伺服B在B面取放位
T1152 BOOL  ; 压板平移伺服B在位置3
T1153 BOOL  ; 压板平移伺服B在位置4
T1154 BOOL  ; 压板平移伺服B在位置5
T1155 BOOL  ; 压板平移伺服B在位置6
T1156 BOOL  ; 压板平移伺服B在位置7
T1157 BOOL  ; 压板平移伺服B在位置8
T1158 BOOL  ; 压板平移伺服B在位置9
T1159 BOOL  ; 压板平移伺服B在位置10
T1160 BOOL  ; B1左伺服在待机位
T1161 BOOL  ; B1左伺服在拨料退回位
T1162 BOOL  ; B1左伺服在拨料位
T1163 BOOL  ; B1左伺服在减速位
T1164 BOOL  ; B1左伺服在等距热压位
T1165 BOOL  ; B1左伺服在位置6
T1166 BOOL  ; B1左伺服在位置7
T1167 BOOL  ; B1左伺服在位置8
T1168 BOOL  ; B1左伺服在位置9
T1169 BOOL  ; B1左伺服在位置10
T1170 BOOL  ; B1右伺服在待机位
T1171 BOOL  ; B1右伺服在拨料退回位
T1172 BOOL  ; B1右伺服在拨料位
T1173 BOOL  ; B1右伺服在减速位
T1174 BOOL  ; B1右伺服在等距热压位
T1175 BOOL  ; B1右伺服在位置6
T1176 BOOL  ; B1右伺服在位置7
T1177 BOOL  ; B1右伺服在位置8
T1178 BOOL  ; B1右伺服在位置9
T1179 BOOL  ; B1右伺服在位置10
T1180 BOOL  ; B2左伺服在待机位
T1181 BOOL  ; B2左伺服在拨料退回位
T1182 BOOL  ; B2左伺服在拨料位
T1183 BOOL  ; B2左伺服在减速位
T1184 BOOL  ; B2左伺服在等距热压位
T1185 BOOL  ; B2左伺服在位置6
T1186 BOOL  ; B2左伺服在位置7
T1187 BOOL  ; B2左伺服在位置8
T1188 BOOL  ; B2左伺服在位置9
T1189 BOOL  ; B2左伺服在位置10
T1190 BOOL  ; B2右伺服在待机位
T1191 BOOL  ; B2右伺服在拨料退回位
T1192 BOOL  ; B2右伺服在拨料位
T1193 BOOL  ; B2右伺服在减速位
T1194 BOOL  ; B2右伺服在等距热压位
T1195 BOOL  ; B2右伺服在位置6
T1196 BOOL  ; B2右伺服在位置7
T1197 BOOL  ; B2右伺服在位置8
T1198 BOOL  ; B2右伺服在位置9
T1199 BOOL  ; B2右伺服在位置10
T1200 BOOL  ; B3左伺服在待机位
T1201 BOOL  ; B3左伺服在拨料退回位
T1202 BOOL  ; B3左伺服在拨料位
T1203 BOOL  ; B3左伺服在减速位
T1204 BOOL  ; B3左伺服在等距热压位
T1205 BOOL  ; B3左伺服在位置6
T1206 BOOL  ; B3左伺服在位置7
T1207 BOOL  ; B3左伺服在位置8
T1208 BOOL  ; B3左伺服在位置9
T1209 BOOL  ; B3左伺服在位置10
T1210 BOOL  ; B3右伺服在待机位
T1211 BOOL  ; B3右伺服在拨料退回位
T1212 BOOL  ; B3右伺服在拨料位
T1213 BOOL  ; B3右伺服在减速位
T1214 BOOL  ; B3右伺服在等距热压位
T1215 BOOL  ; B3右伺服在位置6
T1216 BOOL  ; B3右伺服在位置7
T1217 BOOL  ; B3右伺服在位置8
T1218 BOOL  ; B3右伺服在位置9
T1219 BOOL  ; B3右伺服在位置10
T1220 BOOL  ; B4左伺服在待机位
T1221 BOOL  ; B4左伺服在拨料退回位
T1222 BOOL  ; B4左伺服在拨料位
T1223 BOOL  ; B4左伺服在减速位
T1224 BOOL  ; B4左伺服在等距热压位
T1225 BOOL  ; B4左伺服在位置6
T1226 BOOL  ; B4左伺服在位置7
T1227 BOOL  ; B4左伺服在位置8
T1228 BOOL  ; B4左伺服在位置9
T1229 BOOL  ; B4左伺服在位置10
T1230 BOOL  ; B4右伺服在待机位
T1231 BOOL  ; B4右伺服在拨料退回位
T1232 BOOL  ; B4右伺服在拨料位
T1233 BOOL  ; B4右伺服在减速位
T1234 BOOL  ; B4右伺服在等距热压位
T1235 BOOL  ; B4右伺服在位置6
T1236 BOOL  ; B4右伺服在位置7
T1237 BOOL  ; B4右伺服在位置8
T1238 BOOL  ; B4右伺服在位置9
T1239 BOOL  ; B4右伺服在位置10
T1240 BOOL  ; 出料伸缩伺服A在初始位
T1241 BOOL  ; 出料伸缩伺服A在热压取料位
T1242 BOOL  ; 出料伸缩伺服A在出料平台放料位
T1243 BOOL  ; 出料伸缩伺服A在位置4
T1244 BOOL  ; 出料伸缩伺服A在位置5
T1245 BOOL  ; 出料伸缩伺服A在位置6
T1246 BOOL  ; 出料伸缩伺服A在位置7
T1247 BOOL  ; 出料伸缩伺服A在位置8
T1248 BOOL  ; 出料伸缩伺服A在位置9
T1249 BOOL  ; 出料伸缩伺服A在位置10
T1250 BOOL  ; 26#伺服在位置1
T1251 BOOL  ; 26#伺服在位置2
T1252 BOOL  ; 26#伺服在位置3
T1253 BOOL  ; 26#伺服在位置4
T1254 BOOL  ; 26#伺服在位置5
T1255 BOOL  ; 26#伺服在位置6
T1256 BOOL  ; 26#伺服在位置7
T1257 BOOL  ; 26#伺服在位置8
T1258 BOOL  ; 26#伺服在位置9
T1259 BOOL  ; 26#伺服在位置10
T1260 BOOL  ; 27#左伺服在位置1
T1261 BOOL  ; 27#左伺服在位置2
T1262 BOOL  ; 27#左伺服在位置3
T1263 BOOL  ; 27#左伺服在位置4
T1264 BOOL  ; 27#左伺服在位置5
T1265 BOOL  ; 27#左伺服在位置6
T1266 BOOL  ; 27#左伺服在位置7
T1267 BOOL  ; 27#左伺服在位置8
T1268 BOOL  ; 27#左伺服在位置9
T1269 BOOL  ; 27#左伺服在位置10
T1270 BOOL  ; 接料伺服在出料位
T1271 BOOL  ; 接料伺服在接料位
T1272 BOOL  ; 接料伺服在位置3
T1273 BOOL  ; 接料伺服在位置4
T1274 BOOL  ; 接料伺服在位置5
T1275 BOOL  ; 接料伺服在位置6
T1276 BOOL  ; 接料伺服在位置7
T1277 BOOL  ; 接料伺服在位置8
T1278 BOOL  ; 接料伺服在位置9
T1279 BOOL  ; 接料伺服在位置10
T1500 BOOL  ; 进出料横移伺服A进料位启动延时
T1501 BOOL  ; 进出料横移伺服A进料等待位启动延时
T1502 BOOL  ; 进出料横移伺服A上料位A启动延时
T1503 BOOL  ; 进出料横移伺服A上料位B启动延时
T1504 BOOL  ; 进出料横移伺服A下料位A启动延时
T1505 BOOL  ; 进出料横移伺服A下料位B启动延时
T1506 BOOL  ; 进出料横移伺服A出料等待位启动延时
T1507 BOOL  ; 进出料横移伺服A出料位启动延时
T1508 BOOL  ; 进出料横移伺服A位置9启动延时
T1509 BOOL  ; 进出料横移伺服A位置10启动延时
T1510 BOOL  ; 进出料伸缩伺服A初始位启动延时
T1511 BOOL  ; 进出料伸缩伺服A平台取料位启动延时
T1512 BOOL  ; 进出料伸缩伺服A热压取放位启动延时
T1513 BOOL  ; 进出料伸缩伺服热压位取放料料条件
T1514 BOOL  ; 进出料伸缩伺服A位置5启动延时
T1515 BOOL  ; 进出料伸缩伺服A位置6启动延时
T1516 BOOL  ; 进出料伸缩伺服A位置7启动延时
T1517 BOOL  ; 进出料伸缩伺服A位置8启动延时
T1518 BOOL  ; 进出料伸缩伺服A位置9启动延时
T1519 BOOL  ; 进出料伸缩伺服A位置10启动延时
T1520 BOOL  ; 进出料横移伺服B进料位启动延时
T1521 BOOL  ; 进出料横移伺服B进料等待位启动延时
T1522 BOOL  ; 进出料横移伺服B上料位A启动延时
T1523 BOOL  ; 进出料横移伺服B上料位B启动延时
T1524 BOOL  ; 进出料横移伺服B下料位A启动延时
T1525 BOOL  ; 进出料横移伺服B下料位B启动延时
T1526 BOOL  ; 进出料横移伺服B出料等待位启动延时
T1527 BOOL  ; 进出料横移伺服B出料位启动延时
T1528 BOOL  ; 进出料横移伺服B位置9启动延时
T1529 BOOL  ; 进出料横移伺服B位置10启动延时
T1530 BOOL  ; 进出料伸缩伺服B初始位启动延时
T1531 BOOL  ; 进出料伸缩伺服B平台取料位启动延时
T1532 BOOL  ; 进出料伸缩伺服B热压取放位启动延时
T1533 BOOL  ; 进出料伸缩伺服B平台放料位启动延时
T1534 BOOL  ; 进出料伸缩伺服B位置5启动延时
T1535 BOOL  ; 进出料伸缩伺服B位置6启动延时
T1536 BOOL  ; 进出料伸缩伺服B位置7启动延时
T1537 BOOL  ; 进出料伸缩伺服B位置8启动延时
T1538 BOOL  ; 进出料伸缩伺服B位置9启动延时
T1539 BOOL  ; 进出料伸缩伺服B位置10启动延时
T1540 BOOL  ; 正压伺服A初始位启动延时
T1541 BOOL  ; 正压伺服A减速位启动延时
T1542 BOOL  ; 正压伺服A等距热压位启动延时
T1543 BOOL  ; 正压伺服A预压退回位启动延时
T1544 BOOL  ; 正压伺服AMASK测试位启动延时
T1545 BOOL  ; 正压伺服A位置6启动延时
T1546 BOOL  ; 正压伺服A位置7启动延时
T1547 BOOL  ; 正压伺服A位置8启动延时
T1548 BOOL  ; 正压伺服A位置9启动延时
T1549 BOOL  ; 正压伺服A位置10启动延时
T1550 BOOL  ; 压板平移伺服AA面取放位启动延时
T1551 BOOL  ; 压板平移伺服AB面取放位启动延时
T1552 BOOL  ; 压板平移伺服A位置3启动延时
T1553 BOOL  ; 压板平移伺服A位置4启动延时
T1554 BOOL  ; 压板平移伺服A位置5启动延时
T1555 BOOL  ; 压板平移伺服A位置6启动延时
T1556 BOOL  ; 压板平移伺服A位置7启动延时
T1557 BOOL  ; 压板平移伺服A位置8启动延时
T1558 BOOL  ; 压板平移伺服A位置9启动延时
T1559 BOOL  ; 压板平移伺服A位置10启动延时
T1560 BOOL  ; A1左伺服待机位启动延时
T1561 BOOL  ; A1左伺服拨料退回位启动延时
T1562 BOOL  ; A1左伺服拨料位启动延时
T1563 BOOL  ; A1左伺服减速位启动延时
T1564 BOOL  ; A1左伺服等距热压位启动延时
T1565 BOOL  ; A1左伺服位置6启动延时
T1566 BOOL  ; A1左伺服位置7启动延时
T1567 BOOL  ; A1左伺服位置8启动延时
T1568 BOOL  ; A1左伺服位置9启动延时
T1569 BOOL  ; A1左伺服位置10启动延时
T1570 BOOL  ; A1右伺服待机位启动延时
T1571 BOOL  ; A1右伺服拨料退回位启动延时
T1572 BOOL  ; A1右伺服拨料位启动延时
T1573 BOOL  ; A1右伺服减速位启动延时
T1574 BOOL  ; A1右伺服等距热压位启动延时
T1575 BOOL  ; A1右伺服位置6启动延时
T1576 BOOL  ; A1右伺服位置7启动延时
T1577 BOOL  ; A1右伺服位置8启动延时
T1578 BOOL  ; A1右伺服位置9启动延时
T1579 BOOL  ; A1右伺服位置10启动延时
T1580 BOOL  ; A2左伺服待机位启动延时
T1581 BOOL  ; A2左伺服拨料退回位启动延时
T1582 BOOL  ; A2左伺服拨料位启动延时
T1583 BOOL  ; A2左伺服减速位启动延时
T1584 BOOL  ; A2左伺服等距热压位启动延时
T1585 BOOL  ; A2左伺服位置6启动延时
T1586 BOOL  ; A2左伺服位置7启动延时
T1587 BOOL  ; A2左伺服位置8启动延时
T1588 BOOL  ; A2左伺服位置9启动延时
T1589 BOOL  ; A2左伺服位置10启动延时
T1590 BOOL  ; A2右伺服待机位启动延时
T1591 BOOL  ; A2右伺服拨料退回位启动延时
T1592 BOOL  ; A2右伺服拨料位启动延时
T1593 BOOL  ; A2右伺服减速位启动延时
T1594 BOOL  ; A2右伺服等距热压位启动延时
T1595 BOOL  ; A2右伺服位置6启动延时
T1596 BOOL  ; A2右伺服位置7启动延时
T1597 BOOL  ; A2右伺服位置8启动延时
T1598 BOOL  ; A2右伺服位置9启动延时
T1599 BOOL  ; A2右伺服位置10启动延时
T1600 BOOL  ; A3左伺服待机位启动延时
T1601 BOOL  ; A3左伺服拨料退回位启动延时
T1602 BOOL  ; A3左伺服拨料位启动延时
T1603 BOOL  ; A3左伺服减速位启动延时
T1604 BOOL  ; A3左伺服等距热压位启动延时
T1605 BOOL  ; A3左伺服位置6启动延时
T1606 BOOL  ; A3左伺服位置7启动延时
T1607 BOOL  ; A3左伺服位置8启动延时
T1608 BOOL  ; A3左伺服位置9启动延时
T1609 BOOL  ; A3左伺服位置10启动延时
T1610 BOOL  ; A3右伺服待机位启动延时
T1611 BOOL  ; A3右伺服拨料退回位启动延时
T1612 BOOL  ; A3右伺服拨料位启动延时
T1613 BOOL  ; A3右伺服减速位启动延时
T1614 BOOL  ; A3右伺服等距热压位启动延时
T1615 BOOL  ; A3右伺服位置6启动延时
T1616 BOOL  ; A3右伺服位置7启动延时
T1617 BOOL  ; A3右伺服位置8启动延时
T1618 BOOL  ; A3右伺服位置9启动延时
T1619 BOOL  ; A3右伺服位置10启动延时
T1620 BOOL  ; A4左伺服待机位启动延时
T1621 BOOL  ; A4左伺服拨料退回位启动延时
T1622 BOOL  ; A4左伺服拨料位启动延时
T1623 BOOL  ; A4左伺服减速位启动延时
T1624 BOOL  ; A4左伺服等距热压位启动延时
T1625 BOOL  ; A4左伺服位置6启动延时
T1626 BOOL  ; A4左伺服位置7启动延时
T1627 BOOL  ; A4左伺服位置8启动延时
T1628 BOOL  ; A4左伺服位置9启动延时
T1629 BOOL  ; A4左伺服位置10启动延时
T1630 BOOL  ; A4右伺服待机位启动延时
T1631 BOOL  ; A4右伺服拨料退回位启动延时
T1632 BOOL  ; A4右伺服拨料位启动延时
T1633 BOOL  ; A4右伺服减速位启动延时
T1634 BOOL  ; A4右伺服等距热压位启动延时
T1635 BOOL  ; A4右伺服位置6启动延时
T1636 BOOL  ; A4右伺服位置7启动延时
T1637 BOOL  ; A4右伺服位置8启动延时
T1638 BOOL  ; A4右伺服位置9启动延时
T1639 BOOL  ; A4右伺服位置10启动延时
T1640 BOOL  ; 正压伺服B初始位启动延时
T1641 BOOL  ; 正压伺服B减速位启动延时
T1642 BOOL  ; 正压伺服B等距热压位启动延时
T1643 BOOL  ; 正压伺服B预压退回位启动延时
T1644 BOOL  ; 正压伺服BMASK测试位启动延时
T1645 BOOL  ; 正压伺服B位置6启动延时
T1646 BOOL  ; 正压伺服B位置7启动延时
T1647 BOOL  ; 正压伺服B位置8启动延时
T1648 BOOL  ; 正压伺服B位置9启动延时
T1649 BOOL  ; 正压伺服B位置10启动延时
T1650 BOOL  ; 压板平移伺服BA面取放位启动延时
T1651 BOOL  ; 压板平移伺服BB面取放位启动延时
T1652 BOOL  ; 压板平移伺服B位置3启动延时
T1653 BOOL  ; 压板平移伺服B位置4启动延时
T1654 BOOL  ; 压板平移伺服B位置5启动延时
T1655 BOOL  ; 压板平移伺服B位置6启动延时
T1656 BOOL  ; 压板平移伺服B位置7启动延时
T1657 BOOL  ; 压板平移伺服B位置8启动延时
T1658 BOOL  ; 压板平移伺服B位置9启动延时
T1659 BOOL  ; 压板平移伺服B位置10启动延时
T1660 BOOL  ; B1左伺服待机位启动延时
T1661 BOOL  ; B1左伺服拨料退回位启动延时
T1662 BOOL  ; B1左伺服拨料位启动延时
T1663 BOOL  ; B1左伺服减速位启动延时
T1664 BOOL  ; B1左伺服等距热压位启动延时
T1665 BOOL  ; B1左伺服位置6启动延时
T1666 BOOL  ; B1左伺服位置7启动延时
T1667 BOOL  ; B1左伺服位置8启动延时
T1668 BOOL  ; B1左伺服位置9启动延时
T1669 BOOL  ; B1左伺服位置10启动延时
T1670 BOOL  ; B1右伺服待机位启动延时
T1671 BOOL  ; B1右伺服拨料退回位启动延时
T1672 BOOL  ; B1右伺服拨料位启动延时
T1673 BOOL  ; B1右伺服减速位启动延时
T1674 BOOL  ; B1右伺服等距热压位启动延时
T1675 BOOL  ; B1右伺服位置6启动延时
T1676 BOOL  ; B1右伺服位置7启动延时
T1677 BOOL  ; B1右伺服位置8启动延时
T1678 BOOL  ; B1右伺服位置9启动延时
T1679 BOOL  ; B1右伺服位置10启动延时
T1680 BOOL  ; B2左伺服待机位启动延时
T1681 BOOL  ; B2左伺服拨料退回位启动延时
T1682 BOOL  ; B2左伺服拨料位启动延时
T1683 BOOL  ; B2左伺服减速位启动延时
T1684 BOOL  ; B2左伺服等距热压位启动延时
T1685 BOOL  ; B2左伺服位置6启动延时
T1686 BOOL  ; B2左伺服位置7启动延时
T1687 BOOL  ; B2左伺服位置8启动延时
T1688 BOOL  ; B2左伺服位置9启动延时
T1689 BOOL  ; B2左伺服位置10启动延时
T1690 BOOL  ; B2右伺服待机位启动延时
T1691 BOOL  ; B2右伺服拨料退回位启动延时
T1692 BOOL  ; B2右伺服拨料位启动延时
T1693 BOOL  ; B2右伺服减速位启动延时
T1694 BOOL  ; B2右伺服等距热压位启动延时
T1695 BOOL  ; B2右伺服位置6启动延时
T1696 BOOL  ; B2右伺服位置7启动延时
T1697 BOOL  ; B2右伺服位置8启动延时
T1698 BOOL  ; B2右伺服位置9启动延时
T1699 BOOL  ; B2右伺服位置10启动延时
T1700 BOOL  ; B3左伺服待机位启动延时
T1701 BOOL  ; B3左伺服拨料退回位启动延时
T1702 BOOL  ; B3左伺服拨料位启动延时
T1703 BOOL  ; B3左伺服减速位启动延时
T1704 BOOL  ; B3左伺服等距热压位启动延时
T1705 BOOL  ; B3左伺服位置6启动延时
T1706 BOOL  ; B3左伺服位置7启动延时
T1707 BOOL  ; B3左伺服位置8启动延时
T1708 BOOL  ; B3左伺服位置9启动延时
T1709 BOOL  ; B3左伺服位置10启动延时
T1710 BOOL  ; B3右伺服待机位启动延时
T1711 BOOL  ; B3右伺服拨料退回位启动延时
T1712 BOOL  ; B3右伺服拨料位启动延时
T1713 BOOL  ; B3右伺服减速位启动延时
T1714 BOOL  ; B3右伺服等距热压位启动延时
T1715 BOOL  ; B3右伺服位置6启动延时
T1716 BOOL  ; B3右伺服位置7启动延时
T1717 BOOL  ; B3右伺服位置8启动延时
T1718 BOOL  ; B3右伺服位置9启动延时
T1719 BOOL  ; B3右伺服位置10启动延时
T1720 BOOL  ; B4左伺服待机位启动延时
T1721 BOOL  ; B4左伺服拨料退回位启动延时
T1722 BOOL  ; B4左伺服拨料位启动延时
T1723 BOOL  ; B4左伺服减速位启动延时
T1724 BOOL  ; B4左伺服等距热压位启动延时
T1725 BOOL  ; B4左伺服位置6启动延时
T1726 BOOL  ; B4左伺服位置7启动延时
T1727 BOOL  ; B4左伺服位置8启动延时
T1728 BOOL  ; B4左伺服位置9启动延时
T1729 BOOL  ; B4左伺服位置10启动延时
T1730 BOOL  ; B4右伺服待机位启动延时
T1731 BOOL  ; B4右伺服拨料退回位启动延时
T1732 BOOL  ; B4右伺服拨料位启动延时
T1733 BOOL  ; B4右伺服减速位启动延时
T1734 BOOL  ; B4右伺服等距热压位启动延时
T1735 BOOL  ; B4右伺服位置6启动延时
T1736 BOOL  ; B4右伺服位置7启动延时
T1737 BOOL  ; B4右伺服位置8启动延时
T1738 BOOL  ; B4右伺服位置9启动延时
T1739 BOOL  ; B4右伺服位置10启动延时
T1740 BOOL  ; 出料伸缩伺服A初始位启动延时
T1741 BOOL  ; 出料伸缩伺服A热压取料位启动延时
T1742 BOOL  ; 出料伸缩伺服A出料平台放料位启动延时
T1743 BOOL  ; 出料伸缩伺服A位置4启动延时
T1744 BOOL  ; 出料伸缩伺服A位置5启动延时
T1745 BOOL  ; 出料伸缩伺服A位置6启动延时
T1746 BOOL  ; 出料伸缩伺服A位置7启动延时
T1747 BOOL  ; 出料伸缩伺服A位置8启动延时
T1748 BOOL  ; 出料伸缩伺服A位置9启动延时
T1749 BOOL  ; 出料伸缩伺服A位置10启动延时
T1750 BOOL  ; 26#伺服位置1启动延时
T1751 BOOL  ; 26#伺服位置2启动延时
T1752 BOOL  ; 26#伺服位置3启动延时
T1753 BOOL  ; 26#伺服位置4启动延时
T1754 BOOL  ; 26#伺服位置5启动延时
T1755 BOOL  ; 26#伺服位置6启动延时
T1756 BOOL  ; 26#伺服位置7启动延时
T1757 BOOL  ; 26#伺服位置8启动延时
T1758 BOOL  ; 26#伺服位置9启动延时
T1759 BOOL  ; 26#伺服位置10启动延时
T1760 BOOL  ; 27#左伺服位置1启动延时
T1761 BOOL  ; 27#左伺服位置2启动延时
T1762 BOOL  ; 27#左伺服位置3启动延时
T1763 BOOL  ; 27#左伺服位置4启动延时
T1764 BOOL  ; 27#左伺服位置5启动延时
T1765 BOOL  ; 27#左伺服位置6启动延时
T1766 BOOL  ; 27#左伺服位置7启动延时
T1767 BOOL  ; 27#左伺服位置8启动延时
T1768 BOOL  ; 27#左伺服位置9启动延时
T1769 BOOL  ; 27#左伺服位置10启动延时
T1770 BOOL  ; 接料伺服出料位启动延时
T1771 BOOL  ; 接料伺服接料位启动延时
T1772 BOOL  ; 接料伺服位置3启动延时
T1773 BOOL  ; 接料伺服位置4启动延时
T1774 BOOL  ; 接料伺服位置5启动延时
T1775 BOOL  ; 接料伺服位置6启动延时
T1776 BOOL  ; 接料伺服位置7启动延时
T1777 BOOL  ; 接料伺服位置8启动延时
T1778 BOOL  ; 接料伺服位置9启动延时
T1779 BOOL  ; 接料伺服位置10启动延时
T1810 BOOL  ; ST5520_A1 手动通讯测试触发延时判断结果
T1812 BOOL  ; ST5520_A1 手动通讯测试触发OK延时关闭
T1813 BOOL  ; ST5520_A 测试电压读取延时
T1814 BOOL  ; 延时RSET 读取
T1815 BOOL  ; ST5520_通讯全测试延时
T1816 BOOL  ; 1秒间隔触发下一个端口
T1817 BOOL  ; 通讯延时1S断开
T1818 BOOL  ; 测试通讯延时断开
T1820 BOOL  ; ST5520_A1 档位延时写入
T1821 BOOL  ; ST5520_A1 速度延时写入
T1822 BOOL  ; ST5520_A1 模式延时写入
T1823 BOOL  ; 全写延时
T1824 BOOL  ; 全写入延时
T1825 BOOL  ; 参数全写入延时
T1826 BOOL  ; 延时1S
T1827 BOOL  ; 延时1S断开
T1828 BOOL  ; 参数全写入延时断开
T1830 BOOL  ; 热压A1工位Hipot检测延时触发信号
T1831 BOOL  ; 热压A1不使用延时完成
T1832 BOOL  ; 热压A2工位Hipot检测延时触发信号
T1833 BOOL  ; 热压A2不使用延时完成
T1834 BOOL  ; 热压A3工位Hipot检测延时触发信号
T1835 BOOL  ; 热压A3不使用延时完成
T1836 BOOL  ; 热压A4工位Hipot检测延时触发信号
T1837 BOOL  ; 热压A4不使用延时完成
T1838 BOOL  ; 热压A5工位Hipot检测延时触发信号
T1839 BOOL  ; 热压A5不使用延时完成
T1840 BOOL  ; 热压B1工位Hipot检测延时触发信号
T1841 BOOL  ; 热压B1不使用延时完成
T1842 BOOL  ; 热压B2工位Hipot检测延时触发信号
T1843 BOOL  ; 热压B2不使用延时完成
T1844 BOOL  ; 热压B3工位Hipot检测延时触发信号
T1845 BOOL  ; 热压B3不使用延时完成
T1846 BOOL  ; 热压B4工位Hipot检测延时触发信号
T1847 BOOL  ; 热压B4不使用延时完成
T1848 BOOL  ; 热压B5工位Hipot检测延时触发信号
T1849 BOOL  ; 热压B5不使用延时完成
T2000 BOOL  ; 1ST进料机器人R1左夹紧气缸1松开位异常延时
T2001 BOOL  ; 1ST进料机器人R1左夹紧气缸1夹紧位异常延时
T2002 BOOL  ; 1ST进料机器人R1右夹紧气缸1松开位异常延时
T2003 BOOL  ; 1ST进料机器人R1右夹紧气缸1夹紧位异常延时
T2004 BOOL  ; 1ST进料机器人R1左夹紧气缸2松开位异常延时
T2005 BOOL  ; 1ST进料机器人R1左夹紧气缸2夹紧位异常延时
T2006 BOOL  ; 1ST进料机器人R1右夹紧气缸2松开位异常延时
T2007 BOOL  ; 1ST进料机器人R1右夹紧气缸2夹紧位异常延时
T2008 BOOL  ; 1ST进料机器人R1左夹紧气缸3松开位异常延时
T2009 BOOL  ; 1ST进料机器人R1左夹紧气缸3夹紧位异常延时
T2010 BOOL  ; 1ST进料机器人R1右夹紧气缸3松开位异常延时
T2011 BOOL  ; 1ST进料机器人R1右夹紧气缸3夹紧位异常延时
T2012 BOOL  ; 1ST进料机器人R1左夹紧气缸4松开位异常延时
T2013 BOOL  ; 1ST进料机器人R1左夹紧气缸4夹紧位异常延时
T2014 BOOL  ; 1ST进料机器人R1右夹紧气缸4松开位异常延时
T2015 BOOL  ; 1ST进料机器人R1右夹紧气缸4夹紧位异常延时
T2016 BOOL  ; 1ST进料机器人R1左夹紧气缸5松开位异常延时
T2017 BOOL  ; 1ST进料机器人R1左夹紧气缸5夹紧位异常延时
T2018 BOOL  ; 1ST进料机器人R1右夹紧气缸5松开位异常延时
T2019 BOOL  ; 1ST进料机器人R1右夹紧气缸5夹紧位异常延时
T2020 BOOL  ; 1ST进料机器人R1左压紧1上升位异常延时
T2021 BOOL  ; 1ST进料机器人R1右压紧1上升位异常延时
T2022 BOOL  ; 1ST进料机器人R1左压紧2上升位异常延时
T2023 BOOL  ; 1ST进料机器人R1右压紧2上升位异常延时
T2024 BOOL  ; 1ST进料机器人R1左压紧3上升位异常延时
T2025 BOOL  ; 1ST进料机器人R1右压紧3上升位异常延时
T2026 BOOL  ; 1ST进料机器人R1左压紧4上升位异常延时
T2027 BOOL  ; 1ST进料机器人R1右压紧4上升位异常延时
T2028 BOOL  ; 1ST进料机器人R1左压紧5上升位异常延时
T2029 BOOL  ; 1ST进料机器人R1右压紧5上升位异常延时
T2030 BOOL  ; 1ST进料机器人R1有料反射光电感应1异常延时
T2031 BOOL  ; 1ST进料机器人R1有料反射光电感应2异常延时
T2032 BOOL  ; 1ST进料机器人R1有料反射光电感应3异常延时
T2033 BOOL  ; 1ST进料机器人R1有料反射光电感应4异常延时
T2034 BOOL  ; 1ST进料机器人R1有料反射光电感应5异常延时
T2050 BOOL  ; 1ST进料定位上层前后松开位异常延时
T2051 BOOL  ; 1ST进料定位上层前后夹紧位异常延时
T2052 BOOL  ; 1ST进料定位下层前后松开位异常延时
T2053 BOOL  ; 1ST进料定位下层前后夹紧位异常延时
T2054 BOOL  ; 1ST进料定位上层左右松开位异常延时
T2055 BOOL  ; 1ST进料定位上层左右夹紧位异常延时
T2056 BOOL  ; 1ST进料定位下层左右松开位异常延时
T2057 BOOL  ; 1ST进料定位下层左右夹紧位异常延时
T2058 BOOL  ; 1ST进料定位平台上层待料位异常延时
T2059 BOOL  ; 1ST进料定位平台上层出料位异常延时
T2060 BOOL  ; 1ST进料定位平台下层待料位异常延时
T2061 BOOL  ; 1ST进料定位平台下层出料位异常延时
T2062 BOOL  ; 1ST进料定位上层有料感应异常延时
T2063 BOOL  ; 1ST进料定位下层有料感应异常延时
T2100 BOOL  ; 2ST出料定位上层前后松开位异常延时
T2101 BOOL  ; 2ST出料定位上层前后夹紧位异常延时
T2102 BOOL  ; 2ST出料定位下层前后松开位异常延时
T2103 BOOL  ; 2ST出料定位下层前后夹紧位异常延时
T2104 BOOL  ; 2ST出料定位上层左右松开位异常延时
T2105 BOOL  ; 2ST出料定位上层左右夹紧位异常延时
T2106 BOOL  ; 2ST出料定位下层左右松开位异常延时
T2107 BOOL  ; 2ST出料定位下层左右夹紧位异常延时
T2108 BOOL  ; 2ST出料定位平台上层接料位异常延时
T2109 BOOL  ; 2ST出料定位平台上层出料位异常延时
T2110 BOOL  ; 2ST出料定位平台下层接料位异常延时
T2111 BOOL  ; 2ST出料定位平台下层出料位异常延时
T2112 BOOL  ; 2ST出料定位上层有料感应异常延时
T2113 BOOL  ; 2ST出料定位下层有料感应异常延时
T2150 BOOL  ; 3ST进料夹爪张开位异常延时
T2151 BOOL  ; 3ST进料夹爪夹紧位异常延时
T2152 BOOL  ; 3ST进料爪上层左压紧上升位异常延时
T2153 BOOL  ; 3ST进料爪上层右压紧上升位异常延时
T2154 BOOL  ; 3ST进料爪下层左压紧上升位异常延时
T2155 BOOL  ; 3ST进料爪下层右压紧上升位异常延时
T2156 BOOL  ; 3ST进料爪上层中间压紧上升位异常延时
T2157 BOOL  ; 3ST进料爪下层中间压紧上升位异常延时
T2158 BOOL  ; 3ST进料夹爪上升位异常延时
T2159 BOOL  ; 3ST进料夹爪下降位异常延时
T2160 BOOL  ; 3ST进料爪上层有料感应异常延时
T2161 BOOL  ; 3ST进料爪下层有料感应异常延时
T2162 BOOL  ; 3ST出料夹爪张开位异常延时
T2163 BOOL  ; 3ST出料夹爪夹紧位异常延时
T2164 BOOL  ; 3ST出料爪上层左压紧上升位异常延时
T2165 BOOL  ; 3ST出料爪上层右压紧上升位异常延时
T2166 BOOL  ; 3ST出料爪下层左压紧上升位异常延时
T2167 BOOL  ; 3ST出料爪下层右压紧上升位异常延时
T2168 BOOL  ; 3ST出料夹爪上升位异常延时
T2169 BOOL  ; 3ST出料夹爪下降位异常延时
T2170 BOOL  ; 3ST出料爪上层有料感应异常延时
T2171 BOOL  ; 3ST出料爪下层有料感应异常延时
T2200 BOOL  ; 4ST-1热压A增压缸上升位异常延时
T2201 BOOL  ; 4ST-1热压A增压缸下降位异常延时
T2202 BOOL  ; 4ST-1热压A上层顶升气缸上升位异常延时
T2203 BOOL  ; 4ST-1热压A上层顶升气缸下降位异常延时
T2204 BOOL  ; 4ST-1热压A下层顶升气缸上升位异常延时
T2205 BOOL  ; 4ST-1热压A下层顶升气缸下降位异常延时
T2206 BOOL  ; 4ST-1热压A垫高气缸移出位异常延时
T2207 BOOL  ; 4ST-1热压A垫高气缸热压位异常延时
T2208 BOOL  ; 4ST-1热压A上层Hip测试气缸上升位异常延时
T2209 BOOL  ; 4ST-1热压A上层Hip测试气缸下降位异常延时
T2210 BOOL  ; 4ST-1热压A下层Hip测试气缸上升位异常延时
T2211 BOOL  ; 4ST-1热压A下层Hip测试气缸下降位异常延时
T2212 BOOL  ; 4ST-1热压A上层有料感应异常延时
T2213 BOOL  ; 4ST-1热压A下层有料感应异常延时
T2214 BOOL  ; 4ST-1热压A上层极耳检查异常延时
T2215 BOOL  ; 4ST-1热压A下层极耳检查异常延时
T2216 BOOL  ; 4ST-1热压A加热跳闸延时
T2250 BOOL  ; 4ST-2 热压B增压缸上升位异常延时
T2251 BOOL  ; 4ST-2 热压B增压缸下降位异常延时
T2252 BOOL  ; 4ST-2 热压B上层顶升气缸上升位异常延时
T2253 BOOL  ; 4ST-2 热压B上层顶升气缸下降位异常延时
T2254 BOOL  ; 4ST-2 热压B下层顶升气缸上升位异常延时
T2255 BOOL  ; 4ST-2 热压B下层顶升气缸下降位异常延时
T2256 BOOL  ; 4ST-2 热压B垫高气缸移出位异常延时
T2257 BOOL  ; 4ST-2 热压B垫高气缸热压位异常延时
T2258 BOOL  ; 4ST-2 热压B上层Hip测试气缸上升位异常延时
T2259 BOOL  ; 4ST-2 热压B上层Hip测试气缸下降位异常延时
T2260 BOOL  ; 4ST-2 热压B下层Hip测试气缸上升位异常延时
T2261 BOOL  ; 4ST-2 热压B下层Hip测试气缸下降位异常延时
T2262 BOOL  ; 4ST-2 热压B上层有料感应异常延时
T2263 BOOL  ; 4ST-2 热压B下层有料感应异常延时
T2264 BOOL  ; 4ST-2 热压B上层极耳检查输入异常延时
T2265 BOOL  ; 4ST-2 热压B下层极耳检查输入异常延时
T2266 BOOL  ; 4ST-2 热压B加热跳闸延时
T2300 BOOL  ; 4ST-3热压C增压缸上升位异常延时
T2301 BOOL  ; 4ST-3热压C增压缸下降位异常延时
T2302 BOOL  ; 4ST-3热压C上层顶升气缸上升位异常延时
T2303 BOOL  ; 4ST-3热压C上层顶升气缸下降位异常延时
T2304 BOOL  ; 4ST-3热压C下层顶升气缸上升位异常延时
T2305 BOOL  ; 4ST-3热压C下层顶升气缸下降位异常延时
T2306 BOOL  ; 4ST-3热压C垫高气缸移出位异常延时
T2307 BOOL  ; 4ST-3热压C垫高气缸热压位异常延时
T2308 BOOL  ; 4ST-3热压C上层Hip测试气缸上升位异常延时
T2309 BOOL  ; 4ST-3热压C上层Hip测试气缸下降位异常延时
T2310 BOOL  ; 4ST-3热压C下层Hip测试气缸上升位异常延时
T2311 BOOL  ; 4ST-3热压C下层Hip测试气缸下降位异常延时
T2312 BOOL  ; 4ST-3热压C上层有料感应异常延时
T2313 BOOL  ; 4ST-3热压C下层有料感应异常延时
T2314 BOOL  ; 4ST-3热压C上层极耳检查输入异常延时
T2315 BOOL  ; 4ST-3热压C下层极耳检查输入异常延时
T2316 BOOL  ; 4ST-3热压C加热跳闸延时
T2350 BOOL  ; 5ST-A下料定位A下料定位A下降位异常延时
T2351 BOOL  ; 5ST-A下料定位A下料定位A上升位异常延时
T2352 BOOL  ; 5ST-A下料定位A下料定位A水平位异常延时
T2353 BOOL  ; 5ST-A下料定位A下料定位A垂直位异常延时
T2354 BOOL  ; 5ST-A下料定位A下料定位A1左右松开位异常延时
T2355 BOOL  ; 5ST-A下料定位A下料定位A1左右夹紧位异常延时
T2356 BOOL  ; 5ST-A下料定位A下料定位A2左右松开位异常延时
T2357 BOOL  ; 5ST-A下料定位A下料定位A2左右夹紧位异常延时
T2358 BOOL  ; 5ST-A下料定位A下料定位A3左右松开位异常延时
T2359 BOOL  ; 5ST-A下料定位A下料定位A3左右夹紧位异常延时
T2360 BOOL  ; 5ST-A下料定位A下料定位A4左右松开位异常延时
T2361 BOOL  ; 5ST-A下料定位A下料定位A4左右夹紧位异常延时
T2362 BOOL  ; 5ST-A下料定位A下料定位A5左右松开位异常延时
T2363 BOOL  ; 5ST-A下料定位A下料定位A5左右夹紧位异常延时
T2364 BOOL  ; 5ST-A下料定位A下料定位A1前后松开位异常延时
T2365 BOOL  ; 5ST-A下料定位A下料定位A1前后夹紧位异常延时
T2366 BOOL  ; 5ST-A下料定位A下料定位A2前后松开位异常延时
T2367 BOOL  ; 5ST-A下料定位A下料定位A2前后夹紧位异常延时
T2368 BOOL  ; 5ST-A下料定位A下料定位A3前后松开位异常延时
T2369 BOOL  ; 5ST-A下料定位A下料定位A3前后夹紧位异常延时
T2370 BOOL  ; 5ST-A下料定位A下料定位A4前后松开位异常延时
T2371 BOOL  ; 5ST-A下料定位A下料定位A4前后夹紧位异常延时
T2372 BOOL  ; 5ST-A下料定位A下料定位A5前后松开位异常延时
T2373 BOOL  ; 5ST-A下料定位A下料定位A5前后夹紧位异常延时
T2374 BOOL  ; 5ST-A下料定位A下料定位A1有料感应异常延时
T2375 BOOL  ; 5ST-A下料定位A下料定位A2有料感应异常延时
T2376 BOOL  ; 5ST-A下料定位A下料定位A3有料感应异常延时
T2377 BOOL  ; 5ST-A下料定位A下料定位A4有料感应异常延时
T2378 BOOL  ; 5ST-A下料定位A下料定位A5有料感应异常延时
T2379 BOOL  ; 5ST-A下料定位A下料定位A料平整检测（预留）异常延时
T2400 BOOL  ; 5ST-B下料定位B下料定位B下降位异常延时
T2401 BOOL  ; 5ST-B下料定位B下料定位B上升位异常延时
T2402 BOOL  ; 5ST-B下料定位B下料定位B水平位异常延时
T2403 BOOL  ; 5ST-B下料定位B下料定位B垂直位异常延时
T2404 BOOL  ; 5ST-B下料定位B下料定位B1左右松开位异常延时
T2405 BOOL  ; 5ST-B下料定位B下料定位B1左右夹紧位异常延时
T2406 BOOL  ; 5ST-B下料定位B下料定位B2左右松开位异常延时
T2407 BOOL  ; 5ST-B下料定位B下料定位B2左右夹紧位异常延时
T2408 BOOL  ; 5ST-B下料定位B下料定位B3左右松开位异常延时
T2409 BOOL  ; 5ST-B下料定位B下料定位B3左右夹紧位异常延时
T2410 BOOL  ; 5ST-B下料定位B下料定位B4左右松开位异常延时
T2411 BOOL  ; 5ST-B下料定位B下料定位B4左右夹紧位异常延时
T2412 BOOL  ; 5ST-B下料定位B下料定位B5左右松开位异常延时
T2413 BOOL  ; 5ST-B下料定位B下料定位B5左右夹紧位异常延时
T2414 BOOL  ; 5ST-B下料定位B下料定位B1前后松开位异常延时
T2415 BOOL  ; 5ST-B下料定位B下料定位B1前后夹紧位异常延时
T2416 BOOL  ; 5ST-B下料定位B下料定位B2前后松开位异常延时
T2417 BOOL  ; 5ST-B下料定位B下料定位B2前后夹紧位异常延时
T2418 BOOL  ; 5ST-B下料定位B下料定位B3前后松开位异常延时
T2419 BOOL  ; 5ST-B下料定位B下料定位B3前后夹紧位异常延时
T2420 BOOL  ; 5ST-B下料定位B下料定位B4前后松开位异常延时
T2421 BOOL  ; 5ST-B下料定位B下料定位B4前后夹紧位异常延时
T2422 BOOL  ; 5ST-B下料定位B下料定位B5前后松开位异常延时
T2423 BOOL  ; 5ST-B下料定位B下料定位B5前后夹紧位异常延时
T2424 BOOL  ; 5ST-B下料定位B下料定位B1有料感应异常延时
T2425 BOOL  ; 5ST-B下料定位B下料定位B2有料感应异常延时
T2426 BOOL  ; 5ST-B下料定位B下料定位B3有料感应异常延时
T2427 BOOL  ; 5ST-B下料定位B下料定位B4有料感应异常延时
T2428 BOOL  ; 5ST-B下料定位B下料定位B5有料感应异常延时
T2429 BOOL  ; 5ST-B下料定位B下料定位B料平整检测（预留）异常延时
T2450 BOOL  ; 6ST下料机器人R2左夹紧气缸1松开位异常延时
T2451 BOOL  ; 6ST下料机器人R2左夹紧气缸1夹紧位异常延时
T2452 BOOL  ; 6ST下料机器人R2右夹紧气缸1松开位异常延时
T2453 BOOL  ; 6ST下料机器人R2右夹紧气缸1夹紧位异常延时
T2454 BOOL  ; 6ST下料机器人R2左夹紧气缸2松开位异常延时
T2455 BOOL  ; 6ST下料机器人R2左夹紧气缸2夹紧位异常延时
T2456 BOOL  ; 6ST下料机器人R2右夹紧气缸2松开位异常延时
T2457 BOOL  ; 6ST下料机器人R2右夹紧气缸2夹紧位异常延时
T2458 BOOL  ; 6ST下料机器人R2左夹紧气缸3松开位异常延时
T2459 BOOL  ; 6ST下料机器人R2左夹紧气缸3夹紧位异常延时
T2460 BOOL  ; 6ST下料机器人R2右夹紧气缸3松开位异常延时
T2461 BOOL  ; 6ST下料机器人R2右夹紧气缸3夹紧位异常延时
T2462 BOOL  ; 6ST下料机器人R2左夹紧气缸4松开位异常延时
T2463 BOOL  ; 6ST下料机器人R2左夹紧气缸4夹紧位异常延时
T2464 BOOL  ; 6ST下料机器人R2右夹紧气缸4松开位异常延时
T2465 BOOL  ; 6ST下料机器人R2右夹紧气缸4夹紧位异常延时
T2466 BOOL  ; 6ST下料机器人R2左夹紧气缸5松开位异常延时
T2467 BOOL  ; 6ST下料机器人R2左夹紧气缸5夹紧位异常延时
T2468 BOOL  ; 6ST下料机器人R2右夹紧气缸5松开位异常延时
T2469 BOOL  ; 6ST下料机器人R2右夹紧气缸5夹紧位异常延时
T2470 BOOL  ; 6ST下料机器人R2左压紧1上升位异常延时
T2471 BOOL  ; 6ST下料机器人R2右压紧1上升位异常延时
T2472 BOOL  ; 6ST下料机器人R2左压紧2上升位异常延时
T2473 BOOL  ; 6ST下料机器人R2右压紧2上升位异常延时
T2474 BOOL  ; 6ST下料机器人R2左压紧3上升位异常延时
T2475 BOOL  ; 6ST下料机器人R2右压紧3上升位异常延时
T2476 BOOL  ; 6ST下料机器人R2左压紧4上升位异常延时
T2477 BOOL  ; 6ST下料机器人R2右压紧4上升位异常延时
T2478 BOOL  ; 6ST下料机器人R2左压紧5上升位异常延时
T2479 BOOL  ; 6ST下料机器人R2右压紧5上升位异常延时
T2480 BOOL  ; 6ST下料机器人R2有料反射光电感应1异常延时
T2481 BOOL  ; 6ST下料机器人R2有料反射光电感应2异常延时
T2482 BOOL  ; 6ST下料机器人R2有料反射光电感应3异常延时
T2483 BOOL  ; 6ST下料机器人R2有料反射光电感应4异常延时
T2484 BOOL  ; 6ST下料机器人R2有料反射光电感应5异常延时
T2485 BOOL  ; 变距气缸异常
T2500 BOOL  ; $?St$Bk?_#[473] / 上层扫码后退感应异常延时 / $?St$Bk?_#[473]
T2501 BOOL  ; $?St$Bk?_#[474] / 上层扫码前进感应异常延时 / $?St$Bk?_#[474]
T2502 BOOL  ; $?St$Bk?_#[475] / 上层扫码缩回感应异常延时 / $?St$Bk?_#[475]
T2503 BOOL  ; $?St$Bk?_#[476] / 上层扫码伸出感应异常延时 / $?St$Bk?_#[476]
T2504 BOOL  ; $?St$Bk?_#[477] / 下层扫码后退感应异常延时 / $?St$Bk?_#[477]
T2505 BOOL  ; $?St$Bk?_#[478] / 下层扫码前进感应异常延时 / $?St$Bk?_#[478]
T2506 BOOL  ; $?St$Bk?_#[479] / 下层扫码缩回感应异常延时 / $?St$Bk?_#[479]
T2507 BOOL  ; $?St$Bk?_#[480] / 下层扫码伸出感应异常延时 / $?St$Bk?_#[480]
T2600 BOOL  ; 侧压A1左低压快速调整延时
T2601 BOOL  ; 侧压A1左接近慢速调整延时
T2602 BOOL  ; 侧压A1左超压慢速调回延时
T2603 BOOL  ; 侧压A1右低压快速调整延时
T2604 BOOL  ; 侧压A1右接近慢速调整延时
T2605 BOOL  ; 侧压A1右超压慢速调回延时
T2610 BOOL  ; 侧压A2左低压快速调整延时
T2611 BOOL  ; 侧压A2左接近慢速调整延时
T2612 BOOL  ; 侧压A2左超压慢速调回延时
T2613 BOOL  ; 侧压A2右低压快速调整延时
T2614 BOOL  ; 侧压A2右接近慢速调整延时
T2615 BOOL  ; 侧压A2右超压慢速调回延时
T2620 BOOL  ; 侧压A3左低压快速调整延时
T2621 BOOL  ; 侧压A3左接近慢速调整延时
T2622 BOOL  ; 侧压A3左超压慢速调回延时
T2623 BOOL  ; 侧压A3右低压快速调整延时
T2624 BOOL  ; 侧压A3右接近慢速调整延时
T2625 BOOL  ; 侧压A3右超压慢速调回延时
T2630 BOOL  ; 侧压A4左低压快速调整延时
T2631 BOOL  ; 侧压A4左接近慢速调整延时
T2632 BOOL  ; 侧压A4左超压慢速调回延时
T2633 BOOL  ; 侧压A4右低压快速调整延时
T2634 BOOL  ; 侧压A4右接近慢速调整延时
T2635 BOOL  ; 侧压A4右超压慢速调回延时
T2640 BOOL  ; 侧压A5左低压快速调整延时
T2641 BOOL  ; 侧压A5左接近慢速调整延时
T2642 BOOL  ; 侧压A5左超压慢速调回延时
T2643 BOOL  ; 侧压A5右低压快速调整延时
T2644 BOOL  ; 侧压A5右接近慢速调整延时
T2645 BOOL  ; 侧压A5右超压慢速调回延时
T2650 BOOL  ; 侧压B1左低压快速调整延时
T2651 BOOL  ; 侧压B1左接近慢速调整延时
T2652 BOOL  ; 侧压B1左超压慢速调回延时
T2653 BOOL  ; 侧压B1右低压快速调整延时
T2654 BOOL  ; 侧压B1右接近慢速调整延时
T2655 BOOL  ; 侧压B1右超压慢速调回延时
T2657 BOOL  ; 正压B原点回归完成延时
T2658 BOOL  ; 侧压B原位完成延时
T2659 BOOL  ; B压板移位伺服复位完成延时
T2660 BOOL  ; 侧压B2左低压快速调整延时
T2661 BOOL  ; 侧压B2左接近慢速调整延时
T2662 BOOL  ; 侧压B2左超压慢速调回延时
T2663 BOOL  ; 侧压B2右低压快速调整延时
T2664 BOOL  ; 侧压B2右接近慢速调整延时
T2665 BOOL  ; 侧压B2右超压慢速调回延时
T2670 BOOL  ; 侧压B3左低压快速调整延时
T2671 BOOL  ; 侧压B3左接近慢速调整延时
T2672 BOOL  ; 侧压B3左超压慢速调回延时
T2673 BOOL  ; 侧压B3右低压快速调整延时
T2674 BOOL  ; 侧压B3右接近慢速调整延时
T2675 BOOL  ; 侧压B3右超压慢速调回延时
T2680 BOOL  ; 侧压B4左低压快速调整延时
T2681 BOOL  ; 侧压B4左接近慢速调整延时
T2682 BOOL  ; 侧压B4左超压慢速调回延时
T2683 BOOL  ; 侧压B4右低压快速调整延时
T2684 BOOL  ; 侧压B4右接近慢速调整延时
T2685 BOOL  ; 侧压B4右超压慢速调回延时
T2690 BOOL  ; 侧压B5左低压快速调整延时
T2691 BOOL  ; 侧压B5左接近慢速调整延时
T2692 BOOL  ; 侧压B5左超压慢速调回延时
T2693 BOOL  ; 侧压B5右低压快速调整延时
T2694 BOOL  ; 侧压B5右接近慢速调整延时
T2695 BOOL  ; 侧压B5右超压慢速调回延时
T2700 BOOL  ; 1#副PLC离线超时报警
T2701 BOOL  ; 2#副PLC离线超时报警
T2702 BOOL  ; 3#副PLC离线超时报警
W0.01 BOOL  ; 状态指示
W0.02 BOOL  ; 错误指示
W100.00 BOOL  ; 进料定位上层前后松开手动
W100.01 BOOL  ; 进料定位上层前后夹紧手动
W100.02 BOOL  ; 进料定位下层前后松开手动
W100.03 BOOL  ; 进料定位下层前后夹紧手动
W100.04 BOOL  ; 进料定位上层左右松开手动
W100.05 BOOL  ; 进料定位上层左右夹紧手动
W100.06 BOOL  ; 进料定位下层左右松开手动
W100.07 BOOL  ; 进料定位下层左右夹紧手动
W100.08 BOOL  ; 进料定位上层平台待料手动
W100.09 BOOL  ; 进料定位上层平台出料手动
W100.10 BOOL  ; 进料定位下层平台待料手动
W100.11 BOOL  ; 进料定位下层平台出料手动
W103.00 BOOL  ; 出料定位上层前后松开手动
W103.01 BOOL  ; 出料定位上层前后夹紧手动
W103.02 BOOL  ; 出料定位下层前后松开手动
W103.03 BOOL  ; 出料定位下层前后夹紧手动
W103.04 BOOL  ; 出料定位上层左右松开手动
W103.05 BOOL  ; 出料定位上层左右夹紧手动
W103.06 BOOL  ; 出料定位下层左右松开手动
W103.07 BOOL  ; 出料定位下层左右夹紧手动
W103.08 BOOL  ; 出料定位上层平台接料手动
W103.09 BOOL  ; 出料定位上层平台出料手动
W103.10 BOOL  ; 出料定位下层平台接料手动
W103.11 BOOL  ; 出料定位下层平台出料手动
W103.12 BOOL  ; 上下层吹气手动
W106.00 BOOL  ; 进料夹爪张开手动
W106.01 BOOL  ; 进料夹爪夹紧手动
W106.02 BOOL  ; 进料爪上下层左右压紧上升手动
W106.03 BOOL  ; 进料爪上下层左右压紧下降手动
W106.04 BOOL  ; 进料爪上下层中间压紧上升手动
W106.05 BOOL  ; 进料爪上下层中间压紧下降手动
W106.06 BOOL  ; 进料夹爪上升手动
W106.07 BOOL  ; 进料夹爪下降手动
W107.00 BOOL  ; 出料夹爪张开手动
W107.01 BOOL  ; 出料夹爪夹紧手动
W107.02 BOOL  ; 出料爪上下层左右压紧上升手动
W107.03 BOOL  ; 出料爪上下层左右压紧下降手动
W107.04 BOOL  ; 出料夹爪上升手动
W107.05 BOOL  ; 出料夹爪下降手动
W10.03 BOOL  ; 应放A平台
W11 CHANNEL  ; 上料机器人任务信息
W110.00 BOOL  ; 热压A增压缸上升手动
W110.01 BOOL  ; 热压A增压缸下降手动
W110.02 BOOL  ; 热压A上层顶升气缸上升手动
W110.03 BOOL  ; 热压A上层顶升气缸下降手动
W110.04 BOOL  ; 热压A下层顶升气缸上升手动
W110.05 BOOL  ; 热压A下层顶升气缸下降手动
W110.06 BOOL  ; 热压A垫高气缸移出手动
W110.07 BOOL  ; 热压A垫高气缸热压手动
W110.08 BOOL  ; 热压AHip测试气缸上升手动
W110.09 BOOL  ; 热压AHip测试气缸下降手动
W110.10 BOOL  ; 热压A上下层吹气手动
W110.11 BOOL  ; 热压A上层HIP测试选择手动
W110.12 BOOL  ; 热压A下层HIP测试选择手动
W110.13 BOOL  ; 热压A极耳测试手动
W110.14 BOOL  ; 热压A压力清零手动
W113.00 BOOL  ; 热压B增压缸上升手动
W113.01 BOOL  ; 热压B增压缸下降手动
W113.02 BOOL  ; 热压B上层顶升气缸上升手动
W113.03 BOOL  ; 热压B上层顶升气缸下降手动
W113.04 BOOL  ; 热压B下层顶升气缸上升手动
W113.05 BOOL  ; 热压B下层顶升气缸下降手动
W113.06 BOOL  ; 热压B垫高气缸移出手动
W113.07 BOOL  ; 热压B垫高气缸热压手动
W113.08 BOOL  ; 热压BHip测试气缸上升手动
W113.09 BOOL  ; 热压BHip测试气缸下降手动
W113.10 BOOL  ; 热压B上下层吹气手动
W113.11 BOOL  ; 热压B上层HIP测试选择手动
W113.12 BOOL  ; 热压B下层HIP测试选择手动
W113.13 BOOL  ; 热压B极耳测试手动
W113.14 BOOL  ; 热压B压力清零手动
W116.00 BOOL  ; 热压C增压缸上升手动
W116.01 BOOL  ; 热压C增压缸下降手动
W116.02 BOOL  ; 热压C上层顶升气缸上升手动
W116.03 BOOL  ; 热压C上层顶升气缸下降手动
W116.04 BOOL  ; 热压C下层顶升气缸上升手动
W116.05 BOOL  ; 热压C下层顶升气缸下降手动
W116.06 BOOL  ; 热压C垫高气缸移出手动
W116.07 BOOL  ; 热压C垫高气缸热压手动
W116.08 BOOL  ; 热压CHip测试气缸上升手动
W116.09 BOOL  ; 热压CHip测试气缸下降手动
W116.10 BOOL  ; 热压C上下层吹气手动
W116.11 BOOL  ; 热压C上层HIP测试选择手动
W116.12 BOOL  ; 热压C下层HIP测试选择手动
W116.13 BOOL  ; 热压C极耳测试手动
W116.14 BOOL  ; 热压C压力清零手动
W12 CHANNEL  ; 上料机器人位置信息
W138.00 BOOL  ; 下料定位A下降手动
W138.01 BOOL  ; 下料定位A上升手动
W138.02 BOOL  ; 下料定位A0度翻转手动
W138.03 BOOL  ; 下料定位A90度翻转手动
W138.04 BOOL  ; 下料定位A1前后左右松开手动
W138.05 BOOL  ; 下料定位A1前后左右夹紧手动
W138.06 BOOL  ; 下料定位A2前后左右松开手动
W138.07 BOOL  ; 下料定位A2前后左右夹紧手动
W138.08 BOOL  ; 下料定位A3前后左右松开手动
W138.09 BOOL  ; 下料定位A3前后左右夹紧手动
W138.10 BOOL  ; 下料定位A4前后左右松开手动
W138.11 BOOL  ; 下料定位A4前后左右夹紧手动
W138.12 BOOL  ; 下料定位A5前后左右松开手动
W138.13 BOOL  ; 下料定位A5前后左右夹紧手动
W138.14 BOOL  ; 下料定位平台A吹气手动
W139.00 BOOL  ; 下料定位B下降手动
W139.01 BOOL  ; 下料定位B上升手动
W139.02 BOOL  ; 下料定位B0度翻转手动
W139.03 BOOL  ; 下料定位B90度翻转手动
W139.04 BOOL  ; 下料定位B1前后左右松开手动
W139.05 BOOL  ; 下料定位B1前后左右夹紧手动
W139.06 BOOL  ; 下料定位B2前后左右松开手动
W139.07 BOOL  ; 下料定位B2前后左右夹紧手动
W139.08 BOOL  ; 下料定位B3前后左右松开手动
W139.09 BOOL  ; 下料定位B3前后左右夹紧手动
W139.10 BOOL  ; 下料定位B4前后左右松开手动
W139.11 BOOL  ; 下料定位B4前后左右夹紧手动
W139.12 BOOL  ; 下料定位B5前后左右松开手动
W139.13 BOOL  ; 下料定位B5前后左右夹紧手动
W139.14 BOOL  ; 下料定位平台B吹气手动
W13.11 BOOL  ; 放料A位(12)
W13.14 BOOL  ; 初始位(15)
W14 CHANNEL  ; 上料夹爪状态正确
W140.00 BOOL  ; 进料定位上层前后松开[M]
W140.01 BOOL  ; 进料定位上层前后夹紧[M]
W140.02 BOOL  ; 进料定位下层前后松开[M]
W140.03 BOOL  ; 进料定位下层前后夹紧[M]
W140.04 BOOL  ; 进料定位上层左右松开[M]
W140.05 BOOL  ; 进料定位上层左右夹紧[M]
W140.06 BOOL  ; 进料定位下层左右松开[M]
W140.07 BOOL  ; 进料定位下层左右夹紧[M]
W140.08 BOOL  ; 进料定位上层平台待料[M]
W140.09 BOOL  ; 进料定位上层平台出料[M]
W140.10 BOOL  ; 进料定位下层平台待料[M]
W140.11 BOOL  ; 进料定位下层平台出料[M]
W143.00 BOOL  ; 出料定位上层前后松开[M]
W143.01 BOOL  ; 出料定位上层前后夹紧[M]
W143.02 BOOL  ; 出料定位下层前后松开[M]
W143.03 BOOL  ; 出料定位下层前后夹紧[M]
W143.04 BOOL  ; 出料定位上层左右松开[M]
W143.05 BOOL  ; 出料定位上层左右夹紧[M]
W143.06 BOOL  ; 出料定位下层左右松开[M]
W143.07 BOOL  ; 出料定位下层左右夹紧[M]
W143.08 BOOL  ; 出料定位上层平台接料[M]
W143.09 BOOL  ; 出料定位上层平台出料[M]
W143.10 BOOL  ; 出料定位下层平台接料[M]
W143.11 BOOL  ; 出料定位下层平台出料[M]
W143.12 BOOL  ; 上下层吹气[M]
W146.00 BOOL  ; 进料夹爪张开[M]
W146.01 BOOL  ; 进料夹爪夹紧[M]
W146.02 BOOL  ; 进料爪上下层左右压紧上升[M]
W146.03 BOOL  ; 进料爪上下层左右压紧下降[M]
W146.04 BOOL  ; 进料爪上下层中间压紧上升[M]
W146.05 BOOL  ; 进料爪上下层中间压紧下降[M]
W146.06 BOOL  ; 进料夹爪上升[M]
W146.07 BOOL  ; 进料夹爪下降[M]
W147.00 BOOL  ; 出料夹爪张开[M]
W147.01 BOOL  ; 出料夹爪夹紧[M]
W147.02 BOOL  ; 出料爪上下层左右压紧上升[M]
W147.03 BOOL  ; 出料爪上下层左右压紧下降[M]
W147.04 BOOL  ; 出料夹爪上升[M]
W147.05 BOOL  ; 出料夹爪下降[M]
W150.00 BOOL  ; 热压A增压缸上升[M]
W150.01 BOOL  ; 热压A增压缸下降[M]
W150.02 BOOL  ; 热压A上层顶升气缸上升[M]
W150.03 BOOL  ; 热压A上层顶升气缸下降[M]
W150.04 BOOL  ; 热压A下层顶升气缸上升[M]
W150.05 BOOL  ; 热压A下层顶升气缸下降[M]
W150.06 BOOL  ; 热压A垫高气缸移出[M]
W150.07 BOOL  ; 热压A垫高气缸热压[M]
W150.08 BOOL  ; 热压AHip测试气缸上升[M]
W150.09 BOOL  ; 热压AHip测试气缸下降[M]
W150.10 BOOL  ; 热压A上下层吹气[M]
W150.11 BOOL  ; 热压A上层HIP测试选择[M]
W150.12 BOOL  ; 热压A下层HIP测试选择[M]
W150.13 BOOL  ; 热压A极耳测试[M]
W150.14 BOOL  ; 热压A压力清零[M]
W153.00 BOOL  ; 热压B增压缸上升[M]
W153.01 BOOL  ; 热压B增压缸下降[M]
W153.02 BOOL  ; 热压B上层顶升气缸上升[M]
W153.03 BOOL  ; 热压B上层顶升气缸下降[M]
W153.04 BOOL  ; 热压B下层顶升气缸上升[M]
W153.05 BOOL  ; 热压B下层顶升气缸下降[M]
W153.06 BOOL  ; 热压B垫高气缸移出[M]
W153.07 BOOL  ; 热压B垫高气缸热压[M]
W153.08 BOOL  ; 热压BHip测试气缸上升[M]
W153.09 BOOL  ; 热压BHip测试气缸下降[M]
W153.10 BOOL  ; 热压B上下层吹气[M]
W153.11 BOOL  ; 热压B上层HIP测试选择[M]
W153.12 BOOL  ; 热压B下层HIP测试选择[M]
W153.13 BOOL  ; 热压B极耳测试[M]
W153.14 BOOL  ; 热压B压力清零[M]
W156.00 BOOL  ; 热压C增压缸上升[M]
W156.01 BOOL  ; 热压C增压缸下降[M]
W156.02 BOOL  ; 热压C上层顶升气缸上升[M]
W156.03 BOOL  ; 热压C上层顶升气缸下降[M]
W156.04 BOOL  ; 热压C下层顶升气缸上升[M]
W156.05 BOOL  ; 热压C下层顶升气缸下降[M]
W156.06 BOOL  ; 热压C垫高气缸移出[M]
W156.07 BOOL  ; 热压C垫高气缸热压[M]
W156.08 BOOL  ; 热压CHip测试气缸上升[M]
W156.09 BOOL  ; 热压CHip测试气缸下降[M]
W156.10 BOOL  ; 热压C上下层吹气[M]
W156.11 BOOL  ; 热压C上层HIP测试选择[M]
W156.12 BOOL  ; 热压C下层HIP测试选择[M]
W156.13 BOOL  ; 热压C极耳测试[M]
W156.14 BOOL  ; 热压C压力清零[M]
W15.00 BOOL  ; 1ST-手动允许输出
W15.01 BOOL  ; 1ST-自动允许输出
W16.00 BOOL  ; 进料平台可取料
W180.00 BOOL  ; 进料定位上层前后松开[A]
W180.01 BOOL  ; 进料定位上层前后夹紧[A]
W180.02 BOOL  ; 进料定位下层前后松开[A]
W180.03 BOOL  ; 进料定位下层前后夹紧[A]
W180.04 BOOL  ; 进料定位上层左右松开[A]
W180.05 BOOL  ; 进料定位上层左右夹紧[A]
W180.06 BOOL  ; 进料定位下层左右松开[A]
W180.07 BOOL  ; 进料定位下层左右夹紧[A]
W180.08 BOOL  ; 进料定位上层平台待料[A]
W180.09 BOOL  ; 进料定位上层平台出料[A]
W180.10 BOOL  ; 进料定位下层平台待料[A]
W180.11 BOOL  ; 进料定位下层平台出料[A]
W183.00 BOOL  ; 出料定位上层前后松开[A]
W183.01 BOOL  ; 出料定位上层前后夹紧[A]
W183.02 BOOL  ; 出料定位下层前后松开[A]
W183.03 BOOL  ; 出料定位下层前后夹紧[A]
W183.04 BOOL  ; 出料定位上层左右松开[A]
W183.05 BOOL  ; 出料定位上层左右夹紧[A]
W183.06 BOOL  ; 出料定位下层左右松开[A]
W183.07 BOOL  ; 出料定位下层左右夹紧[A]
W183.08 BOOL  ; 出料定位上层平台接料[A]
W183.09 BOOL  ; 出料定位上层平台出料[A]
W183.10 BOOL  ; 出料定位下层平台接料[A]
W183.11 BOOL  ; 出料定位下层平台出料[A]
W183.12 BOOL  ; 上下层吹气[A]
W186.00 BOOL  ; 进料夹爪张开[A]
W186.01 BOOL  ; 进料夹爪夹紧[A]
W186.02 BOOL  ; 进料爪上下层左右压紧上升[A]
W186.03 BOOL  ; 进料爪上下层左右压紧下降[A]
W186.04 BOOL  ; 进料爪上下层中间压紧上升[A]
W186.05 BOOL  ; 进料爪上下层中间压紧下降[A]
W186.06 BOOL  ; 进料夹爪上升[A]
W186.07 BOOL  ; 进料夹爪下降[A]
W187.00 BOOL  ; 出料夹爪张开[A]
W187.01 BOOL  ; 出料夹爪夹紧[A]
W187.02 BOOL  ; 出料爪上下层左右压紧上升[A]
W187.03 BOOL  ; 出料爪上下层左右压紧下降[A]
W187.04 BOOL  ; 出料夹爪上升[A]
W187.05 BOOL  ; 出料夹爪下降[A]
W190.00 BOOL  ; 热压A增压缸上升[A]
W190.01 BOOL  ; 热压A增压缸下降[A]
W190.02 BOOL  ; 热压A上层顶升气缸上升[A]
W190.03 BOOL  ; 热压A上层顶升气缸下降[A]
W190.04 BOOL  ; 热压A下层顶升气缸上升[A]
W190.05 BOOL  ; 热压A下层顶升气缸下降[A]
W190.06 BOOL  ; 热压A垫高气缸移出[A]
W190.07 BOOL  ; 热压A垫高气缸热压[A]
W190.08 BOOL  ; 热压AHip测试气缸上升[A]
W190.09 BOOL  ; 热压AHip测试气缸下降[A]
W190.10 BOOL  ; 热压A上下层吹气[A]
W190.11 BOOL  ; 热压A上层HIP测试选择[A]
W190.12 BOOL  ; 热压A下层HIP测试选择[A]
W190.13 BOOL  ; 热压A极耳测试[A]
W190.14 BOOL  ; 热压A压力清零[A]
W193.00 BOOL  ; 热压B增压缸上升[A]
W193.01 BOOL  ; 热压B增压缸下降[A]
W193.02 BOOL  ; 热压B上层顶升气缸上升[A]
W193.03 BOOL  ; 热压B上层顶升气缸下降[A]
W193.04 BOOL  ; 热压B下层顶升气缸上升[A]
W193.05 BOOL  ; 热压B下层顶升气缸下降[A]
W193.06 BOOL  ; 热压B垫高气缸移出[A]
W193.07 BOOL  ; 热压B垫高气缸热压[A]
W193.08 BOOL  ; 热压BHip测试气缸上升[A]
W193.09 BOOL  ; 热压BHip测试气缸下降[A]
W193.10 BOOL  ; 热压B上下层吹气[A]
W193.11 BOOL  ; 热压B上层HIP测试选择[A]
W193.12 BOOL  ; 热压B下层HIP测试选择[A]
W193.13 BOOL  ; 热压B极耳测试[A]
W193.14 BOOL  ; 热压B压力清零[A]
W196.00 BOOL  ; 热压C增压缸上升[A]
W196.01 BOOL  ; 热压C增压缸下降[A]
W196.02 BOOL  ; 热压C上层顶升气缸上升[A]
W196.03 BOOL  ; 热压C上层顶升气缸下降[A]
W196.04 BOOL  ; 热压C下层顶升气缸上升[A]
W196.05 BOOL  ; 热压C下层顶升气缸下降[A]
W196.06 BOOL  ; 热压C垫高气缸移出[A]
W196.07 BOOL  ; 热压C垫高气缸热压[A]
W196.08 BOOL  ; 热压CHip测试气缸上升[A]
W196.09 BOOL  ; 热压CHip测试气缸下降[A]
W196.10 BOOL  ; 热压C上下层吹气[A]
W196.11 BOOL  ; 热压C上层HIP测试选择[A]
W196.12 BOOL  ; 热压C下层HIP测试选择[A]
W196.13 BOOL  ; 热压C极耳测试[A]
W196.14 BOOL  ; 热压C压力清零[A]
W201 CHANNEL  ; 副PLC加热控制字
W20.00 BOOL  ; 2ST-B手动允许输出
W20.01 BOOL  ; 2ST-B自动允许输出
W210.00 BOOL  ; 进出料横移伺服A回原点手动(HMI)
W210.01 BOOL  ; 进出料横移伺服A错误清除(HMI)
W210.02 BOOL  ; 进出料横移伺服AJOG高速(HMI)
W210.03 BOOL  ; 进出料横移伺服AJOG低速（（HMI）
W210.04 BOOL  ; 进出料横移伺服AJOG+（HMI）
W210.05 BOOL  ; 进出料横移伺服AJOG-（HMI）
W210.06 BOOL  ; 进出料横移伺服A进料位设置（HMI）
W210.07 BOOL  ; 进出料横移伺服A进料等待位设置（HMI）
W210.08 BOOL  ; 进出料横移伺服A上料位A设置（HMI）
W210.09 BOOL  ; 进出料横移伺服A上料位B设置（HMI）
W210.10 BOOL  ; 进出料横移伺服A下料位A设置（HMI）
W210.11 BOOL  ; 进出料横移伺服A下料位B设置（HMI）
W210.12 BOOL  ; 进出料横移伺服A出料等待位设置（HMI）
W210.13 BOOL  ; 进出料横移伺服A出料位设置（HMI）
W210.14 BOOL  ; 进出料横移伺服A位置9设置（HMI）
W210.15 BOOL  ; 进出料横移伺服A位置10设置（HMI）
W211.00 BOOL  ; 进出料横移伺服A进料位手动(HMI)
W211.01 BOOL  ; 进出料横移伺服A进料等待位手动(HMI)
W211.02 BOOL  ; 进出料横移伺服A上料位A手动(HMI)
W211.03 BOOL  ; 进出料横移伺服A上料位B手动(HMI)
W211.04 BOOL  ; 进出料横移伺服A下料位A手动(HMI)
W211.05 BOOL  ; 进出料横移伺服A下料位B手动(HMI)
W211.06 BOOL  ; 进出料横移伺服A出料等待位手动(HMI)
W211.07 BOOL  ; 进出料横移伺服A出料位手动(HMI)
W211.08 BOOL  ; 进出料横移伺服A位置9手动(HMI)
W211.09 BOOL  ; 进出料横移伺服A位置10手动(HMI)
W211.10 BOOL  ; 进出料横移伺服A回原条件
W211.11 BOOL  ; 进出料横移伺服A运行锁定
W211.12 BOOL  ; 进出料横移伺服A定位条件
W211.13 BOOL  ; 进出料横移伺服A回原启动
W211.14 BOOL  ; 进出料横移伺服A回原完成
W211.15 BOOL  ; 进出料横移伺服A辅助3
W212.00 BOOL  ; 进出料伸缩伺服A回原点手动(HMI)
W212.01 BOOL  ; 进出料伸缩伺服A错误清除(HMI)
W212.02 BOOL  ; 进出料伸缩伺服AJOG高速(HMI)
W212.03 BOOL  ; 进出料伸缩伺服AJOG低速（（HMI）
W212.04 BOOL  ; 进出料伸缩伺服AJOG+（HMI）
W212.05 BOOL  ; 进出料伸缩伺服AJOG-（HMI）
W212.06 BOOL  ; 进出料伸缩伺服A初始位设置（HMI）
W212.07 BOOL  ; 进出料伸缩伺服A平台取料位设置（HMI）
W212.08 BOOL  ; 进出料伸缩伺服A热压取放位设置（HMI）
W212.09 BOOL  ; 进出料伸缩伺服A平台放料位设置（HMI）
W212.10 BOOL  ; 进出料伸缩伺服A位置5设置（HMI）
W212.11 BOOL  ; 进出料伸缩伺服A位置6设置（HMI）
W212.12 BOOL  ; 进出料伸缩伺服A位置7设置（HMI）
W212.13 BOOL  ; 进出料伸缩伺服A位置8设置（HMI）
W212.14 BOOL  ; 进出料伸缩伺服A位置9设置（HMI）
W212.15 BOOL  ; 进出料伸缩伺服A位置10设置（HMI）
W213.00 BOOL  ; 进出料伸缩伺服A初始位手动(HMI)
W213.01 BOOL  ; 进出料伸缩伺服A平台取料位手动(HMI)
W213.02 BOOL  ; 进出料伸缩伺服A热压取放位手动(HMI)
W213.03 BOOL  ; 进出料伸缩伺服A平台放料位手动(HMI)
W213.04 BOOL  ; 进出料伸缩伺服A位置5手动(HMI)
W213.05 BOOL  ; 进出料伸缩伺服A位置6手动(HMI)
W213.06 BOOL  ; 进出料伸缩伺服A位置7手动(HMI)
W213.07 BOOL  ; 进出料伸缩伺服A位置8手动(HMI)
W213.08 BOOL  ; 进出料伸缩伺服A位置9手动(HMI)
W213.09 BOOL  ; 进出料伸缩伺服A位置10手动(HMI)
W213.10 BOOL  ; 进出料伸缩伺服A回原条件
W213.11 BOOL  ; 进出料伸缩伺服A运行锁定
W213.12 BOOL  ; 进出料伸缩伺服A定位条件
W213.13 BOOL  ; 进出料伸缩伺服A回原启动
W213.14 BOOL  ; 进出料伸缩伺服A回原完成
W213.15 BOOL  ; 进出料伸缩伺服A辅助3
W214.00 BOOL  ; 进出料横移伺服B回原点手动(HMI)
W214.01 BOOL  ; 进出料横移伺服B错误清除(HMI)
W214.02 BOOL  ; 进出料横移伺服BJOG高速(HMI)
W214.03 BOOL  ; 进出料横移伺服BJOG低速（（HMI）
W214.04 BOOL  ; 进出料横移伺服BJOG+（HMI）
W214.05 BOOL  ; 进出料横移伺服BJOG-（HMI）
W214.06 BOOL  ; 进出料横移伺服B进料位设置（HMI）
W214.07 BOOL  ; 进出料横移伺服B进料等待位设置（HMI）
W214.08 BOOL  ; 进出料横移伺服B上料位A设置（HMI）
W214.09 BOOL  ; 进出料横移伺服B上料位B设置（HMI）
W214.10 BOOL  ; 进出料横移伺服B下料位A设置（HMI）
W214.11 BOOL  ; 进出料横移伺服B下料位B设置（HMI）
W214.12 BOOL  ; 进出料横移伺服B出料等待位设置（HMI）
W214.13 BOOL  ; 进出料横移伺服B出料位设置（HMI）
W214.14 BOOL  ; 进出料横移伺服B位置9设置（HMI）
W214.15 BOOL  ; 进出料横移伺服B位置10设置（HMI）
W215.00 BOOL  ; 进出料横移伺服B进料位手动(HMI)
W215.01 BOOL  ; 进出料横移伺服B进料等待位手动(HMI)
W215.02 BOOL  ; 进出料横移伺服B上料位A手动(HMI)
W215.03 BOOL  ; 进出料横移伺服B上料位B手动(HMI)
W215.04 BOOL  ; 进出料横移伺服B下料位A手动(HMI)
W215.05 BOOL  ; 进出料横移伺服B下料位B手动(HMI)
W215.06 BOOL  ; 进出料横移伺服B出料等待位手动(HMI)
W215.07 BOOL  ; 进出料横移伺服B出料位手动(HMI)
W215.08 BOOL  ; 进出料横移伺服B位置9手动(HMI)
W215.09 BOOL  ; 进出料横移伺服B位置10手动(HMI)
W215.10 BOOL  ; 进出料横移伺服B回原条件
W215.11 BOOL  ; 进出料横移伺服B运行锁定
W215.12 BOOL  ; 进出料横移伺服B定位条件
W215.13 BOOL  ; 进出料横移伺服B回原启动
W215.14 BOOL  ; 进出料横移伺服B回原完成
W215.15 BOOL  ; 进出料横移伺服B辅助3
W216.00 BOOL  ; 进出料伸缩伺服B回原点手动(HMI)
W216.01 BOOL  ; 进出料伸缩伺服B错误清除(HMI)
W216.02 BOOL  ; 进出料伸缩伺服BJOG高速(HMI)
W216.03 BOOL  ; 进出料伸缩伺服BJOG低速（（HMI）
W216.04 BOOL  ; 进出料伸缩伺服BJOG+（HMI）
W216.05 BOOL  ; 进出料伸缩伺服BJOG-（HMI）
W216.06 BOOL  ; 进出料伸缩伺服B初始位设置（HMI）
W216.07 BOOL  ; 进出料伸缩伺服B平台取料位设置（HMI）
W216.08 BOOL  ; 进出料伸缩伺服B热压取放位设置（HMI）
W216.09 BOOL  ; 进出料伸缩伺服B平台放料位设置（HMI）
W216.10 BOOL  ; 进出料伸缩伺服B位置5设置（HMI）
W216.11 BOOL  ; 进出料伸缩伺服B位置6设置（HMI）
W216.12 BOOL  ; 进出料伸缩伺服B位置7设置（HMI）
W216.13 BOOL  ; 进出料伸缩伺服B位置8设置（HMI）
W216.14 BOOL  ; 进出料伸缩伺服B位置9设置（HMI）
W216.15 BOOL  ; 进出料伸缩伺服B位置10设置（HMI）
W217.00 BOOL  ; 进出料伸缩伺服B初始位手动(HMI)
W217.01 BOOL  ; 进出料伸缩伺服B平台取料位手动(HMI)
W217.02 BOOL  ; 进出料伸缩伺服B热压取放位手动(HMI)
W217.03 BOOL  ; 进出料伸缩伺服B平台放料位手动(HMI)
W217.04 BOOL  ; 进出料伸缩伺服B位置5手动(HMI)
W217.05 BOOL  ; 进出料伸缩伺服B位置6手动(HMI)
W217.06 BOOL  ; 进出料伸缩伺服B位置7手动(HMI)
W217.07 BOOL  ; 进出料伸缩伺服B位置8手动(HMI)
W217.08 BOOL  ; 进出料伸缩伺服B位置9手动(HMI)
W217.09 BOOL  ; 进出料伸缩伺服B位置10手动(HMI)
W217.10 BOOL  ; 进出料伸缩伺服B回原条件
W217.11 BOOL  ; 进出料伸缩伺服B运行锁定
W217.12 BOOL  ; 进出料伸缩伺服B定位条件
W217.13 BOOL  ; 进出料伸缩伺服B回原启动
W217.14 BOOL  ; 进出料伸缩伺服B回原完成
W217.15 BOOL  ; 进出料伸缩伺服B辅助3
W218.00 BOOL  ; 下料定位A下降[A]
W218.01 BOOL  ; 下料定位A上升[A]
W218.02 BOOL  ; 下料定位A0度翻转[A]
W218.03 BOOL  ; 下料定位A90度翻转[A]
W218.04 BOOL  ; 下料定位A1前后左右松开[A]
W218.05 BOOL  ; 下料定位A1前后左右夹紧[A]
W218.06 BOOL  ; 下料定位A2前后左右松开[A]
W218.07 BOOL  ; 下料定位A2前后左右夹紧[A]
W218.08 BOOL  ; 下料定位A3前后左右松开[A]
W218.09 BOOL  ; 下料定位A3前后左右夹紧[A]
W218.10 BOOL  ; 下料定位A4前后左右松开[A]
W218.11 BOOL  ; 下料定位A4前后左右夹紧[A]
W218.12 BOOL  ; 下料定位A5前后左右松开[A]
W218.13 BOOL  ; 下料定位A5前后左右夹紧[A]
W218.14 BOOL  ; 下料定位平台A吹气[A]
W219.00 BOOL  ; 下料定位B下降[A]
W219.01 BOOL  ; 下料定位B上升[A]
W219.02 BOOL  ; 下料定位B0度翻转[A]
W219.03 BOOL  ; 下料定位B90度翻转[A]
W219.04 BOOL  ; 下料定位B1前后左右松开[A]
W219.05 BOOL  ; 下料定位B1前后左右夹紧[A]
W219.06 BOOL  ; 下料定位B2前后左右松开[A]
W219.07 BOOL  ; 下料定位B2前后左右夹紧[A]
W219.08 BOOL  ; 下料定位B3前后左右松开[A]
W219.09 BOOL  ; 下料定位B3前后左右夹紧[A]
W219.10 BOOL  ; 下料定位B4前后左右松开[A]
W219.11 BOOL  ; 下料定位B4前后左右夹紧[A]
W219.12 BOOL  ; 下料定位B5前后左右松开[A]
W219.13 BOOL  ; 下料定位B5前后左右夹紧[A]
W219.14 BOOL  ; 下料定位平台B吹气[A]
W21.00 BOOL  ; 出料平台出料允许
W220.00 BOOL  ; 进出料横移伺服A回原点手动(HMI)
W220.01 BOOL  ; 进出料横移伺服A错误清除(HMI)
W220.02 BOOL  ; 进出料横移伺服AJOG高速(HMI)
W220.03 BOOL  ; 进出料横移伺服AJOG低速（（HMI）
W220.04 BOOL  ; 进出料横移伺服AJOG+（HMI）
W220.05 BOOL  ; 进出料横移伺服AJOG-（HMI）
W220.06 BOOL  ; 进出料横移伺服A进料位设置（HMI）
W220.07 BOOL  ; 进出料横移伺服A进料等待位设置（HMI）
W220.08 BOOL  ; 进出料横移伺服A上料位A设置（HMI）
W220.09 BOOL  ; 进出料横移伺服A上料位B设置（HMI）
W220.10 BOOL  ; 进出料横移伺服A下料位A设置（HMI）
W220.11 BOOL  ; 进出料横移伺服A下料位B设置（HMI）
W220.12 BOOL  ; 进出料横移伺服A出料等待位设置（HMI）
W220.13 BOOL  ; 进出料横移伺服A出料位设置（HMI）
W220.14 BOOL  ; 进出料横移伺服A位置9设置（HMI）
W220.15 BOOL  ; 进出料横移伺服A位置10设置（HMI）
W221.00 BOOL  ; 进出料横移伺服A进料位手动(HMI)
W221.01 BOOL  ; 进出料横移伺服A进料等待位手动(HMI)
W221.02 BOOL  ; 进出料横移伺服A上料位A手动(HMI)
W221.03 BOOL  ; 进出料横移伺服A上料位B手动(HMI)
W221.04 BOOL  ; 进出料横移伺服A下料位A手动(HMI)
W221.05 BOOL  ; 进出料横移伺服A下料位C手动(HMI)
W221.06 BOOL  ; 进出料横移伺服A取料位C手动(HMI)
W221.07 BOOL  ; 进出料横移伺服A出料位手动(HMI)
W221.08 BOOL  ; 进出料横移伺服A位置9手动(HMI)
W221.09 BOOL  ; 进出料横移伺服A位置10手动(HMI)
W221.10 BOOL  ; 进出料横移伺服A回原条件
W221.11 BOOL  ; 进出料横移伺服A运行锁定
W221.12 BOOL  ; 进出料横移伺服A定位条件
W221.13 BOOL  ; 进出料横移伺服A回原启动
W221.14 BOOL  ; 进出料横移伺服A回原完成
W221.15 BOOL  ; 进出料横移伺服A辅助3
W222.00 BOOL  ; 进出料伸缩伺服A回原点手动(HMI)
W222.01 BOOL  ; 进出料伸缩伺服A错误清除(HMI)
W222.02 BOOL  ; 进出料伸缩伺服AJOG高速(HMI)
W222.03 BOOL  ; 进出料伸缩伺服AJOG低速（（HMI）
W222.04 BOOL  ; 进出料伸缩伺服AJOG+（HMI）
W222.05 BOOL  ; 进出料伸缩伺服AJOG-（HMI）
W222.06 BOOL  ; 进出料伸缩伺服A初始位设置（HMI）
W222.07 BOOL  ; 进出料伸缩伺服A平台取料位设置（HMI）
W222.08 BOOL  ; 进出料伸缩伺服A热压取放位设置（HMI）
W222.09 BOOL  ; 进出料伸缩伺服A平台放料位设置（HMI）
W222.10 BOOL  ; 进出料伸缩伺服A位置5设置（HMI）
W222.11 BOOL  ; 进出料伸缩伺服A位置6设置（HMI）
W222.12 BOOL  ; 进出料伸缩伺服A位置7设置（HMI）
W222.13 BOOL  ; 进出料伸缩伺服A位置8设置（HMI）
W222.14 BOOL  ; 进出料伸缩伺服A位置9设置（HMI）
W222.15 BOOL  ; 进出料伸缩伺服A位置10设置（HMI）
W223.00 BOOL  ; 进出料伸缩伺服A初始位手动(HMI)
W223.01 BOOL  ; 进出料伸缩伺服A平台取料位手动(HMI)
W223.02 BOOL  ; 进出料伸缩伺服A热压取放位手动(HMI)
W223.03 BOOL  ; 进出料伸缩伺服A平台放料位手动(HMI)
W223.04 BOOL  ; 进出料伸缩伺服A位置5手动(HMI)
W223.05 BOOL  ; 进出料伸缩伺服A位置6手动(HMI)
W223.06 BOOL  ; 进出料伸缩伺服A位置7手动(HMI)
W223.07 BOOL  ; 进出料伸缩伺服A位置8手动(HMI)
W223.08 BOOL  ; 进出料伸缩伺服A位置9手动(HMI)
W223.09 BOOL  ; 进出料伸缩伺服A位置10手动(HMI)
W223.10 BOOL  ; 进出料伸缩伺服A回原条件
W223.11 BOOL  ; 进出料伸缩伺服A运行锁定
W223.12 BOOL  ; 进出料伸缩伺服A定位条件
W223.13 BOOL  ; 进出料伸缩伺服A回原启动
W223.14 BOOL  ; 进出料伸缩伺服A回原完成
W223.15 BOOL  ; 进出料伸缩伺服A辅助3
W224.00 BOOL  ; 进出料横移伺服B回原点手动(HMI)
W224.01 BOOL  ; 进出料横移伺服B错误清除(HMI)
W224.02 BOOL  ; 进出料横移伺服BJOG高速(HMI)
W224.03 BOOL  ; 进出料横移伺服BJOG低速（（HMI）
W224.04 BOOL  ; 进出料横移伺服BJOG+（HMI）
W224.05 BOOL  ; 进出料横移伺服BJOG-（HMI）
W224.06 BOOL  ; 进出料横移伺服B进料位设置（HMI）
W224.07 BOOL  ; 进出料横移伺服B进料等待位设置（HMI）
W224.08 BOOL  ; 进出料横移伺服B上料位A设置（HMI）
W224.09 BOOL  ; 进出料横移伺服B上料位B设置（HMI）
W224.10 BOOL  ; 进出料横移伺服B下料位A设置（HMI）
W224.11 BOOL  ; 进出料横移伺服B下料位B设置（HMI）
W224.12 BOOL  ; 进出料横移伺服B出料等待位设置（HMI）
W224.13 BOOL  ; 进出料横移伺服B出料位设置（HMI）
W224.14 BOOL  ; 进出料横移伺服B位置9设置（HMI）
W224.15 BOOL  ; 进出料横移伺服B位置10设置（HMI）
W225.00 BOOL  ; 进出料横移伺服B进料位手动(HMI)
W225.01 BOOL  ; 进出料横移伺服B进料等待位手动(HMI)
W225.02 BOOL  ; 进出料横移伺服B上料位A手动(HMI)
W225.03 BOOL  ; 进出料横移伺服B上料位B手动(HMI)
W225.04 BOOL  ; 进出料横移伺服B下料位A手动(HMI)
W225.05 BOOL  ; 进出料横移伺服B下料位B手动(HMI)
W225.06 BOOL  ; 进出料横移伺服B出料等待位手动(HMI)
W225.07 BOOL  ; 进出料横移伺服B出料位手动(HMI)
W225.08 BOOL  ; 进出料横移伺服B位置9手动(HMI)
W225.09 BOOL  ; 进出料横移伺服B位置10手动(HMI)
W225.10 BOOL  ; 进出料横移伺服B回原条件
W225.11 BOOL  ; 进出料横移伺服B运行锁定
W225.12 BOOL  ; 进出料横移伺服B定位条件
W225.13 BOOL  ; 进出料横移伺服B回原启动
W225.14 BOOL  ; 进出料横移伺服B回原完成
W225.15 BOOL  ; 进出料横移伺服B辅助3
W226.00 BOOL  ; 进出料伸缩伺服B回原点手动(HMI)
W226.01 BOOL  ; 进出料伸缩伺服B错误清除(HMI)
W226.02 BOOL  ; 进出料伸缩伺服BJOG高速(HMI)
W226.03 BOOL  ; 进出料伸缩伺服BJOG低速（（HMI）
W226.04 BOOL  ; 进出料伸缩伺服BJOG+（HMI）
W226.05 BOOL  ; 进出料伸缩伺服BJOG-（HMI）
W226.06 BOOL  ; 进出料伸缩伺服B初始位设置（HMI）
W226.07 BOOL  ; 进出料伸缩伺服B平台取料位设置（HMI）
W226.08 BOOL  ; 进出料伸缩伺服B热压取放位设置（HMI）
W226.09 BOOL  ; 进出料伸缩伺服B平台放料位设置（HMI）
W226.10 BOOL  ; 进出料伸缩伺服B位置5设置（HMI）
W226.11 BOOL  ; 进出料伸缩伺服B位置6设置（HMI）
W226.12 BOOL  ; 进出料伸缩伺服B位置7设置（HMI）
W226.13 BOOL  ; 进出料伸缩伺服B位置8设置（HMI）
W226.14 BOOL  ; 进出料伸缩伺服B位置9设置（HMI）
W226.15 BOOL  ; 进出料伸缩伺服B位置10设置（HMI）
W227.00 BOOL  ; 进出料伸缩伺服B初始位手动(HMI)
W227.01 BOOL  ; 进出料伸缩伺服B平台取料位手动(HMI)
W227.02 BOOL  ; 进出料伸缩伺服B热压取放位手动(HMI)
W227.03 BOOL  ; 进出料伸缩伺服B平台放料位手动(HMI)
W227.04 BOOL  ; 进出料伸缩伺服B位置5手动(HMI)
W227.05 BOOL  ; 进出料伸缩伺服B位置6手动(HMI)
W227.06 BOOL  ; 进出料伸缩伺服B位置7手动(HMI)
W227.07 BOOL  ; 进出料伸缩伺服B位置8手动(HMI)
W227.08 BOOL  ; 进出料伸缩伺服B位置9手动(HMI)
W227.09 BOOL  ; 进出料伸缩伺服B位置10手动(HMI)
W227.10 BOOL  ; 进出料伸缩伺服B回原条件
W227.11 BOOL  ; 进出料伸缩伺服B运行锁定
W227.12 BOOL  ; 进出料伸缩伺服B定位条件
W227.13 BOOL  ; 进出料伸缩伺服B回原启动
W227.14 BOOL  ; 进出料伸缩伺服B回原完成
W227.15 BOOL  ; 进出料伸缩伺服B辅助3
W228.00 BOOL  ; 正压伺服A回原点手动(HMI)
W228.01 BOOL  ; 正压伺服A错误清除(HMI)
W228.02 BOOL  ; 正压伺服AJOG高速(HMI)
W228.03 BOOL  ; 正压伺服AJOG低速（（HMI）
W228.04 BOOL  ; 正压伺服AJOG+（HMI）
W228.05 BOOL  ; 正压伺服AJOG-（HMI）
W228.06 BOOL  ; 正压伺服A初始位设置（HMI）
W228.07 BOOL  ; 正压伺服A减速位设置（HMI）
W228.08 BOOL  ; 正压伺服A等距热压位设置（HMI）
W228.09 BOOL  ; 正压伺服A预压退回位设置（HMI）
W228.10 BOOL  ; 正压伺服AMASK测试位设置（HMI）
W228.11 BOOL  ; 正压伺服A位置6设置（HMI）
W228.12 BOOL  ; 正压伺服A位置7设置（HMI）
W228.13 BOOL  ; 正压伺服A位置8设置（HMI）
W228.14 BOOL  ; 正压伺服A位置9设置（HMI）
W228.15 BOOL  ; 正压伺服A位置10设置（HMI）
W229.00 BOOL  ; 正压伺服A初始位手动(HMI)
W229.01 BOOL  ; 正压伺服A减速位手动(HMI)
W229.02 BOOL  ; 正压伺服A等距热压位手动(HMI)
W229.03 BOOL  ; 正压伺服A预压退回位手动(HMI)
W229.04 BOOL  ; 正压伺服AMASK测试位手动(HMI)
W229.05 BOOL  ; 正压伺服A位置6手动(HMI)
W229.06 BOOL  ; 正压伺服A位置7手动(HMI)
W229.07 BOOL  ; 正压伺服A位置8手动(HMI)
W229.08 BOOL  ; 正压伺服A位置9手动(HMI)
W229.09 BOOL  ; 正压伺服A位置10手动(HMI)
W229.10 BOOL  ; 正压伺服A回原条件
W229.11 BOOL  ; 正压伺服A运行锁定
W229.12 BOOL  ; 正压伺服A定位条件
W229.13 BOOL  ; 正压伺服A回原启动
W229.14 BOOL  ; 正压伺服A回原完成
W229.15 BOOL  ; 正压伺服A辅助3
W230 CHANNEL  ; 副PLC加热自整定状态起始字
W230.00 BOOL  ; 压板平移伺服A回原点手动(HMI)
W230.01 BOOL  ; 压板平移伺服A错误清除(HMI)
W230.02 BOOL  ; 压板平移伺服AJOG高速(HMI)
W230.03 BOOL  ; 压板平移伺服AJOG低速（（HMI）
W230.04 BOOL  ; 压板平移伺服AJOG+（HMI）
W230.05 BOOL  ; 压板平移伺服AJOG-（HMI）
W230.06 BOOL  ; 压板平移伺服AA面取放位设置（HMI）
W230.07 BOOL  ; 压板平移伺服AB面取放位设置（HMI）
W230.08 BOOL  ; 压板平移伺服A位置3设置（HMI）
W230.09 BOOL  ; 压板平移伺服A位置4设置（HMI）
W230.10 BOOL  ; 压板平移伺服A位置5设置（HMI）
W230.11 BOOL  ; 压板平移伺服A位置6设置（HMI）
W230.12 BOOL  ; 压板平移伺服A位置7设置（HMI）
W230.13 BOOL  ; 压板平移伺服A位置8设置（HMI）
W230.14 BOOL  ; 压板平移伺服A位置9设置（HMI）
W230.15 BOOL  ; 压板平移伺服A位置10设置（HMI）
W231.00 BOOL  ; 压板平移伺服AA面取放位手动(HMI)
W231.01 BOOL  ; 压板平移伺服AB面取放位手动(HMI)
W231.02 BOOL  ; 压板平移伺服A位置3手动(HMI)
W231.03 BOOL  ; 压板平移伺服A位置4手动(HMI)
W231.04 BOOL  ; 压板平移伺服A位置5手动(HMI)
W231.05 BOOL  ; 压板平移伺服A位置6手动(HMI)
W231.06 BOOL  ; 压板平移伺服A位置7手动(HMI)
W231.07 BOOL  ; 压板平移伺服A位置8手动(HMI)
W231.08 BOOL  ; 压板平移伺服A位置9手动(HMI)
W231.09 BOOL  ; 压板平移伺服A位置10手动(HMI)
W231.10 BOOL  ; 压板平移伺服A回原条件
W231.11 BOOL  ; 压板平移伺服A运行锁定
W231.12 BOOL  ; 压板平移伺服A定位条件
W231.13 BOOL  ; 压板平移伺服A回原启动
W231.14 BOOL  ; 压板平移伺服A回原完成
W231.15 BOOL  ; 压板平移伺服A辅助3
W232.00 BOOL  ; A1左伺服回原点手动(HMI)
W232.01 BOOL  ; A1左伺服错误清除(HMI)
W232.02 BOOL  ; A1左伺服JOG高速(HMI)
W232.03 BOOL  ; A1左伺服JOG低速（（HMI）
W232.04 BOOL  ; A1左伺服JOG+（HMI）
W232.05 BOOL  ; A1左伺服JOG-（HMI）
W232.06 BOOL  ; A1左伺服待机位设置（HMI）
W232.07 BOOL  ; A1左伺服拨料位设置（HMI）
W232.08 BOOL  ; A1左伺服减速位设置（HMI）
W232.09 BOOL  ; A1左伺服减速位设置（HMI）
W232.10 BOOL  ; A1左伺服等距热压位设置（HMI）
W232.11 BOOL  ; A1左伺服位置6设置（HMI）
W232.12 BOOL  ; A1左伺服位置7设置（HMI）
W232.13 BOOL  ; A1左伺服位置8设置（HMI）
W232.14 BOOL  ; A1左伺服位置9设置（HMI）
W232.15 BOOL  ; A1左伺服位置10设置（HMI）
W233.00 BOOL  ; A1左伺服待机位手动(HMI)
W233.01 BOOL  ; A1左伺服拨料位手动(HMI)
W233.02 BOOL  ; A1左伺服减速位手动(HMI)
W233.03 BOOL  ; A1左伺服减速位手动(HMI)
W233.04 BOOL  ; A1左伺服等距热压位手动(HMI)
W233.05 BOOL  ; A1左伺服位置6手动(HMI)
W233.06 BOOL  ; A1左伺服位置7手动(HMI)
W233.07 BOOL  ; A1左伺服位置8手动(HMI)
W233.08 BOOL  ; A1左伺服位置9手动(HMI)
W233.09 BOOL  ; A1左伺服位置10手动(HMI)
W233.10 BOOL  ; A1左伺服回原条件
W233.11 BOOL  ; A1左伺服运行锁定
W233.12 BOOL  ; A1左伺服定位条件
W233.13 BOOL  ; A1左伺服回原启动
W233.14 BOOL  ; A1左伺服回原完成
W233.15 BOOL  ; A1左伺服辅助3
W234.00 BOOL  ; A1右伺服回原点手动(HMI)
W234.01 BOOL  ; A1右伺服错误清除(HMI)
W234.02 BOOL  ; A1右伺服JOG高速(HMI)
W234.03 BOOL  ; A1右伺服JOG低速（（HMI）
W234.04 BOOL  ; A1右伺服JOG+（HMI）
W234.05 BOOL  ; A1右伺服JOG-（HMI）
W234.06 BOOL  ; A1右伺服待机位设置（HMI）
W234.07 BOOL  ; A1右伺服拨料退回位设置（HMI）
W234.08 BOOL  ; A1右伺服拨料位设置（HMI）
W234.09 BOOL  ; A1右伺服减速位设置（HMI）
W234.10 BOOL  ; A1右伺服等距热压位设置（HMI）
W234.11 BOOL  ; A1右伺服位置6设置（HMI）
W234.12 BOOL  ; A1右伺服位置7设置（HMI）
W234.13 BOOL  ; A1右伺服位置8设置（HMI）
W234.14 BOOL  ; A1右伺服位置9设置（HMI）
W234.15 BOOL  ; A1右伺服位置10设置（HMI）
W235.00 BOOL  ; A1右伺服待机位手动(HMI)
W235.01 BOOL  ; A1右伺服拨料退回位手动(HMI)
W235.02 BOOL  ; A1右伺服拨料位手动(HMI)
W235.03 BOOL  ; A1右伺服减速位手动(HMI)
W235.04 BOOL  ; A1右伺服等距热压位手动(HMI)
W235.05 BOOL  ; A1右伺服位置6手动(HMI)
W235.06 BOOL  ; A1右伺服位置7手动(HMI)
W235.07 BOOL  ; A1右伺服位置8手动(HMI)
W235.08 BOOL  ; A1右伺服位置9手动(HMI)
W235.09 BOOL  ; A1右伺服位置10手动(HMI)
W235.10 BOOL  ; A1右伺服回原条件
W235.11 BOOL  ; A1右伺服运行锁定
W235.12 BOOL  ; A1右伺服定位条件
W235.13 BOOL  ; A1右伺服回原启动
W235.14 BOOL  ; A1右伺服回原完成
W235.15 BOOL  ; A1右伺服辅助3
W236.00 BOOL  ; A2左伺服回原点手动(HMI)
W236.01 BOOL  ; A2左伺服错误清除(HMI)
W236.02 BOOL  ; A2左伺服JOG高速(HMI)
W236.03 BOOL  ; A2左伺服JOG低速（（HMI）
W236.04 BOOL  ; A2左伺服JOG+（HMI）
W236.05 BOOL  ; A2左伺服JOG-（HMI）
W236.06 BOOL  ; A2左伺服待机位设置（HMI）
W236.07 BOOL  ; A2左伺服拨料退回位设置（HMI）
W236.08 BOOL  ; A2左伺服拨料位设置（HMI）
W236.09 BOOL  ; A2左伺服减速位设置（HMI）
W236.10 BOOL  ; A2左伺服等距热压位设置（HMI）
W236.11 BOOL  ; A2左伺服位置6设置（HMI）
W236.12 BOOL  ; A2左伺服位置7设置（HMI）
W236.13 BOOL  ; A2左伺服位置8设置（HMI）
W236.14 BOOL  ; A2左伺服位置9设置（HMI）
W236.15 BOOL  ; A2左伺服位置10设置（HMI）
W237.00 BOOL  ; A2左伺服待机位手动(HMI)
W237.01 BOOL  ; A2左伺服拨料退回位手动(HMI)
W237.02 BOOL  ; A2左伺服拨料位手动(HMI)
W237.03 BOOL  ; A2左伺服减速位手动(HMI)
W237.04 BOOL  ; A2左伺服等距热压位手动(HMI)
W237.05 BOOL  ; A2左伺服位置6手动(HMI)
W237.06 BOOL  ; A2左伺服位置7手动(HMI)
W237.07 BOOL  ; A2左伺服位置8手动(HMI)
W237.08 BOOL  ; A2左伺服位置9手动(HMI)
W237.09 BOOL  ; A2左伺服位置10手动(HMI)
W237.10 BOOL  ; A2左伺服回原条件
W237.11 BOOL  ; A2左伺服运行锁定
W237.12 BOOL  ; A2左伺服定位条件
W237.13 BOOL  ; A2左伺服回原启动
W237.14 BOOL  ; A2左伺服回原完成
W237.15 BOOL  ; A2左伺服辅助3
W238.00 BOOL  ; A2右伺服回原点手动(HMI)
W238.01 BOOL  ; A2右伺服错误清除(HMI)
W238.02 BOOL  ; A2右伺服JOG高速(HMI)
W238.03 BOOL  ; A2右伺服JOG低速（（HMI）
W238.04 BOOL  ; A2右伺服JOG+（HMI）
W238.05 BOOL  ; A2右伺服JOG-（HMI）
W238.06 BOOL  ; A2右伺服待机位设置（HMI）
W238.07 BOOL  ; A2右伺服拨料退回位设置（HMI）
W238.08 BOOL  ; A2右伺服拨料位设置（HMI）
W238.09 BOOL  ; A2右伺服减速位设置（HMI）
W238.10 BOOL  ; A2右伺服等距热压位设置（HMI）
W238.11 BOOL  ; A2右伺服位置6设置（HMI）
W238.12 BOOL  ; A2右伺服位置7设置（HMI）
W238.13 BOOL  ; A2右伺服位置8设置（HMI）
W238.14 BOOL  ; A2右伺服位置9设置（HMI）
W238.15 BOOL  ; A2右伺服位置10设置（HMI）
W239.00 BOOL  ; A2右伺服待机位手动(HMI)
W239.01 BOOL  ; A2右伺服拨料退回位手动(HMI)
W239.02 BOOL  ; A2右伺服拨料位手动(HMI)
W239.03 BOOL  ; A2右伺服减速位手动(HMI)
W239.04 BOOL  ; A2右伺服等距热压位手动(HMI)
W239.05 BOOL  ; A2右伺服位置6手动(HMI)
W239.06 BOOL  ; A2右伺服位置7手动(HMI)
W239.07 BOOL  ; A2右伺服位置8手动(HMI)
W239.08 BOOL  ; A2右伺服位置9手动(HMI)
W239.09 BOOL  ; A2右伺服位置10手动(HMI)
W239.10 BOOL  ; A2右伺服回原条件
W239.11 BOOL  ; A2右伺服运行锁定
W239.12 BOOL  ; A2右伺服定位条件
W239.13 BOOL  ; A2右伺服回原启动
W239.14 BOOL  ; A2右伺服回原完成
W239.15 BOOL  ; A2右伺服辅助3
W240.00 BOOL  ; A3左伺服回原点手动(HMI)
W240.01 BOOL  ; A3左伺服错误清除(HMI)
W240.02 BOOL  ; A3左伺服JOG高速(HMI)
W240.03 BOOL  ; A3左伺服JOG低速（（HMI）
W240.04 BOOL  ; A3左伺服JOG+（HMI）
W240.05 BOOL  ; A3左伺服JOG-（HMI）
W240.06 BOOL  ; A3左伺服待机位设置（HMI）
W240.07 BOOL  ; A3左伺服拨料退回位设置（HMI）
W240.08 BOOL  ; A3左伺服拨料位设置（HMI）
W240.09 BOOL  ; A3左伺服减速位设置（HMI）
W240.10 BOOL  ; A3左伺服等距热压位设置（HMI）
W240.11 BOOL  ; A3左伺服位置6设置（HMI）
W240.12 BOOL  ; A3左伺服位置7设置（HMI）
W240.13 BOOL  ; A3左伺服位置8设置（HMI）
W240.14 BOOL  ; A3左伺服位置9设置（HMI）
W240.15 BOOL  ; A3左伺服位置10设置（HMI）
W241.00 BOOL  ; A3左伺服待机位手动(HMI)
W241.01 BOOL  ; A3左伺服拨料退回位手动(HMI)
W241.02 BOOL  ; A3左伺服拨料位手动(HMI)
W241.03 BOOL  ; A3左伺服减速位手动(HMI)
W241.04 BOOL  ; A3左伺服等距热压位手动(HMI)
W241.05 BOOL  ; A3左伺服位置6手动(HMI)
W241.06 BOOL  ; A3左伺服位置7手动(HMI)
W241.07 BOOL  ; A3左伺服位置8手动(HMI)
W241.08 BOOL  ; A3左伺服位置9手动(HMI)
W241.09 BOOL  ; A3左伺服位置10手动(HMI)
W241.10 BOOL  ; A3左伺服回原条件
W241.11 BOOL  ; A3左伺服运行锁定
W241.12 BOOL  ; A3左伺服定位条件
W241.13 BOOL  ; A3左伺服回原启动
W241.14 BOOL  ; A3左伺服回原完成
W241.15 BOOL  ; A3左伺服辅助3
W242.00 BOOL  ; A3右伺服回原点手动(HMI)
W242.01 BOOL  ; A3右伺服错误清除(HMI)
W242.02 BOOL  ; A3右伺服JOG高速(HMI)
W242.03 BOOL  ; A3右伺服JOG低速（（HMI）
W242.04 BOOL  ; A3右伺服JOG+（HMI）
W242.05 BOOL  ; A3右伺服JOG-（HMI）
W242.06 BOOL  ; A3右伺服待机位设置（HMI）
W242.07 BOOL  ; A3右伺服拨料退回位设置（HMI）
W242.08 BOOL  ; A3右伺服拨料位设置（HMI）
W242.09 BOOL  ; A3右伺服减速位设置（HMI）
W242.10 BOOL  ; A3右伺服等距热压位设置（HMI）
W242.11 BOOL  ; A3右伺服位置6设置（HMI）
W242.12 BOOL  ; A3右伺服位置7设置（HMI）
W242.13 BOOL  ; A3右伺服位置8设置（HMI）
W242.14 BOOL  ; A3右伺服位置9设置（HMI）
W242.15 BOOL  ; A3右伺服位置10设置（HMI）
W243.00 BOOL  ; A3右伺服待机位手动(HMI)
W243.01 BOOL  ; A3右伺服拨料退回位手动(HMI)
W243.02 BOOL  ; A3右伺服拨料位手动(HMI)
W243.03 BOOL  ; A3右伺服减速位手动(HMI)
W243.04 BOOL  ; A3右伺服等距热压位手动(HMI)
W243.05 BOOL  ; A3右伺服位置6手动(HMI)
W243.06 BOOL  ; A3右伺服位置7手动(HMI)
W243.07 BOOL  ; A3右伺服位置8手动(HMI)
W243.08 BOOL  ; A3右伺服位置9手动(HMI)
W243.09 BOOL  ; A3右伺服位置10手动(HMI)
W243.10 BOOL  ; A3右伺服回原条件
W243.11 BOOL  ; A3右伺服运行锁定
W243.12 BOOL  ; A3右伺服定位条件
W243.13 BOOL  ; A3右伺服回原启动
W243.14 BOOL  ; A3右伺服回原完成
W243.15 BOOL  ; A3右伺服辅助3
W244.00 BOOL  ; A4左伺服回原点手动(HMI)
W244.01 BOOL  ; A4左伺服错误清除(HMI)
W244.02 BOOL  ; A4左伺服JOG高速(HMI)
W244.03 BOOL  ; A4左伺服JOG低速（（HMI）
W244.04 BOOL  ; A4左伺服JOG+（HMI）
W244.05 BOOL  ; A4左伺服JOG-（HMI）
W244.06 BOOL  ; A4左伺服待机位设置（HMI）
W244.07 BOOL  ; A4左伺服拨料退回位设置（HMI）
W244.08 BOOL  ; A4左伺服拨料位设置（HMI）
W244.09 BOOL  ; A4左伺服减速位设置（HMI）
W244.10 BOOL  ; A4左伺服等距热压位设置（HMI）
W244.11 BOOL  ; A4左伺服位置6设置（HMI）
W244.12 BOOL  ; A4左伺服位置7设置（HMI）
W244.13 BOOL  ; A4左伺服位置8设置（HMI）
W244.14 BOOL  ; A4左伺服位置9设置（HMI）
W244.15 BOOL  ; A4左伺服位置10设置（HMI）
W245.00 BOOL  ; A4左伺服待机位手动(HMI)
W245.01 BOOL  ; A4左伺服拨料退回位手动(HMI)
W245.02 BOOL  ; A4左伺服拨料位手动(HMI)
W245.03 BOOL  ; A4左伺服减速位手动(HMI)
W245.04 BOOL  ; A4左伺服等距热压位手动(HMI)
W245.05 BOOL  ; A4左伺服位置6手动(HMI)
W245.06 BOOL  ; A4左伺服位置7手动(HMI)
W245.07 BOOL  ; A4左伺服位置8手动(HMI)
W245.08 BOOL  ; A4左伺服位置9手动(HMI)
W245.09 BOOL  ; A4左伺服位置10手动(HMI)
W245.10 BOOL  ; A4左伺服回原条件
W245.11 BOOL  ; A4左伺服运行锁定
W245.12 BOOL  ; A4左伺服定位条件
W245.13 BOOL  ; A4左伺服回原启动
W245.14 BOOL  ; A4左伺服回原完成
W245.15 BOOL  ; A4左伺服辅助3
W246.00 BOOL  ; A4右伺服回原点手动(HMI)
W246.01 BOOL  ; A4右伺服错误清除(HMI)
W246.02 BOOL  ; A4右伺服JOG高速(HMI)
W246.03 BOOL  ; A4右伺服JOG低速（（HMI）
W246.04 BOOL  ; A4右伺服JOG+（HMI）
W246.05 BOOL  ; A4右伺服JOG-（HMI）
W246.06 BOOL  ; A4右伺服待机位设置（HMI）
W246.07 BOOL  ; A4右伺服拨料退回位设置（HMI）
W246.08 BOOL  ; A4右伺服拨料位设置（HMI）
W246.09 BOOL  ; A4右伺服减速位设置（HMI）
W246.10 BOOL  ; A4右伺服等距热压位设置（HMI）
W246.11 BOOL  ; A4右伺服位置6设置（HMI）
W246.12 BOOL  ; A4右伺服位置7设置（HMI）
W246.13 BOOL  ; A4右伺服位置8设置（HMI）
W246.14 BOOL  ; A4右伺服位置9设置（HMI）
W246.15 BOOL  ; A4右伺服位置10设置（HMI）
W247.00 BOOL  ; A4右伺服待机位手动(HMI)
W247.01 BOOL  ; A4右伺服拨料退回位手动(HMI)
W247.02 BOOL  ; A4右伺服拨料位手动(HMI)
W247.03 BOOL  ; A4右伺服减速位手动(HMI)
W247.04 BOOL  ; A4右伺服等距热压位手动(HMI)
W247.05 BOOL  ; A4右伺服位置6手动(HMI)
W247.06 BOOL  ; A4右伺服位置7手动(HMI)
W247.07 BOOL  ; A4右伺服位置8手动(HMI)
W247.08 BOOL  ; A4右伺服位置9手动(HMI)
W247.09 BOOL  ; A4右伺服位置10手动(HMI)
W247.10 BOOL  ; A4右伺服回原条件
W247.11 BOOL  ; A4右伺服运行锁定
W247.12 BOOL  ; A4右伺服定位条件
W247.13 BOOL  ; A4右伺服回原点手动(HMI)回原启动
W247.14 BOOL  ; A4右伺服错误清除(HMI)回原完成
W247.15 BOOL  ; A4右伺服辅助3
W248.00 BOOL  ; 正压伺服B回原点手动(HMI)
W248.01 BOOL  ; 正压伺服B错误清除(HMI)
W248.02 BOOL  ; 正压伺服BJOG高速(HMI)
W248.03 BOOL  ; 正压伺服BJOG低速（（HMI）
W248.04 BOOL  ; 正压伺服BJOG+（HMI）
W248.05 BOOL  ; 正压伺服BJOG-（HMI）
W248.06 BOOL  ; 正压伺服B初始位设置（HMI）
W248.07 BOOL  ; 正压伺服B减速位设置（HMI）
W248.08 BOOL  ; 正压伺服B等距热压位设置（HMI）
W248.09 BOOL  ; 正压伺服B预压退回位设置（HMI）
W248.10 BOOL  ; 正压伺服BMASK测试位设置（HMI）
W248.11 BOOL  ; 正压伺服B位置6设置（HMI）
W248.12 BOOL  ; 正压伺服B位置7设置（HMI）
W248.13 BOOL  ; 正压伺服B位置8设置（HMI）
W248.14 BOOL  ; 正压伺服B位置9设置（HMI）
W248.15 BOOL  ; 正压伺服B位置10设置（HMI）
W249.00 BOOL  ; 正压伺服B初始位手动(HMI)
W249.01 BOOL  ; 正压伺服B减速位手动(HMI)
W249.02 BOOL  ; 正压伺服B等距热压位手动(HMI)
W249.03 BOOL  ; 正压伺服B预压退回位手动(HMI)
W249.04 BOOL  ; 正压伺服BMASK测试位手动(HMI)
W249.05 BOOL  ; 正压伺服B位置6手动(HMI)
W249.06 BOOL  ; 正压伺服B位置7手动(HMI)
W249.07 BOOL  ; 正压伺服B位置8手动(HMI)
W249.08 BOOL  ; 正压伺服B位置9手动(HMI)
W249.09 BOOL  ; 正压伺服B位置10手动(HMI)
W249.10 BOOL  ; 正压伺服B回原条件
W249.11 BOOL  ; 正压伺服B运行锁定
W249.12 BOOL  ; 正压伺服B定位条件
W249.13 BOOL  ; 正压伺服B回原点手动(HMI)回原启动
W249.14 BOOL  ; 正压伺服B错误清除(HMI)回原完成
W249.15 BOOL  ; 正压伺服B辅助3
W250.00 BOOL  ; 压板平移伺服B回原点手动(HMI)
W250.01 BOOL  ; 压板平移伺服B错误清除(HMI)
W250.02 BOOL  ; 压板平移伺服BJOG高速(HMI)
W250.03 BOOL  ; 压板平移伺服BJOG低速（（HMI）
W250.04 BOOL  ; 压板平移伺服BJOG+（HMI）
W250.05 BOOL  ; 压板平移伺服BJOG-（HMI）
W250.06 BOOL  ; 压板平移伺服BA面取放位设置（HMI）
W250.07 BOOL  ; 压板平移伺服BB面取放位设置（HMI）
W250.08 BOOL  ; 压板平移伺服B位置3设置（HMI）
W250.09 BOOL  ; 压板平移伺服B位置4设置（HMI）
W250.10 BOOL  ; 压板平移伺服B位置5设置（HMI）
W250.11 BOOL  ; 压板平移伺服B位置6设置（HMI）
W250.12 BOOL  ; 压板平移伺服B位置7设置（HMI）
W250.13 BOOL  ; 压板平移伺服B位置8设置（HMI）
W250.14 BOOL  ; 压板平移伺服B位置9设置（HMI）
W250.15 BOOL  ; 压板平移伺服B位置10设置（HMI）
W251.00 BOOL  ; 压板平移伺服BA面取放位手动(HMI)
W251.01 BOOL  ; 压板平移伺服BB面取放位手动(HMI)
W251.02 BOOL  ; 压板平移伺服B位置3手动(HMI)
W251.03 BOOL  ; 压板平移伺服B位置4手动(HMI)
W251.04 BOOL  ; 压板平移伺服B位置5手动(HMI)
W251.05 BOOL  ; 压板平移伺服B位置6手动(HMI)
W251.06 BOOL  ; 压板平移伺服B位置7手动(HMI)
W251.07 BOOL  ; 压板平移伺服B位置8手动(HMI)
W251.08 BOOL  ; 压板平移伺服B位置9手动(HMI)
W251.09 BOOL  ; 压板平移伺服B位置10手动(HMI)
W251.10 BOOL  ; 压板平移伺服B回原条件
W251.11 BOOL  ; 压板平移伺服B运行锁定
W251.12 BOOL  ; 压板平移伺服B定位条件
W251.13 BOOL  ; 压板平移伺服B回原启动
W251.14 BOOL  ; 压板平移伺服B回原完成
W251.15 BOOL  ; 压板平移伺服B辅助3
W252.00 BOOL  ; B1左伺服回原点手动(HMI)
W252.01 BOOL  ; B1左伺服错误清除(HMI)
W252.02 BOOL  ; B1左伺服JOG高速(HMI)
W252.03 BOOL  ; B1左伺服JOG低速（（HMI）
W252.04 BOOL  ; B1左伺服JOG+（HMI）
W252.05 BOOL  ; B1左伺服JOG-（HMI）
W252.06 BOOL  ; B1左伺服待机位设置（HMI）
W252.07 BOOL  ; B1左伺服拨料退回位设置（HMI）
W252.08 BOOL  ; B1左伺服拨料位设置（HMI）
W252.09 BOOL  ; B1左伺服减速位设置（HMI）
W252.10 BOOL  ; B1左伺服等距热压位设置（HMI）
W252.11 BOOL  ; B1左伺服位置6设置（HMI）
W252.12 BOOL  ; B1左伺服位置7设置（HMI）
W252.13 BOOL  ; B1左伺服位置8设置（HMI）
W252.14 BOOL  ; B1左伺服位置9设置（HMI）
W252.15 BOOL  ; B1左伺服位置10设置（HMI）
W253.00 BOOL  ; B1左伺服待机位手动(HMI)
W253.01 BOOL  ; B1左伺服拨料退回位手动(HMI)
W253.02 BOOL  ; B1左伺服拨料位手动(HMI)
W253.03 BOOL  ; B1左伺服减速位手动(HMI)
W253.04 BOOL  ; B1左伺服等距热压位手动(HMI)
W253.05 BOOL  ; B1左伺服位置6手动(HMI)
W253.06 BOOL  ; B1左伺服位置7手动(HMI)
W253.07 BOOL  ; B1左伺服位置8手动(HMI)
W253.08 BOOL  ; B1左伺服位置9手动(HMI)
W253.09 BOOL  ; B1左伺服位置10手动(HMI)
W253.10 BOOL  ; B1左伺服回原条件
W253.11 BOOL  ; B1左伺服运行锁定
W253.12 BOOL  ; B1左伺服定位条件
W253.13 BOOL  ; B1左伺服回原启动
W253.14 BOOL  ; B1左伺服回原完成
W253.15 BOOL  ; B1左伺服辅助3
W254.00 BOOL  ; B1右伺服回原点手动(HMI)
W254.01 BOOL  ; B1右伺服错误清除(HMI)
W254.02 BOOL  ; B1右伺服JOG高速(HMI)
W254.03 BOOL  ; B1右伺服JOG低速（（HMI）
W254.04 BOOL  ; B1右伺服JOG+（HMI）
W254.05 BOOL  ; B1右伺服JOG-（HMI）
W254.06 BOOL  ; B1右伺服待机位设置（HMI）
W254.07 BOOL  ; B1右伺服拨料退回位设置（HMI）
W254.08 BOOL  ; B1右伺服拨料位设置（HMI）
W254.09 BOOL  ; B1右伺服减速位设置（HMI）
W254.10 BOOL  ; B1右伺服等距热压位设置（HMI）
W254.11 BOOL  ; B1右伺服位置6设置（HMI）
W254.12 BOOL  ; B1右伺服位置7设置（HMI）
W254.13 BOOL  ; B1右伺服位置8设置（HMI）
W254.14 BOOL  ; B1右伺服位置9设置（HMI）
W254.15 BOOL  ; B1右伺服位置10设置（HMI）
W255.00 BOOL  ; B1右伺服待机位手动(HMI)
W255.01 BOOL  ; B1右伺服拨料退回位手动(HMI)
W255.02 BOOL  ; B1右伺服拨料位手动(HMI)
W255.03 BOOL  ; B1右伺服减速位手动(HMI)
W255.04 BOOL  ; B1右伺服等距热压位手动(HMI)
W255.05 BOOL  ; B1右伺服位置6手动(HMI)
W255.06 BOOL  ; B1右伺服位置7手动(HMI)
W255.07 BOOL  ; B1右伺服位置8手动(HMI)
W255.08 BOOL  ; B1右伺服位置9手动(HMI)
W255.09 BOOL  ; B1右伺服位置10手动(HMI)
W255.10 BOOL  ; B1右伺服回原条件
W255.11 BOOL  ; B1右伺服运行锁定
W255.12 BOOL  ; B1右伺服定位条件
W255.13 BOOL  ; B1右伺服回原启动
W255.14 BOOL  ; B1右伺服回原完成
W255.15 BOOL  ; B1右伺服辅助3
W256.00 BOOL  ; B2左伺服回原点手动(HMI)
W256.01 BOOL  ; B2左伺服错误清除(HMI)
W256.02 BOOL  ; B2左伺服JOG高速(HMI)
W256.03 BOOL  ; B2左伺服JOG低速（（HMI）
W256.04 BOOL  ; B2左伺服JOG+（HMI）
W256.05 BOOL  ; B2左伺服JOG-（HMI）
W256.06 BOOL  ; B2左伺服待机位设置（HMI）
W256.07 BOOL  ; B2左伺服拨料退回位设置（HMI）
W256.08 BOOL  ; B2左伺服拨料位设置（HMI）
W256.09 BOOL  ; B2左伺服减速位设置（HMI）
W256.10 BOOL  ; B2左伺服等距热压位设置（HMI）
W256.11 BOOL  ; B2左伺服位置6设置（HMI）
W256.12 BOOL  ; B2左伺服位置7设置（HMI）
W256.13 BOOL  ; B2左伺服位置8设置（HMI）
W256.14 BOOL  ; B2左伺服位置9设置（HMI）
W256.15 BOOL  ; B2左伺服位置10设置（HMI）
W257.00 BOOL  ; B2左伺服待机位手动(HMI)
W257.01 BOOL  ; B2左伺服拨料退回位手动(HMI)
W257.02 BOOL  ; B2左伺服拨料位手动(HMI)
W257.03 BOOL  ; B2左伺服减速位手动(HMI)
W257.04 BOOL  ; B2左伺服等距热压位手动(HMI)
W257.05 BOOL  ; B2左伺服位置6手动(HMI)
W257.06 BOOL  ; B2左伺服位置7手动(HMI)
W257.07 BOOL  ; B2左伺服位置8手动(HMI)
W257.08 BOOL  ; B2左伺服位置9手动(HMI)
W257.09 BOOL  ; B2左伺服位置10手动(HMI)
W257.10 BOOL  ; B2左伺服回原条件
W257.11 BOOL  ; B2左伺服运行锁定
W257.12 BOOL  ; B2左伺服定位条件
W257.13 BOOL  ; B2左伺服回原启动
W257.14 BOOL  ; B2左伺服回原完成
W257.15 BOOL  ; B2左伺服辅助3
W258.00 BOOL  ; B2右伺服回原点手动(HMI)
W258.01 BOOL  ; B2右伺服错误清除(HMI)
W258.02 BOOL  ; B2右伺服JOG高速(HMI)
W258.03 BOOL  ; B2右伺服JOG低速（（HMI）
W258.04 BOOL  ; B2右伺服JOG+（HMI）
W258.05 BOOL  ; B2右伺服JOG-（HMI）
W258.06 BOOL  ; B2右伺服待机位设置（HMI）
W258.07 BOOL  ; B2右伺服拨料退回位设置（HMI）
W258.08 BOOL  ; B2右伺服拨料位设置（HMI）
W258.09 BOOL  ; B2右伺服减速位设置（HMI）
W258.10 BOOL  ; B2右伺服等距热压位设置（HMI）
W258.11 BOOL  ; B2右伺服位置6设置（HMI）
W258.12 BOOL  ; B2右伺服位置7设置（HMI）
W258.13 BOOL  ; B2右伺服位置8设置（HMI）
W258.14 BOOL  ; B2右伺服位置9设置（HMI）
W258.15 BOOL  ; B2右伺服位置10设置（HMI）
W259.00 BOOL  ; B2右伺服待机位手动(HMI)
W259.01 BOOL  ; B2右伺服拨料退回位手动(HMI)
W259.02 BOOL  ; B2右伺服拨料位手动(HMI)
W259.03 BOOL  ; B2右伺服减速位手动(HMI)
W259.04 BOOL  ; B2右伺服等距热压位手动(HMI)
W259.05 BOOL  ; B2右伺服位置6手动(HMI)
W259.06 BOOL  ; B2右伺服位置7手动(HMI)
W259.07 BOOL  ; B2右伺服位置8手动(HMI)
W259.08 BOOL  ; B2右伺服位置9手动(HMI)
W259.09 BOOL  ; B2右伺服位置10手动(HMI)
W259.10 BOOL  ; B2右伺服回原条件
W259.11 BOOL  ; B2右伺服运行锁定
W259.12 BOOL  ; B2右伺服定位条件
W259.13 BOOL  ; B2右伺服回原启动
W259.14 BOOL  ; B2右伺服回原完成
W259.15 BOOL  ; B2右伺服辅助3
W25.00 BOOL  ; 3ST_A手动切换允许输出标志
W25.01 BOOL  ; 3ST_A自动切换允许输出标志
W25.02 BOOL  ; 3ST_B手动切换允许输出标志
W25.03 BOOL  ; 3ST_B自动切换允许输出标志
W25.05 BOOL  ; 到出料等待位
W25.06 BOOL  ; A边无进料计时
W25.07 BOOL  ; 3ST_A A侧取料
W25.08 BOOL  ; 3ST_B A侧取料
W260.00 BOOL  ; B3左伺服回原点手动(HMI)
W260.01 BOOL  ; B3左伺服错误清除(HMI)
W260.02 BOOL  ; B3左伺服JOG高速(HMI)
W260.03 BOOL  ; B3左伺服JOG低速（（HMI）
W260.04 BOOL  ; B3左伺服JOG+（HMI）
W260.05 BOOL  ; B3左伺服JOG-（HMI）
W260.06 BOOL  ; B3左伺服待机位设置（HMI）
W260.07 BOOL  ; B3左伺服拨料退回位设置（HMI）
W260.08 BOOL  ; B3左伺服拨料位设置（HMI）
W260.09 BOOL  ; B3左伺服减速位设置（HMI）
W260.10 BOOL  ; B3左伺服等距热压位设置（HMI）
W260.11 BOOL  ; B3左伺服位置6设置（HMI）
W260.12 BOOL  ; B3左伺服位置7设置（HMI）
W260.13 BOOL  ; B3左伺服位置8设置（HMI）
W260.14 BOOL  ; B3左伺服位置9设置（HMI）
W260.15 BOOL  ; B3左伺服位置10设置（HMI）
W261.00 BOOL  ; B3左伺服待机位手动(HMI)
W261.01 BOOL  ; B3左伺服拨料退回位手动(HMI)
W261.02 BOOL  ; B3左伺服拨料位手动(HMI)
W261.03 BOOL  ; B3左伺服减速位手动(HMI)
W261.04 BOOL  ; B3左伺服等距热压位手动(HMI)
W261.05 BOOL  ; B3左伺服位置6手动(HMI)
W261.06 BOOL  ; B3左伺服位置7手动(HMI)
W261.07 BOOL  ; B3左伺服位置8手动(HMI)
W261.08 BOOL  ; B3左伺服位置9手动(HMI)
W261.09 BOOL  ; B3左伺服位置10手动(HMI)
W261.10 BOOL  ; B3左伺服回原条件
W261.11 BOOL  ; B3左伺服运行锁定
W261.12 BOOL  ; B3左伺服定位条件
W261.13 BOOL  ; B3左伺服回原启动
W261.14 BOOL  ; B3左伺服回原完成
W261.15 BOOL  ; B3左伺服辅助3
W262.00 BOOL  ; B3右伺服回原点手动(HMI)
W262.01 BOOL  ; B3右伺服错误清除(HMI)
W262.02 BOOL  ; B3右伺服JOG高速(HMI)
W262.03 BOOL  ; B3右伺服JOG低速（（HMI）
W262.04 BOOL  ; B3右伺服JOG+（HMI）
W262.05 BOOL  ; B3右伺服JOG-（HMI）
W262.06 BOOL  ; B3右伺服待机位设置（HMI）
W262.07 BOOL  ; B3右伺服拨料退回位设置（HMI）
W262.08 BOOL  ; B3右伺服拨料位设置（HMI）
W262.09 BOOL  ; B3右伺服减速位设置（HMI）
W262.10 BOOL  ; B3右伺服等距热压位设置（HMI）
W262.11 BOOL  ; B3右伺服位置6设置（HMI）
W262.12 BOOL  ; B3右伺服位置7设置（HMI）
